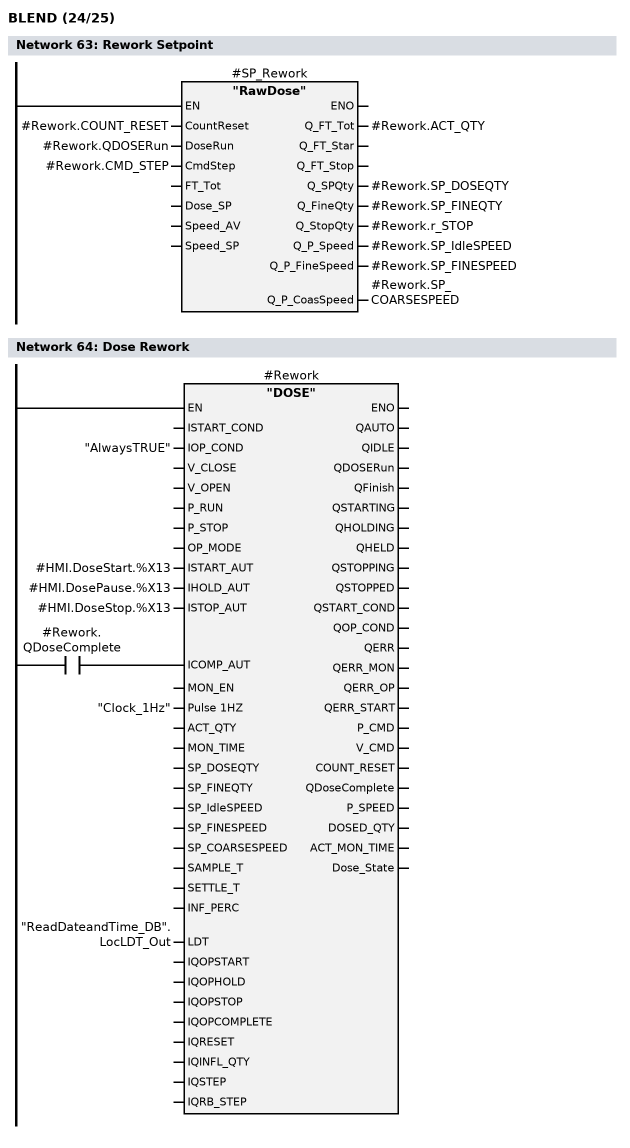
   RUNG wire#powerrail
      #SP_Rework(CountReset := #Rework.COUNT_RESET, DoseRun := #Rework.QDOSERun, CmdStep := #Rework.CMD_STEP, FT_Tot :=, Dose_SP :=, Speed_AV :=, Speed_SP :=, Q_FT_Tot => #Rework.ACT_QTY, Q_FT_Star =>, Q_FT_Stop =>, Q_SPQty => #Rework.SP_DOSEQTY, Q_FineQty => #Rework.SP_FINEQTY, Q_StopQty => #Rework.r_STOP, Q_P_Speed => #Rework.SP_IdleSPEED, Q_P_FineSpeed => #Rework.SP_FINESPEED, Q_P_CoasSpeed => #Rework.SP_COARSESPEED)
   END_RUNG
   // the same network as SCL:
   #SP_Rework(CountReset := #Rework.COUNT_RESET,   // "RawDose"
              DoseRun := #Rework.QDOSERun,
              CmdStep := #Rework.CMD_STEP,
              Q_FT_Tot => #Rework.ACT_QTY,
              Q_SPQty => #Rework.SP_DOSEQTY,
              Q_FineQty => #Rework.SP_FINEQTY,
              Q_StopQty => #Rework.r_STOP,
              Q_P_Speed => #Rework.SP_IdleSPEED,
              Q_P_FineSpeed => #Rework.SP_FINESPEED,
              Q_P_CoasSpeed => #Rework.SP_COARSESPEED);
END_REGION

REGION Network 64: Dose Rework
   RUNG wire#powerrail
      #Rework(ICOMP_AUT := wire#w1, ISTART_COND :=, IOP_COND := "AlwaysTRUE", V_CLOSE :=, V_OPEN :=, P_RUN :=, P_STOP :=, OP_MODE :=, ISTART_AUT := #HMI.DoseStart.%X13, IHOLD_AUT := #HMI.DosePause.%X13, ISTOP_AUT := #HMI.DoseStop.%X13, MON_EN :=, "Pulse 1HZ" := "Clock_1Hz", ACT_QTY :=, MON_TIME :=, SP_DOSEQTY :=, SP_FINEQTY :=, SP_IdleSPEED :=, SP_FINESPEED :=, SP_COARSESPEED :=, SAMPLE_T :=, SETTLE_T :=, INF_PERC :=, LDT := "ReadDateandTime_DB".LocLDT_Out, IQOPSTART :=, IQOPHOLD :=, IQOPSTOP :=, IQOPCOMPLETE :=, IQRESET :=, IQINFL_QTY :=, IQSTEP :=, IQRB_STEP :=, QAUTO =>, QIDLE =>, QDOSERun =>, QFinish =>, QSTARTING =>, QHOLDING =>, QHELD =>, QSTOPPING =>, QSTOPPED =>, QSTART_COND =>, QOP_COND =>, QERR =>, QERR_MON =>, QERR_OP =>, QERR_START =>, P_CMD =>, V_CMD =>, COUNT_RESET =>, QDoseComplete =>, P_SPEED =>, DOSED_QTY =>, ACT_MON_TIME =>, Dose_State =>)
   END_RUNG
   RUNG wire#powerrail
      Contact( #Rework.QDoseComplete )
   END_RUNG wire#w1
   // the same network as SCL:
   #Rework(IOP_COND := "AlwaysTRUE",   // "DOSE"
           ISTART_AUT := #HMI.DoseStart.%X13,
           IHOLD_AUT := #HMI.DosePause.%X13,
           ISTOP_AUT := #HMI.DoseStop.%X13,
           ICOMP_AUT := #Rework.QDoseComplete,
           "Pulse 1HZ" := "Clock_1Hz",
           LDT := "ReadDateandTime_DB".LocLDT_Out);
END_REGION

REGION Network 65: Dose Rework Enable Command
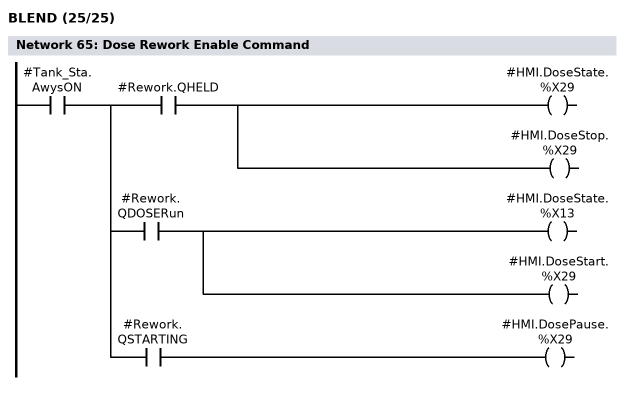
   RUNG wire#powerrail
      Contact( #Tank_Sta.AwysON )
      wire#w1
      Contact( #Rework.QHELD )
      wire#w2
      Coil( #HMI.DoseState.%X29 )
   END_RUNG
   RUNG wire#w2
      Coil( #HMI.DoseStop.%X29 )
   END_RUNG
   RUNG wire#w1
      Contact( #Rework.QDOSERun )
      wire#w3
      Coil( #HMI.DoseState.%X13 )
   END_RUNG
   RUNG wire#w3
      Coil( #HMI.DoseStart.%X29 )
   END_RUNG
   RUNG wire#w1
      Contact( #Rework.QSTARTING )
      Coil( #HMI.DosePause.%X29 )
   END_RUNG
   // the same network as SCL:
   #HMI.DoseState.%X29 := #Tank_Sta.AwysON AND #Rework.QHELD;
   #HMI.DoseStop.%X29 := #HMI.DoseState.%X29;
   #HMI.DoseState.%X13 := #Tank_Sta.AwysON AND #Rework.QDOSERun;
   #HMI.DoseStart.%X29 := #HMI.DoseState.%X13;
   #HMI.DosePause.%X29 := #Tank_Sta.AwysON AND #Rework.QSTARTING;
END_REGION
END_FUNCTION_BLOCK

FUNCTION "Blending" : Void   // FC8, LAD
{ S7_Optimized_Access := 'TRUE' }
VERSION : 0.1
// stored: AutoNumber true, IsIECCheckEnabled false, SetENOAutomatically false, UDAEnableTagReadback false
   VAR_TEMP   // added for the SCL form of the ladder/FBD networks
      _w1 : Bool;
   END_VAR
BEGIN

REGION Network 1
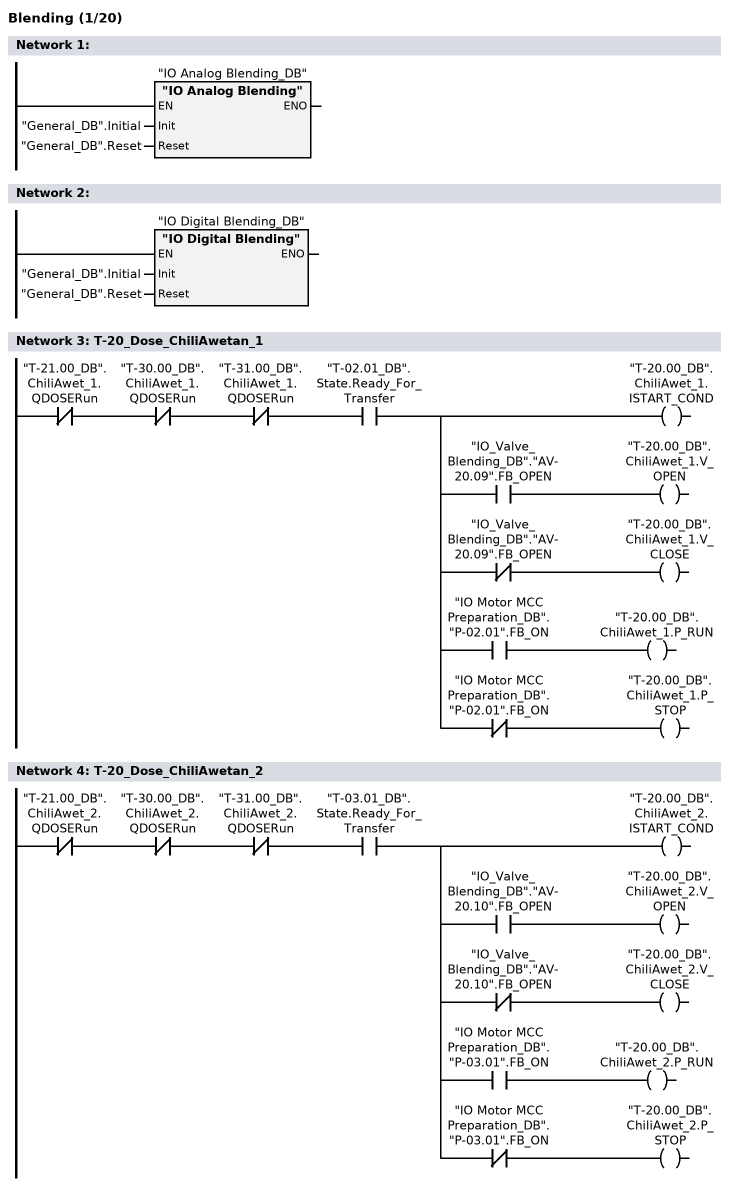
   RUNG wire#powerrail
      "IO Analog Blending_DB"(Init := "General_DB".Initial, Reset := "General_DB".Reset)
   END_RUNG
   // the same network as SCL:
   "IO Analog Blending_DB"(Init := "General_DB".Initial, Reset := "General_DB".Reset);   // "IO Analog Blending"
END_REGION

REGION Network 2
   RUNG wire#powerrail
      "IO Digital Blending_DB"(Init := "General_DB".Initial, Reset := "General_DB".Reset)
   END_RUNG
   // the same network as SCL:
   "IO Digital Blending_DB"(Init := "General_DB".Initial, Reset := "General_DB".Reset);   // "IO Digital Blending"
END_REGION

REGION Network 3: T-20_Dose_ChiliAwetan_1
   RUNG wire#powerrail
      I_Contact( "T-21.00_DB".ChiliAwet_1.QDOSERun )
      I_Contact( "T-30.00_DB".ChiliAwet_1.QDOSERun )
      I_Contact( "T-31.00_DB".ChiliAwet_1.QDOSERun )
      Contact( "T-02.01_DB".State.Ready_For_Transfer )
      wire#w1
      Coil( "T-20.00_DB".ChiliAwet_1.ISTART_COND )
   END_RUNG
   RUNG wire#w1
      Contact( "IO_Valve_Blending_DB"."AV-20.09".FB_OPEN )
      Coil( "T-20.00_DB".ChiliAwet_1.V_OPEN )
   END_RUNG
   RUNG wire#w1
      I_Contact( "IO_Valve_Blending_DB"."AV-20.09".FB_OPEN )
      Coil( "T-20.00_DB".ChiliAwet_1.V_CLOSE )
   END_RUNG
   RUNG wire#w1
      Contact( "IO Motor MCC Preparation_DB"."P-02.01".FB_ON )
      Coil( "T-20.00_DB".ChiliAwet_1.P_RUN )
   END_RUNG
   RUNG wire#w1
      I_Contact( "IO Motor MCC Preparation_DB"."P-02.01".FB_ON )
      Coil( "T-20.00_DB".ChiliAwet_1.P_STOP )
   END_RUNG
   // the same network as SCL:
   "T-20.00_DB".ChiliAwet_1.ISTART_COND := NOT "T-21.00_DB".ChiliAwet_1.QDOSERun AND NOT "T-30.00_DB".ChiliAwet_1.QDOSERun AND NOT "T-31.00_DB".ChiliAwet_1.QDOSERun AND "T-02.01_DB".State.Ready_For_Transfer;
   "T-20.00_DB".ChiliAwet_1.V_OPEN := "T-20.00_DB".ChiliAwet_1.ISTART_COND AND "IO_Valve_Blending_DB"."AV-20.09".FB_OPEN;
   "T-20.00_DB".ChiliAwet_1.V_CLOSE := "T-20.00_DB".ChiliAwet_1.ISTART_COND AND NOT "IO_Valve_Blending_DB"."AV-20.09".FB_OPEN;
   "T-20.00_DB".ChiliAwet_1.P_RUN := "T-20.00_DB".ChiliAwet_1.ISTART_COND AND "IO Motor MCC Preparation_DB"."P-02.01".FB_ON;
   "T-20.00_DB".ChiliAwet_1.P_STOP := "T-20.00_DB".ChiliAwet_1.ISTART_COND AND NOT "IO Motor MCC Preparation_DB"."P-02.01".FB_ON;
END_REGION

REGION Network 4: T-20_Dose_ChiliAwetan_2
   RUNG wire#powerrail
      I_Contact( "T-21.00_DB".ChiliAwet_2.QDOSERun )
      I_Contact( "T-30.00_DB".ChiliAwet_2.QDOSERun )
      I_Contact( "T-31.00_DB".ChiliAwet_2.QDOSERun )
      Contact( "T-03.01_DB".State.Ready_For_Transfer )
      wire#w1
      Coil( "T-20.00_DB".ChiliAwet_2.ISTART_COND )
   END_RUNG
   RUNG wire#w1
      Contact( "IO_Valve_Blending_DB"."AV-20.10".FB_OPEN )
      Coil( "T-20.00_DB".ChiliAwet_2.V_OPEN )
   END_RUNG
   RUNG wire#w1
      I_Contact( "IO_Valve_Blending_DB"."AV-20.10".FB_OPEN )
      Coil( "T-20.00_DB".ChiliAwet_2.V_CLOSE )
   END_RUNG
   RUNG wire#w1
      Contact( "IO Motor MCC Preparation_DB"."P-03.01".FB_ON )
      Coil( "T-20.00_DB".ChiliAwet_2.P_RUN )
   END_RUNG
   RUNG wire#w1
      I_Contact( "IO Motor MCC Preparation_DB"."P-03.01".FB_ON )
      Coil( "T-20.00_DB".ChiliAwet_2.P_STOP )
   END_RUNG
   // the same network as SCL:
   "T-20.00_DB".ChiliAwet_2.ISTART_COND := NOT "T-21.00_DB".ChiliAwet_2.QDOSERun AND NOT "T-30.00_DB".ChiliAwet_2.QDOSERun AND NOT "T-31.00_DB".ChiliAwet_2.QDOSERun AND "T-03.01_DB".State.Ready_For_Transfer;
   "T-20.00_DB".ChiliAwet_2.V_OPEN := "T-20.00_DB".ChiliAwet_2.ISTART_COND AND "IO_Valve_Blending_DB"."AV-20.10".FB_OPEN;
   "T-20.00_DB".ChiliAwet_2.V_CLOSE := "T-20.00_DB".ChiliAwet_2.ISTART_COND AND NOT "IO_Valve_Blending_DB"."AV-20.10".FB_OPEN;
   "T-20.00_DB".ChiliAwet_2.P_RUN := "T-20.00_DB".ChiliAwet_2.ISTART_COND AND "IO Motor MCC Preparation_DB"."P-03.01".FB_ON;
   "T-20.00_DB".ChiliAwet_2.P_STOP := "T-20.00_DB".ChiliAwet_2.ISTART_COND AND NOT "IO Motor MCC Preparation_DB"."P-03.01".FB_ON;
END_REGION

REGION Network 5: T-20_Dose_ChiliAwetan_3
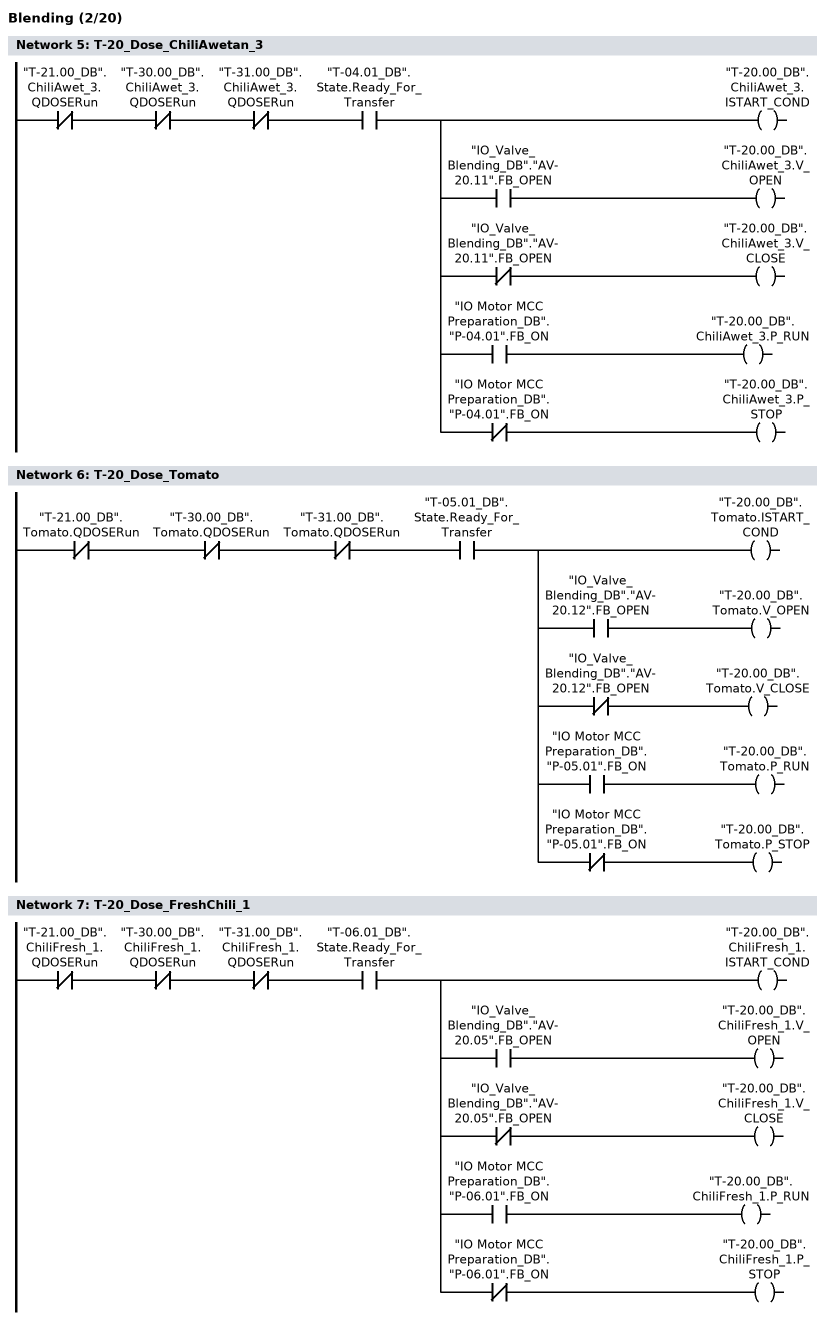
   RUNG wire#powerrail
      I_Contact( "T-21.00_DB".ChiliAwet_3.QDOSERun )
      I_Contact( "T-30.00_DB".ChiliAwet_3.QDOSERun )
      I_Contact( "T-31.00_DB".ChiliAwet_3.QDOSERun )
      Contact( "T-04.01_DB".State.Ready_For_Transfer )
      wire#w1
      Coil( "T-20.00_DB".ChiliAwet_3.ISTART_COND )
   END_RUNG
   RUNG wire#w1
      Contact( "IO_Valve_Blending_DB"."AV-20.11".FB_OPEN )
      Coil( "T-20.00_DB".ChiliAwet_3.V_OPEN )
   END_RUNG
   RUNG wire#w1
      I_Contact( "IO_Valve_Blending_DB"."AV-20.11".FB_OPEN )
      Coil( "T-20.00_DB".ChiliAwet_3.V_CLOSE )
   END_RUNG
   RUNG wire#w1
      Contact( "IO Motor MCC Preparation_DB"."P-04.01".FB_ON )
      Coil( "T-20.00_DB".ChiliAwet_3.P_RUN )
   END_RUNG
   RUNG wire#w1
      I_Contact( "IO Motor MCC Preparation_DB"."P-04.01".FB_ON )
      Coil( "T-20.00_DB".ChiliAwet_3.P_STOP )
   END_RUNG
   // the same network as SCL:
   "T-20.00_DB".ChiliAwet_3.ISTART_COND := NOT "T-21.00_DB".ChiliAwet_3.QDOSERun AND NOT "T-30.00_DB".ChiliAwet_3.QDOSERun AND NOT "T-31.00_DB".ChiliAwet_3.QDOSERun AND "T-04.01_DB".State.Ready_For_Transfer;
   "T-20.00_DB".ChiliAwet_3.V_OPEN := "T-20.00_DB".ChiliAwet_3.ISTART_COND AND "IO_Valve_Blending_DB"."AV-20.11".FB_OPEN;
   "T-20.00_DB".ChiliAwet_3.V_CLOSE := "T-20.00_DB".ChiliAwet_3.ISTART_COND AND NOT "IO_Valve_Blending_DB"."AV-20.11".FB_OPEN;
   "T-20.00_DB".ChiliAwet_3.P_RUN := "T-20.00_DB".ChiliAwet_3.ISTART_COND AND "IO Motor MCC Preparation_DB"."P-04.01".FB_ON;
   "T-20.00_DB".ChiliAwet_3.P_STOP := "T-20.00_DB".ChiliAwet_3.ISTART_COND AND NOT "IO Motor MCC Preparation_DB"."P-04.01".FB_ON;
END_REGION

REGION Network 6: T-20_Dose_Tomato
   RUNG wire#powerrail
      I_Contact( "T-21.00_DB".Tomato.QDOSERun )
      I_Contact( "T-30.00_DB".Tomato.QDOSERun )
      I_Contact( "T-31.00_DB".Tomato.QDOSERun )
      Contact( "T-05.01_DB".State.Ready_For_Transfer )
      wire#w1
      Coil( "T-20.00_DB".Tomato.ISTART_COND )
   END_RUNG
   RUNG wire#w1
      Contact( "IO_Valve_Blending_DB"."AV-20.12".FB_OPEN )
      Coil( "T-20.00_DB".Tomato.V_OPEN )
   END_RUNG
   RUNG wire#w1
      I_Contact( "IO_Valve_Blending_DB"."AV-20.12".FB_OPEN )
      Coil( "T-20.00_DB".Tomato.V_CLOSE )
   END_RUNG
   RUNG wire#w1
      Contact( "IO Motor MCC Preparation_DB"."P-05.01".FB_ON )
      Coil( "T-20.00_DB".Tomato.P_RUN )
   END_RUNG
   RUNG wire#w1
      I_Contact( "IO Motor MCC Preparation_DB"."P-05.01".FB_ON )
      Coil( "T-20.00_DB".Tomato.P_STOP )
   END_RUNG
   // the same network as SCL:
   "T-20.00_DB".Tomato.ISTART_COND := NOT "T-21.00_DB".Tomato.QDOSERun AND NOT "T-30.00_DB".Tomato.QDOSERun AND NOT "T-31.00_DB".Tomato.QDOSERun AND "T-05.01_DB".State.Ready_For_Transfer;
   "T-20.00_DB".Tomato.V_OPEN := "T-20.00_DB".Tomato.ISTART_COND AND "IO_Valve_Blending_DB"."AV-20.12".FB_OPEN;
   "T-20.00_DB".Tomato.V_CLOSE := "T-20.00_DB".Tomato.ISTART_COND AND NOT "IO_Valve_Blending_DB"."AV-20.12".FB_OPEN;
   "T-20.00_DB".Tomato.P_RUN := "T-20.00_DB".Tomato.ISTART_COND AND "IO Motor MCC Preparation_DB"."P-05.01".FB_ON;
   "T-20.00_DB".Tomato.P_STOP := "T-20.00_DB".Tomato.ISTART_COND AND NOT "IO Motor MCC Preparation_DB"."P-05.01".FB_ON;
END_REGION

REGION Network 7: T-20_Dose_FreshChili_1
   RUNG wire#powerrail
      I_Contact( "T-21.00_DB".ChiliFresh_1.QDOSERun )
      I_Contact( "T-30.00_DB".ChiliFresh_1.QDOSERun )
      I_Contact( "T-31.00_DB".ChiliFresh_1.QDOSERun )
      Contact( "T-06.01_DB".State.Ready_For_Transfer )
      wire#w1
      Coil( "T-20.00_DB".ChiliFresh_1.ISTART_COND )
   END_RUNG
   RUNG wire#w1
      Contact( "IO_Valve_Blending_DB"."AV-20.05".FB_OPEN )
      Coil( "T-20.00_DB".ChiliFresh_1.V_OPEN )
   END_RUNG
   RUNG wire#w1
      I_Contact( "IO_Valve_Blending_DB"."AV-20.05".FB_OPEN )
      Coil( "T-20.00_DB".ChiliFresh_1.V_CLOSE )
   END_RUNG
   RUNG wire#w1
      Contact( "IO Motor MCC Preparation_DB"."P-06.01".FB_ON )
      Coil( "T-20.00_DB".ChiliFresh_1.P_RUN )
   END_RUNG
   RUNG wire#w1
      I_Contact( "IO Motor MCC Preparation_DB"."P-06.01".FB_ON )
      Coil( "T-20.00_DB".ChiliFresh_1.P_STOP )
   END_RUNG
   // the same network as SCL:
   "T-20.00_DB".ChiliFresh_1.ISTART_COND := NOT "T-21.00_DB".ChiliFresh_1.QDOSERun AND NOT "T-30.00_DB".ChiliFresh_1.QDOSERun AND NOT "T-31.00_DB".ChiliFresh_1.QDOSERun AND "T-06.01_DB".State.Ready_For_Transfer;
   "T-20.00_DB".ChiliFresh_1.V_OPEN := "T-20.00_DB".ChiliFresh_1.ISTART_COND AND "IO_Valve_Blending_DB"."AV-20.05".FB_OPEN;
   "T-20.00_DB".ChiliFresh_1.V_CLOSE := "T-20.00_DB".ChiliFresh_1.ISTART_COND AND NOT "IO_Valve_Blending_DB"."AV-20.05".FB_OPEN;
   "T-20.00_DB".ChiliFresh_1.P_RUN := "T-20.00_DB".ChiliFresh_1.ISTART_COND AND "IO Motor MCC Preparation_DB"."P-06.01".FB_ON;
   "T-20.00_DB".ChiliFresh_1.P_STOP := "T-20.00_DB".ChiliFresh_1.ISTART_COND AND NOT "IO Motor MCC Preparation_DB"."P-06.01".FB_ON;
END_REGION

REGION Network 8: T-20_Dose_FreshChili_2
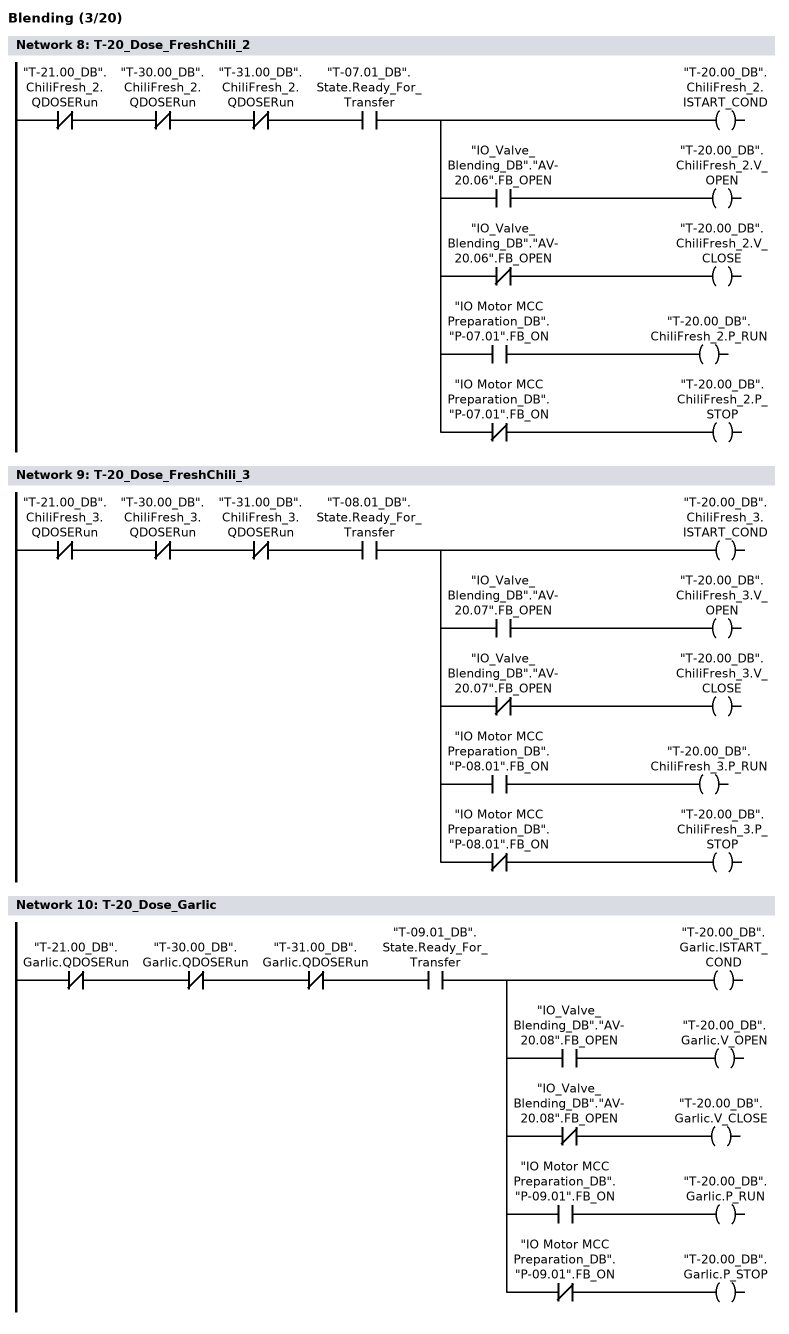
   RUNG wire#powerrail
      I_Contact( "T-21.00_DB".ChiliFresh_2.QDOSERun )
      I_Contact( "T-30.00_DB".ChiliFresh_2.QDOSERun )
      I_Contact( "T-31.00_DB".ChiliFresh_2.QDOSERun )
      Contact( "T-07.01_DB".State.Ready_For_Transfer )
      wire#w1
      Coil( "T-20.00_DB".ChiliFresh_2.ISTART_COND )
   END_RUNG
   RUNG wire#w1
      Contact( "IO_Valve_Blending_DB"."AV-20.06".FB_OPEN )
      Coil( "T-20.00_DB".ChiliFresh_2.V_OPEN )
   END_RUNG
   RUNG wire#w1
      I_Contact( "IO_Valve_Blending_DB"."AV-20.06".FB_OPEN )
      Coil( "T-20.00_DB".ChiliFresh_2.V_CLOSE )
   END_RUNG
   RUNG wire#w1
      Contact( "IO Motor MCC Preparation_DB"."P-07.01".FB_ON )
      Coil( "T-20.00_DB".ChiliFresh_2.P_RUN )
   END_RUNG
   RUNG wire#w1
      I_Contact( "IO Motor MCC Preparation_DB"."P-07.01".FB_ON )
      Coil( "T-20.00_DB".ChiliFresh_2.P_STOP )
   END_RUNG
   // the same network as SCL:
   "T-20.00_DB".ChiliFresh_2.ISTART_COND := NOT "T-21.00_DB".ChiliFresh_2.QDOSERun AND NOT "T-30.00_DB".ChiliFresh_2.QDOSERun AND NOT "T-31.00_DB".ChiliFresh_2.QDOSERun AND "T-07.01_DB".State.Ready_For_Transfer;
   "T-20.00_DB".ChiliFresh_2.V_OPEN := "T-20.00_DB".ChiliFresh_2.ISTART_COND AND "IO_Valve_Blending_DB"."AV-20.06".FB_OPEN;
   "T-20.00_DB".ChiliFresh_2.V_CLOSE := "T-20.00_DB".ChiliFresh_2.ISTART_COND AND NOT "IO_Valve_Blending_DB"."AV-20.06".FB_OPEN;
   "T-20.00_DB".ChiliFresh_2.P_RUN := "T-20.00_DB".ChiliFresh_2.ISTART_COND AND "IO Motor MCC Preparation_DB"."P-07.01".FB_ON;
   "T-20.00_DB".ChiliFresh_2.P_STOP := "T-20.00_DB".ChiliFresh_2.ISTART_COND AND NOT "IO Motor MCC Preparation_DB"."P-07.01".FB_ON;
END_REGION

REGION Network 9: T-20_Dose_FreshChili_3
   RUNG wire#powerrail
      I_Contact( "T-21.00_DB".ChiliFresh_3.QDOSERun )
      I_Contact( "T-30.00_DB".ChiliFresh_3.QDOSERun )
      I_Contact( "T-31.00_DB".ChiliFresh_3.QDOSERun )
      Contact( "T-08.01_DB".State.Ready_For_Transfer )
      wire#w1
      Coil( "T-20.00_DB".ChiliFresh_3.ISTART_COND )
   END_RUNG
   RUNG wire#w1
      Contact( "IO_Valve_Blending_DB"."AV-20.07".FB_OPEN )
      Coil( "T-20.00_DB".ChiliFresh_3.V_OPEN )
   END_RUNG
   RUNG wire#w1
      I_Contact( "IO_Valve_Blending_DB"."AV-20.07".FB_OPEN )
      Coil( "T-20.00_DB".ChiliFresh_3.V_CLOSE )
   END_RUNG
   RUNG wire#w1
      Contact( "IO Motor MCC Preparation_DB"."P-08.01".FB_ON )
      Coil( "T-20.00_DB".ChiliFresh_3.P_RUN )
   END_RUNG
   RUNG wire#w1
      I_Contact( "IO Motor MCC Preparation_DB"."P-08.01".FB_ON )
      Coil( "T-20.00_DB".ChiliFresh_3.P_STOP )
   END_RUNG
   // the same network as SCL:
   "T-20.00_DB".ChiliFresh_3.ISTART_COND := NOT "T-21.00_DB".ChiliFresh_3.QDOSERun AND NOT "T-30.00_DB".ChiliFresh_3.QDOSERun AND NOT "T-31.00_DB".ChiliFresh_3.QDOSERun AND "T-08.01_DB".State.Ready_For_Transfer;
   "T-20.00_DB".ChiliFresh_3.V_OPEN := "T-20.00_DB".ChiliFresh_3.ISTART_COND AND "IO_Valve_Blending_DB"."AV-20.07".FB_OPEN;
   "T-20.00_DB".ChiliFresh_3.V_CLOSE := "T-20.00_DB".ChiliFresh_3.ISTART_COND AND NOT "IO_Valve_Blending_DB"."AV-20.07".FB_OPEN;
   "T-20.00_DB".ChiliFresh_3.P_RUN := "T-20.00_DB".ChiliFresh_3.ISTART_COND AND "IO Motor MCC Preparation_DB"."P-08.01".FB_ON;
   "T-20.00_DB".ChiliFresh_3.P_STOP := "T-20.00_DB".ChiliFresh_3.ISTART_COND AND NOT "IO Motor MCC Preparation_DB"."P-08.01".FB_ON;
END_REGION

REGION Network 10: T-20_Dose_Garlic
   RUNG wire#powerrail
      I_Contact( "T-21.00_DB".Garlic.QDOSERun )
      I_Contact( "T-30.00_DB".Garlic.QDOSERun )
      I_Contact( "T-31.00_DB".Garlic.QDOSERun )
      Contact( "T-09.01_DB".State.Ready_For_Transfer )
      wire#w1
      Coil( "T-20.00_DB".Garlic.ISTART_COND )
   END_RUNG
   RUNG wire#w1
      Contact( "IO_Valve_Blending_DB"."AV-20.08".FB_OPEN )
      Coil( "T-20.00_DB".Garlic.V_OPEN )
   END_RUNG
   RUNG wire#w1
      I_Contact( "IO_Valve_Blending_DB"."AV-20.08".FB_OPEN )
      Coil( "T-20.00_DB".Garlic.V_CLOSE )
   END_RUNG
   RUNG wire#w1
      Contact( "IO Motor MCC Preparation_DB"."P-09.01".FB_ON )
      Coil( "T-20.00_DB".Garlic.P_RUN )
   END_RUNG
   RUNG wire#w1
      I_Contact( "IO Motor MCC Preparation_DB"."P-09.01".FB_ON )
      Coil( "T-20.00_DB".Garlic.P_STOP )
   END_RUNG
   // the same network as SCL:
   "T-20.00_DB".Garlic.ISTART_COND := NOT "T-21.00_DB".Garlic.QDOSERun AND NOT "T-30.00_DB".Garlic.QDOSERun AND NOT "T-31.00_DB".Garlic.QDOSERun AND "T-09.01_DB".State.Ready_For_Transfer;
   "T-20.00_DB".Garlic.V_OPEN := "T-20.00_DB".Garlic.ISTART_COND AND "IO_Valve_Blending_DB"."AV-20.08".FB_OPEN;
   "T-20.00_DB".Garlic.V_CLOSE := "T-20.00_DB".Garlic.ISTART_COND AND NOT "IO_Valve_Blending_DB"."AV-20.08".FB_OPEN;
   "T-20.00_DB".Garlic.P_RUN := "T-20.00_DB".Garlic.ISTART_COND AND "IO Motor MCC Preparation_DB"."P-09.01".FB_ON;
   "T-20.00_DB".Garlic.P_STOP := "T-20.00_DB".Garlic.ISTART_COND AND NOT "IO Motor MCC Preparation_DB"."P-09.01".FB_ON;
END_REGION

REGION Network 11: T-20_Dose_Vinegar
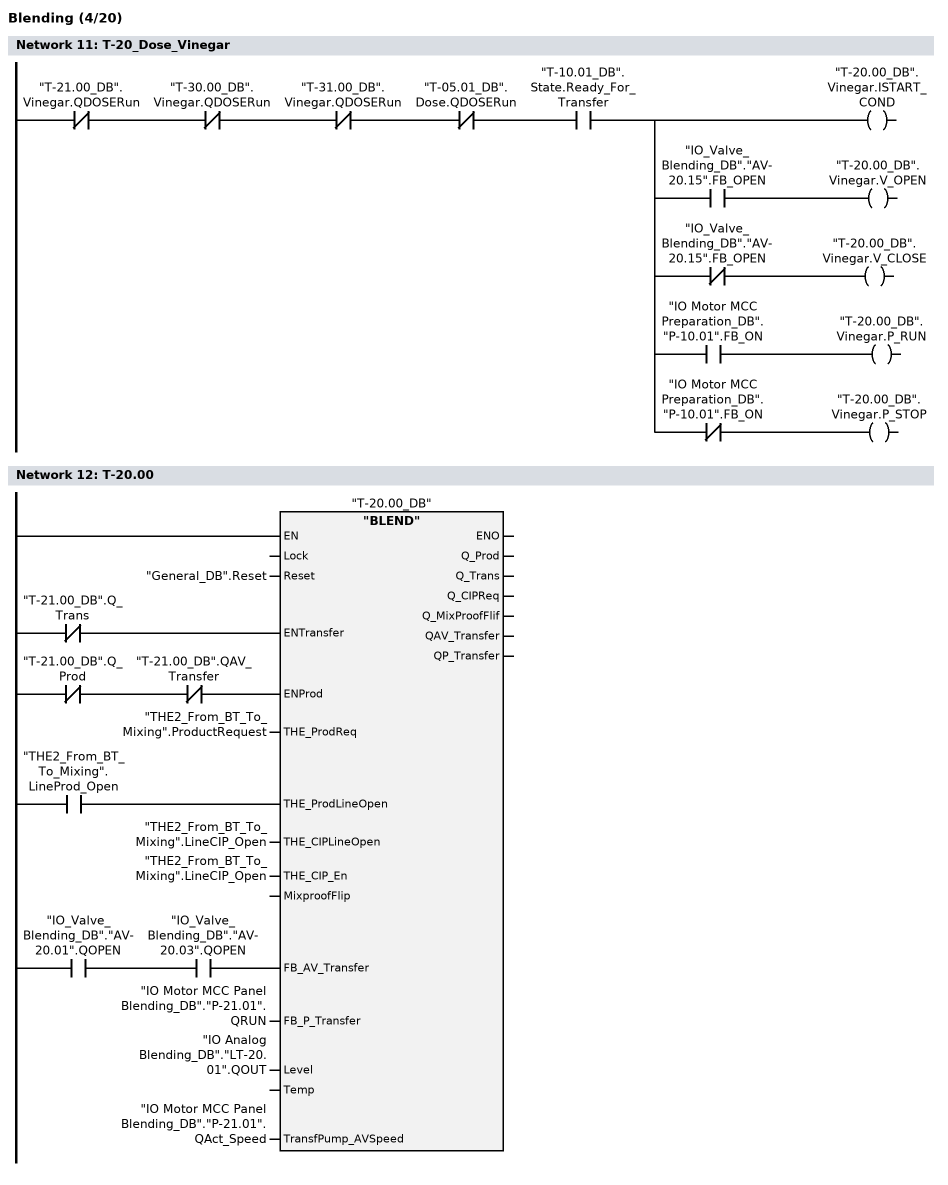
   RUNG wire#powerrail
      I_Contact( "T-21.00_DB".Vinegar.QDOSERun )
      I_Contact( "T-30.00_DB".Vinegar.QDOSERun )
      I_Contact( "T-31.00_DB".Vinegar.QDOSERun )
      I_Contact( "T-05.01_DB".Dose.QDOSERun )
      Contact( "T-10.01_DB".State.Ready_For_Transfer )
      wire#w1
      Coil( "T-20.00_DB".Vinegar.ISTART_COND )
   END_RUNG
   RUNG wire#w1
      Contact( "IO_Valve_Blending_DB"."AV-20.15".FB_OPEN )
      Coil( "T-20.00_DB".Vinegar.V_OPEN )
   END_RUNG
   RUNG wire#w1
      I_Contact( "IO_Valve_Blending_DB"."AV-20.15".FB_OPEN )
      Coil( "T-20.00_DB".Vinegar.V_CLOSE )
   END_RUNG
   RUNG wire#w1
      Contact( "IO Motor MCC Preparation_DB"."P-10.01".FB_ON )
      Coil( "T-20.00_DB".Vinegar.P_RUN )
   END_RUNG
   RUNG wire#w1
      I_Contact( "IO Motor MCC Preparation_DB"."P-10.01".FB_ON )
      Coil( "T-20.00_DB".Vinegar.P_STOP )
   END_RUNG
   // the same network as SCL:
   "T-20.00_DB".Vinegar.ISTART_COND := NOT "T-21.00_DB".Vinegar.QDOSERun AND NOT "T-30.00_DB".Vinegar.QDOSERun AND NOT "T-31.00_DB".Vinegar.QDOSERun AND NOT "T-05.01_DB".Dose.QDOSERun AND "T-10.01_DB".State.Ready_For_Transfer;
   "T-20.00_DB".Vinegar.V_OPEN := "T-20.00_DB".Vinegar.ISTART_COND AND "IO_Valve_Blending_DB"."AV-20.15".FB_OPEN;
   "T-20.00_DB".Vinegar.V_CLOSE := "T-20.00_DB".Vinegar.ISTART_COND AND NOT "IO_Valve_Blending_DB"."AV-20.15".FB_OPEN;
   "T-20.00_DB".Vinegar.P_RUN := "T-20.00_DB".Vinegar.ISTART_COND AND "IO Motor MCC Preparation_DB"."P-10.01".FB_ON;
   "T-20.00_DB".Vinegar.P_STOP := "T-20.00_DB".Vinegar.ISTART_COND AND NOT "IO Motor MCC Preparation_DB"."P-10.01".FB_ON;
END_REGION

REGION Network 12: T-20.00
   RUNG wire#powerrail
      "T-20.00_DB"(ENTransfer := wire#w1, ENProd := wire#w2, THE_ProdLineOpen := wire#w3, FB_AV_Transfer := wire#w4, Lock :=, Reset := "General_DB".Reset, THE_ProdReq := "THE2_From_BT_To_Mixing".ProductRequest, THE_CIPLineOpen := "THE2_From_BT_To_Mixing".LineCIP_Open, THE_CIP_En := "THE2_From_BT_To_Mixing".LineCIP_Open, MixproofFlip :=, FB_P_Transfer := "IO Motor MCC Panel Blending_DB"."P-21.01".QRUN, Level := "IO Analog Blending_DB"."LT-20.01".QOUT, Temp :=, TransfPump_AVSpeed := "IO Motor MCC Panel Blending_DB"."P-21.01".QAct_Speed, Q_Prod =>, Q_Trans =>, Q_CIPReq =>, Q_MixProofFlif =>, QAV_Transfer =>, QP_Transfer =>)
   END_RUNG
   RUNG wire#powerrail
      I_Contact( "T-21.00_DB".Q_Trans )
   END_RUNG wire#w1
   RUNG wire#powerrail
      I_Contact( "T-21.00_DB".Q_Prod )
      I_Contact( "T-21.00_DB".QAV_Transfer )
   END_RUNG wire#w2
   RUNG wire#powerrail
      Contact( "THE2_From_BT_To_Mixing".LineProd_Open )
   END_RUNG wire#w3
   RUNG wire#powerrail
      Contact( "IO_Valve_Blending_DB"."AV-20.01".QOPEN )
      Contact( "IO_Valve_Blending_DB"."AV-20.03".QOPEN )
   END_RUNG wire#w4
   // the same network as SCL:
   "T-20.00_DB"(Reset := "General_DB".Reset,   // "BLEND"
                ENTransfer := NOT "T-21.00_DB".Q_Trans,
                ENProd := NOT "T-21.00_DB".Q_Prod AND NOT "T-21.00_DB".QAV_Transfer,
                THE_ProdReq := "THE2_From_BT_To_Mixing".ProductRequest,
                THE_ProdLineOpen := "THE2_From_BT_To_Mixing".LineProd_Open,
                THE_CIPLineOpen := "THE2_From_BT_To_Mixing".LineCIP_Open,
                THE_CIP_En := "THE2_From_BT_To_Mixing".LineCIP_Open,
                FB_AV_Transfer := "IO_Valve_Blending_DB"."AV-20.01".QOPEN AND "IO_Valve_Blending_DB"."AV-20.03".QOPEN,
                FB_P_Transfer := "IO Motor MCC Panel Blending_DB"."P-21.01".QRUN,
                Level := "IO Analog Blending_DB"."LT-20.01".QOUT,
                TransfPump_AVSpeed := "IO Motor MCC Panel Blending_DB"."P-21.01".QAct_Speed);
END_REGION

REGION Network 14: T-21_Dose_ChiliAwetan_1
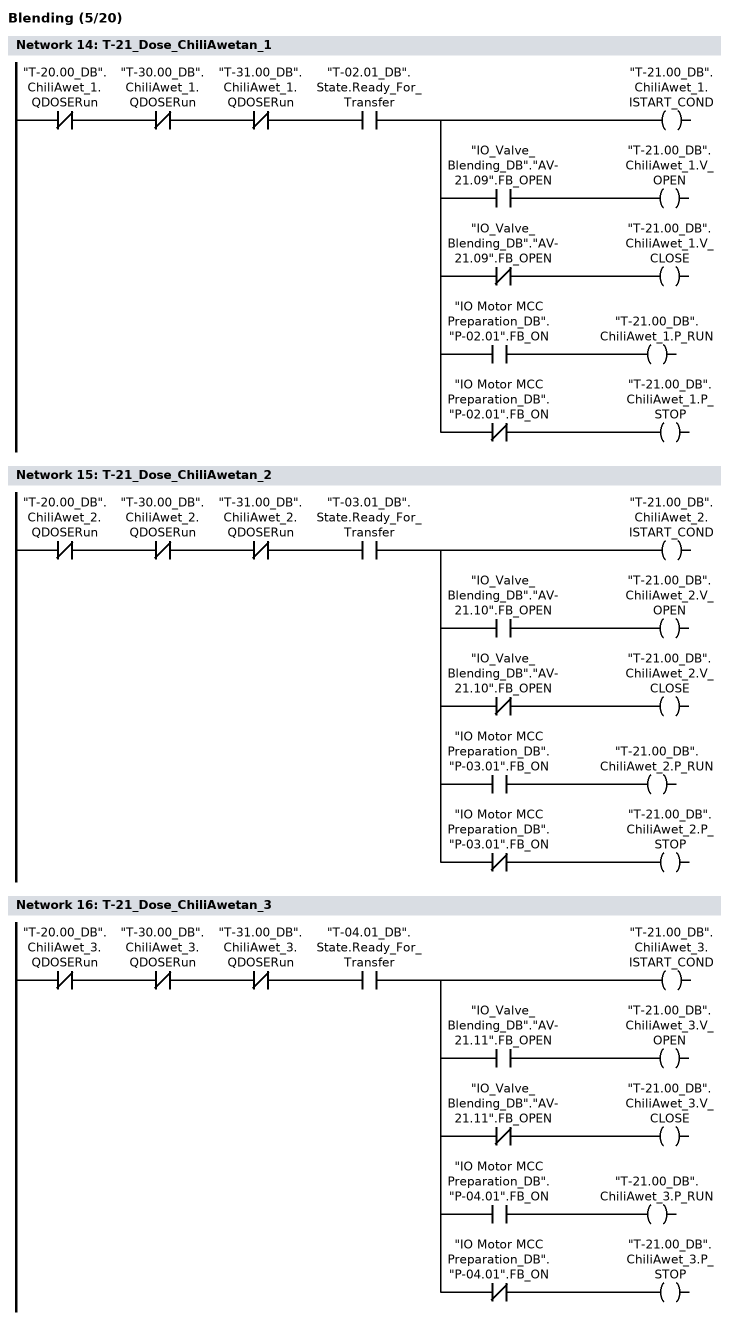
   RUNG wire#powerrail
      I_Contact( "T-20.00_DB".ChiliAwet_1.QDOSERun )
      I_Contact( "T-30.00_DB".ChiliAwet_1.QDOSERun )
      I_Contact( "T-31.00_DB".ChiliAwet_1.QDOSERun )
      Contact( "T-02.01_DB".State.Ready_For_Transfer )
      wire#w1
      Coil( "T-21.00_DB".ChiliAwet_1.ISTART_COND )
   END_RUNG
   RUNG wire#w1
      Contact( "IO_Valve_Blending_DB"."AV-21.09".FB_OPEN )
      Coil( "T-21.00_DB".ChiliAwet_1.V_OPEN )
   END_RUNG
   RUNG wire#w1
      I_Contact( "IO_Valve_Blending_DB"."AV-21.09".FB_OPEN )
      Coil( "T-21.00_DB".ChiliAwet_1.V_CLOSE )
   END_RUNG
   RUNG wire#w1
      Contact( "IO Motor MCC Preparation_DB"."P-02.01".FB_ON )
      Coil( "T-21.00_DB".ChiliAwet_1.P_RUN )
   END_RUNG
   RUNG wire#w1
      I_Contact( "IO Motor MCC Preparation_DB"."P-02.01".FB_ON )
      Coil( "T-21.00_DB".ChiliAwet_1.P_STOP )
   END_RUNG
   // the same network as SCL:
   "T-21.00_DB".ChiliAwet_1.ISTART_COND := NOT "T-20.00_DB".ChiliAwet_1.QDOSERun AND NOT "T-30.00_DB".ChiliAwet_1.QDOSERun AND NOT "T-31.00_DB".ChiliAwet_1.QDOSERun AND "T-02.01_DB".State.Ready_For_Transfer;
   "T-21.00_DB".ChiliAwet_1.V_OPEN := "T-21.00_DB".ChiliAwet_1.ISTART_COND AND "IO_Valve_Blending_DB"."AV-21.09".FB_OPEN;
   "T-21.00_DB".ChiliAwet_1.V_CLOSE := "T-21.00_DB".ChiliAwet_1.ISTART_COND AND NOT "IO_Valve_Blending_DB"."AV-21.09".FB_OPEN;
   "T-21.00_DB".ChiliAwet_1.P_RUN := "T-21.00_DB".ChiliAwet_1.ISTART_COND AND "IO Motor MCC Preparation_DB"."P-02.01".FB_ON;
   "T-21.00_DB".ChiliAwet_1.P_STOP := "T-21.00_DB".ChiliAwet_1.ISTART_COND AND NOT "IO Motor MCC Preparation_DB"."P-02.01".FB_ON;
END_REGION

REGION Network 15: T-21_Dose_ChiliAwetan_2
   RUNG wire#powerrail
      I_Contact( "T-20.00_DB".ChiliAwet_2.QDOSERun )
      I_Contact( "T-30.00_DB".ChiliAwet_2.QDOSERun )
      I_Contact( "T-31.00_DB".ChiliAwet_2.QDOSERun )
      Contact( "T-03.01_DB".State.Ready_For_Transfer )
      wire#w1
      Coil( "T-21.00_DB".ChiliAwet_2.ISTART_COND )
   END_RUNG
   RUNG wire#w1
      Contact( "IO_Valve_Blending_DB"."AV-21.10".FB_OPEN )
      Coil( "T-21.00_DB".ChiliAwet_2.V_OPEN )
   END_RUNG
   RUNG wire#w1
      I_Contact( "IO_Valve_Blending_DB"."AV-21.10".FB_OPEN )
      Coil( "T-21.00_DB".ChiliAwet_2.V_CLOSE )
   END_RUNG
   RUNG wire#w1
      Contact( "IO Motor MCC Preparation_DB"."P-03.01".FB_ON )
      Coil( "T-21.00_DB".ChiliAwet_2.P_RUN )
   END_RUNG
   RUNG wire#w1
      I_Contact( "IO Motor MCC Preparation_DB"."P-03.01".FB_ON )
      Coil( "T-21.00_DB".ChiliAwet_2.P_STOP )
   END_RUNG
   // the same network as SCL:
   "T-21.00_DB".ChiliAwet_2.ISTART_COND := NOT "T-20.00_DB".ChiliAwet_2.QDOSERun AND NOT "T-30.00_DB".ChiliAwet_2.QDOSERun AND NOT "T-31.00_DB".ChiliAwet_2.QDOSERun AND "T-03.01_DB".State.Ready_For_Transfer;
   "T-21.00_DB".ChiliAwet_2.V_OPEN := "T-21.00_DB".ChiliAwet_2.ISTART_COND AND "IO_Valve_Blending_DB"."AV-21.10".FB_OPEN;
   "T-21.00_DB".ChiliAwet_2.V_CLOSE := "T-21.00_DB".ChiliAwet_2.ISTART_COND AND NOT "IO_Valve_Blending_DB"."AV-21.10".FB_OPEN;
   "T-21.00_DB".ChiliAwet_2.P_RUN := "T-21.00_DB".ChiliAwet_2.ISTART_COND AND "IO Motor MCC Preparation_DB"."P-03.01".FB_ON;
   "T-21.00_DB".ChiliAwet_2.P_STOP := "T-21.00_DB".ChiliAwet_2.ISTART_COND AND NOT "IO Motor MCC Preparation_DB"."P-03.01".FB_ON;
END_REGION

REGION Network 16: T-21_Dose_ChiliAwetan_3
   RUNG wire#powerrail
      I_Contact( "T-20.00_DB".ChiliAwet_3.QDOSERun )
      I_Contact( "T-30.00_DB".ChiliAwet_3.QDOSERun )
      I_Contact( "T-31.00_DB".ChiliAwet_3.QDOSERun )
      Contact( "T-04.01_DB".State.Ready_For_Transfer )
      wire#w1
      Coil( "T-21.00_DB".ChiliAwet_3.ISTART_COND )
   END_RUNG
   RUNG wire#w1
      Contact( "IO_Valve_Blending_DB"."AV-21.11".FB_OPEN )
      Coil( "T-21.00_DB".ChiliAwet_3.V_OPEN )
   END_RUNG
   RUNG wire#w1
      I_Contact( "IO_Valve_Blending_DB"."AV-21.11".FB_OPEN )
      Coil( "T-21.00_DB".ChiliAwet_3.V_CLOSE )
   END_RUNG
   RUNG wire#w1
      Contact( "IO Motor MCC Preparation_DB"."P-04.01".FB_ON )
      Coil( "T-21.00_DB".ChiliAwet_3.P_RUN )
   END_RUNG
   RUNG wire#w1
      I_Contact( "IO Motor MCC Preparation_DB"."P-04.01".FB_ON )
      Coil( "T-21.00_DB".ChiliAwet_3.P_STOP )
   END_RUNG
   // the same network as SCL:
   "T-21.00_DB".ChiliAwet_3.ISTART_COND := NOT "T-20.00_DB".ChiliAwet_3.QDOSERun AND NOT "T-30.00_DB".ChiliAwet_3.QDOSERun AND NOT "T-31.00_DB".ChiliAwet_3.QDOSERun AND "T-04.01_DB".State.Ready_For_Transfer;
   "T-21.00_DB".ChiliAwet_3.V_OPEN := "T-21.00_DB".ChiliAwet_3.ISTART_COND AND "IO_Valve_Blending_DB"."AV-21.11".FB_OPEN;
   "T-21.00_DB".ChiliAwet_3.V_CLOSE := "T-21.00_DB".ChiliAwet_3.ISTART_COND AND NOT "IO_Valve_Blending_DB"."AV-21.11".FB_OPEN;
   "T-21.00_DB".ChiliAwet_3.P_RUN := "T-21.00_DB".ChiliAwet_3.ISTART_COND AND "IO Motor MCC Preparation_DB"."P-04.01".FB_ON;
   "T-21.00_DB".ChiliAwet_3.P_STOP := "T-21.00_DB".ChiliAwet_3.ISTART_COND AND NOT "IO Motor MCC Preparation_DB"."P-04.01".FB_ON;
END_REGION

REGION Network 17: T-21_Dose_Tomato
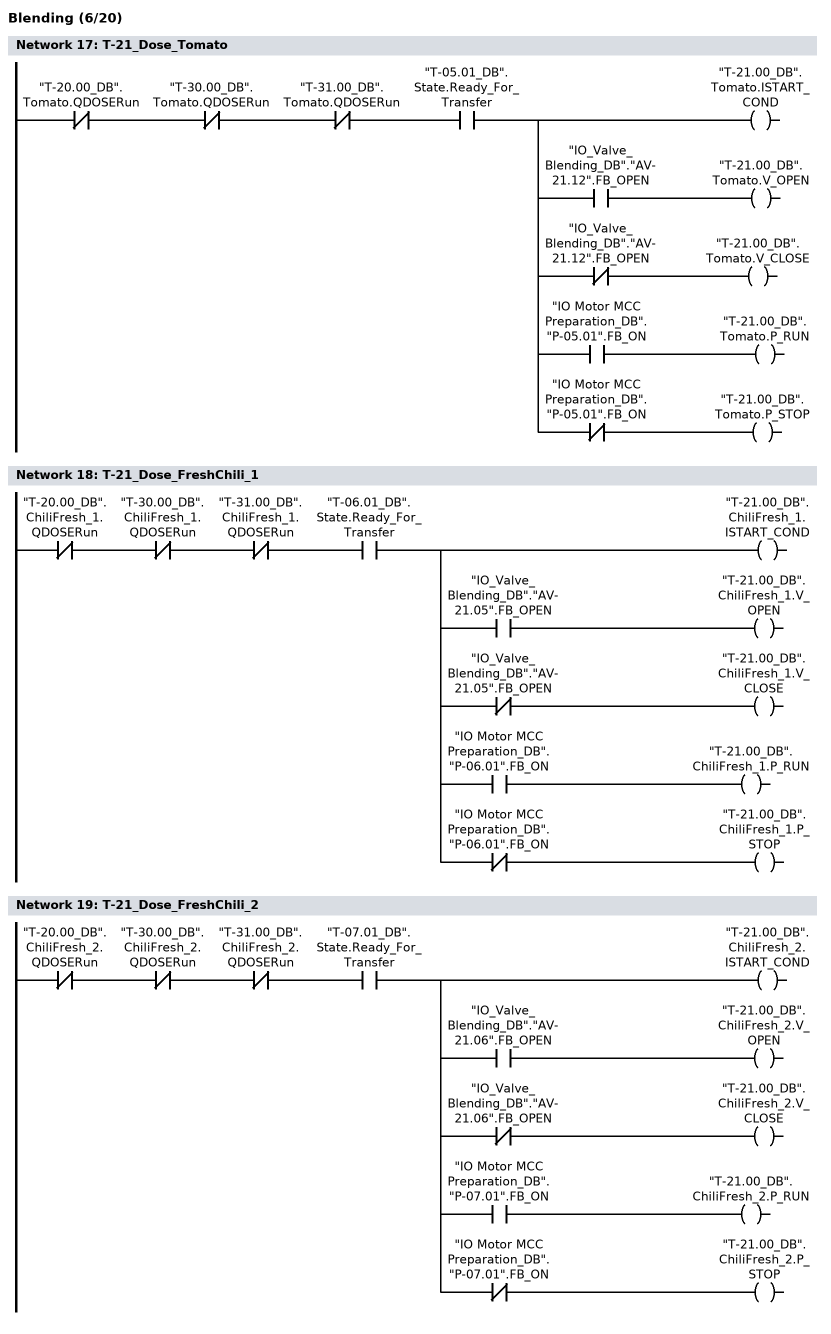
   RUNG wire#powerrail
      I_Contact( "T-20.00_DB".Tomato.QDOSERun )
      I_Contact( "T-30.00_DB".Tomato.QDOSERun )
      I_Contact( "T-31.00_DB".Tomato.QDOSERun )
      Contact( "T-05.01_DB".State.Ready_For_Transfer )
      wire#w1
      Coil( "T-21.00_DB".Tomato.ISTART_COND )
   END_RUNG
   RUNG wire#w1
      Contact( "IO_Valve_Blending_DB"."AV-21.12".FB_OPEN )
      Coil( "T-21.00_DB".Tomato.V_OPEN )
   END_RUNG
   RUNG wire#w1
      I_Contact( "IO_Valve_Blending_DB"."AV-21.12".FB_OPEN )
      Coil( "T-21.00_DB".Tomato.V_CLOSE )
   END_RUNG
   RUNG wire#w1
      Contact( "IO Motor MCC Preparation_DB"."P-05.01".FB_ON )
      Coil( "T-21.00_DB".Tomato.P_RUN )
   END_RUNG
   RUNG wire#w1
      I_Contact( "IO Motor MCC Preparation_DB"."P-05.01".FB_ON )
      Coil( "T-21.00_DB".Tomato.P_STOP )
   END_RUNG
   // the same network as SCL:
   "T-21.00_DB".Tomato.ISTART_COND := NOT "T-20.00_DB".Tomato.QDOSERun AND NOT "T-30.00_DB".Tomato.QDOSERun AND NOT "T-31.00_DB".Tomato.QDOSERun AND "T-05.01_DB".State.Ready_For_Transfer;
   "T-21.00_DB".Tomato.V_OPEN := "T-21.00_DB".Tomato.ISTART_COND AND "IO_Valve_Blending_DB"."AV-21.12".FB_OPEN;
   "T-21.00_DB".Tomato.V_CLOSE := "T-21.00_DB".Tomato.ISTART_COND AND NOT "IO_Valve_Blending_DB"."AV-21.12".FB_OPEN;
   "T-21.00_DB".Tomato.P_RUN := "T-21.00_DB".Tomato.ISTART_COND AND "IO Motor MCC Preparation_DB"."P-05.01".FB_ON;
   "T-21.00_DB".Tomato.P_STOP := "T-21.00_DB".Tomato.ISTART_COND AND NOT "IO Motor MCC Preparation_DB"."P-05.01".FB_ON;
END_REGION

REGION Network 18: T-21_Dose_FreshChili_1
   RUNG wire#powerrail
      I_Contact( "T-20.00_DB".ChiliFresh_1.QDOSERun )
      I_Contact( "T-30.00_DB".ChiliFresh_1.QDOSERun )
      I_Contact( "T-31.00_DB".ChiliFresh_1.QDOSERun )
      Contact( "T-06.01_DB".State.Ready_For_Transfer )
      wire#w1
      Coil( "T-21.00_DB".ChiliFresh_1.ISTART_COND )
   END_RUNG
   RUNG wire#w1
      Contact( "IO_Valve_Blending_DB"."AV-21.05".FB_OPEN )
      Coil( "T-21.00_DB".ChiliFresh_1.V_OPEN )
   END_RUNG
   RUNG wire#w1
      I_Contact( "IO_Valve_Blending_DB"."AV-21.05".FB_OPEN )
      Coil( "T-21.00_DB".ChiliFresh_1.V_CLOSE )
   END_RUNG
   RUNG wire#w1
      Contact( "IO Motor MCC Preparation_DB"."P-06.01".FB_ON )
      Coil( "T-21.00_DB".ChiliFresh_1.P_RUN )
   END_RUNG
   RUNG wire#w1
      I_Contact( "IO Motor MCC Preparation_DB"."P-06.01".FB_ON )
      Coil( "T-21.00_DB".ChiliFresh_1.P_STOP )
   END_RUNG
   // the same network as SCL:
   "T-21.00_DB".ChiliFresh_1.ISTART_COND := NOT "T-20.00_DB".ChiliFresh_1.QDOSERun AND NOT "T-30.00_DB".ChiliFresh_1.QDOSERun AND NOT "T-31.00_DB".ChiliFresh_1.QDOSERun AND "T-06.01_DB".State.Ready_For_Transfer;
   "T-21.00_DB".ChiliFresh_1.V_OPEN := "T-21.00_DB".ChiliFresh_1.ISTART_COND AND "IO_Valve_Blending_DB"."AV-21.05".FB_OPEN;
   "T-21.00_DB".ChiliFresh_1.V_CLOSE := "T-21.00_DB".ChiliFresh_1.ISTART_COND AND NOT "IO_Valve_Blending_DB"."AV-21.05".FB_OPEN;
   "T-21.00_DB".ChiliFresh_1.P_RUN := "T-21.00_DB".ChiliFresh_1.ISTART_COND AND "IO Motor MCC Preparation_DB"."P-06.01".FB_ON;
   "T-21.00_DB".ChiliFresh_1.P_STOP := "T-21.00_DB".ChiliFresh_1.ISTART_COND AND NOT "IO Motor MCC Preparation_DB"."P-06.01".FB_ON;
END_REGION

REGION Network 19: T-21_Dose_FreshChili_2
   RUNG wire#powerrail
      I_Contact( "T-20.00_DB".ChiliFresh_2.QDOSERun )
      I_Contact( "T-30.00_DB".ChiliFresh_2.QDOSERun )
      I_Contact( "T-31.00_DB".ChiliFresh_2.QDOSERun )
      Contact( "T-07.01_DB".State.Ready_For_Transfer )
      wire#w1
      Coil( "T-21.00_DB".ChiliFresh_2.ISTART_COND )
   END_RUNG
   RUNG wire#w1
      Contact( "IO_Valve_Blending_DB"."AV-21.06".FB_OPEN )
      Coil( "T-21.00_DB".ChiliFresh_2.V_OPEN )
   END_RUNG
   RUNG wire#w1
      I_Contact( "IO_Valve_Blending_DB"."AV-21.06".FB_OPEN )
      Coil( "T-21.00_DB".ChiliFresh_2.V_CLOSE )
   END_RUNG
   RUNG wire#w1
      Contact( "IO Motor MCC Preparation_DB"."P-07.01".FB_ON )
      Coil( "T-21.00_DB".ChiliFresh_2.P_RUN )
   END_RUNG
   RUNG wire#w1
      I_Contact( "IO Motor MCC Preparation_DB"."P-07.01".FB_ON )
      Coil( "T-21.00_DB".ChiliFresh_2.P_STOP )
   END_RUNG
   // the same network as SCL:
   "T-21.00_DB".ChiliFresh_2.ISTART_COND := NOT "T-20.00_DB".ChiliFresh_2.QDOSERun AND NOT "T-30.00_DB".ChiliFresh_2.QDOSERun AND NOT "T-31.00_DB".ChiliFresh_2.QDOSERun AND "T-07.01_DB".State.Ready_For_Transfer;
   "T-21.00_DB".ChiliFresh_2.V_OPEN := "T-21.00_DB".ChiliFresh_2.ISTART_COND AND "IO_Valve_Blending_DB"."AV-21.06".FB_OPEN;
   "T-21.00_DB".ChiliFresh_2.V_CLOSE := "T-21.00_DB".ChiliFresh_2.ISTART_COND AND NOT "IO_Valve_Blending_DB"."AV-21.06".FB_OPEN;
   "T-21.00_DB".ChiliFresh_2.P_RUN := "T-21.00_DB".ChiliFresh_2.ISTART_COND AND "IO Motor MCC Preparation_DB"."P-07.01".FB_ON;
   "T-21.00_DB".ChiliFresh_2.P_STOP := "T-21.00_DB".ChiliFresh_2.ISTART_COND AND NOT "IO Motor MCC Preparation_DB"."P-07.01".FB_ON;
END_REGION

REGION Network 20: T-21_Dose_FreshChili_3
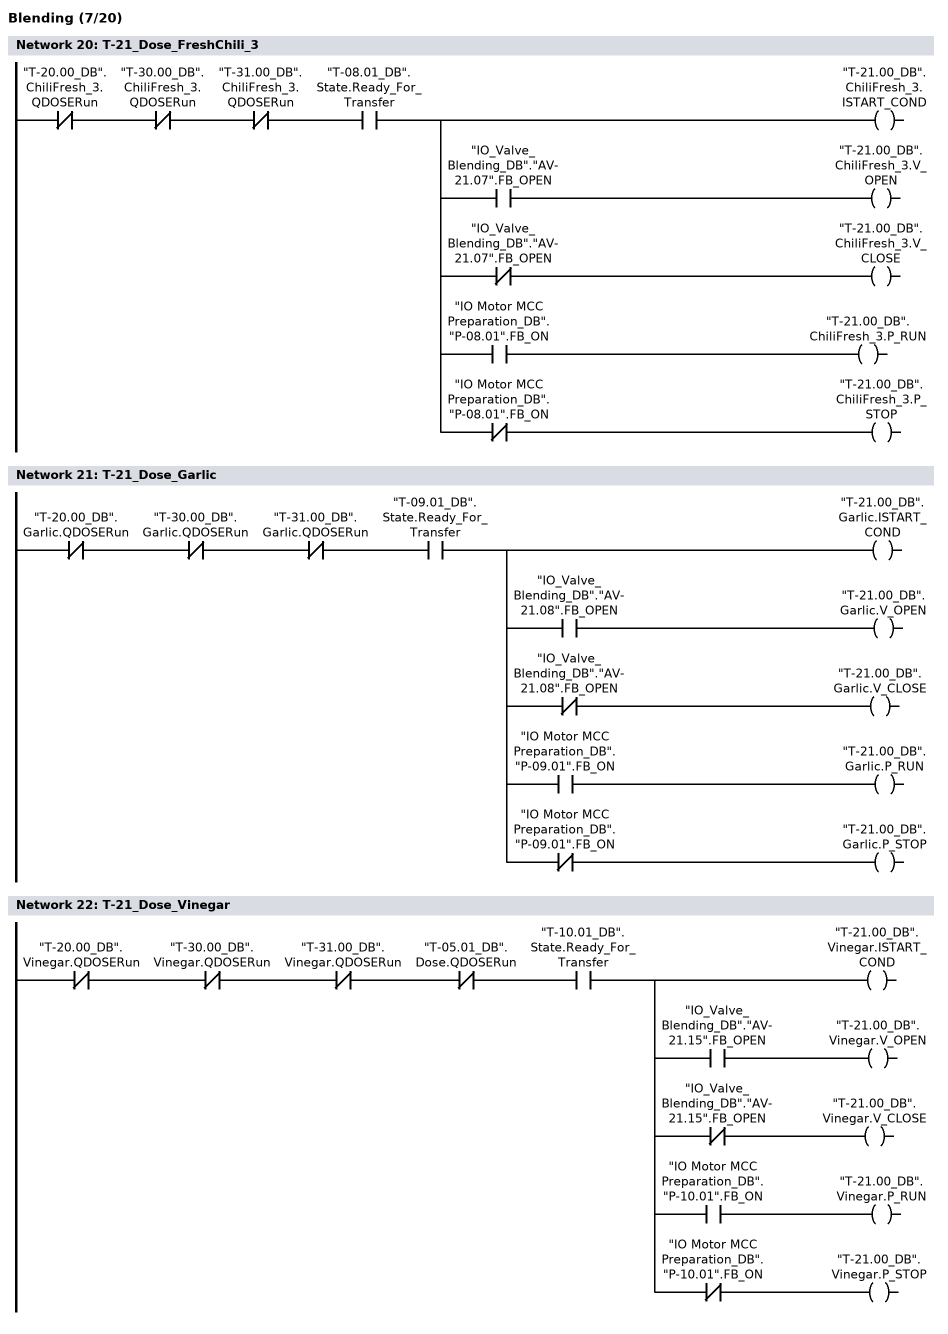
   RUNG wire#powerrail
      I_Contact( "T-20.00_DB".ChiliFresh_3.QDOSERun )
      I_Contact( "T-30.00_DB".ChiliFresh_3.QDOSERun )
      I_Contact( "T-31.00_DB".ChiliFresh_3.QDOSERun )
      Contact( "T-08.01_DB".State.Ready_For_Transfer )
      wire#w1
      Coil( "T-21.00_DB".ChiliFresh_3.ISTART_COND )
   END_RUNG
   RUNG wire#w1
      Contact( "IO_Valve_Blending_DB"."AV-21.07".FB_OPEN )
      Coil( "T-21.00_DB".ChiliFresh_3.V_OPEN )
   END_RUNG
   RUNG wire#w1
      I_Contact( "IO_Valve_Blending_DB"."AV-21.07".FB_OPEN )
      Coil( "T-21.00_DB".ChiliFresh_3.V_CLOSE )
   END_RUNG
   RUNG wire#w1
      Contact( "IO Motor MCC Preparation_DB"."P-08.01".FB_ON )
      Coil( "T-21.00_DB".ChiliFresh_3.P_RUN )
   END_RUNG
   RUNG wire#w1
      I_Contact( "IO Motor MCC Preparation_DB"."P-08.01".FB_ON )
      Coil( "T-21.00_DB".ChiliFresh_3.P_STOP )
   END_RUNG
   // the same network as SCL:
   "T-21.00_DB".ChiliFresh_3.ISTART_COND := NOT "T-20.00_DB".ChiliFresh_3.QDOSERun AND NOT "T-30.00_DB".ChiliFresh_3.QDOSERun AND NOT "T-31.00_DB".ChiliFresh_3.QDOSERun AND "T-08.01_DB".State.Ready_For_Transfer;
   "T-21.00_DB".ChiliFresh_3.V_OPEN := "T-21.00_DB".ChiliFresh_3.ISTART_COND AND "IO_Valve_Blending_DB"."AV-21.07".FB_OPEN;
   "T-21.00_DB".ChiliFresh_3.V_CLOSE := "T-21.00_DB".ChiliFresh_3.ISTART_COND AND NOT "IO_Valve_Blending_DB"."AV-21.07".FB_OPEN;
   "T-21.00_DB".ChiliFresh_3.P_RUN := "T-21.00_DB".ChiliFresh_3.ISTART_COND AND "IO Motor MCC Preparation_DB"."P-08.01".FB_ON;
   "T-21.00_DB".ChiliFresh_3.P_STOP := "T-21.00_DB".ChiliFresh_3.ISTART_COND AND NOT "IO Motor MCC Preparation_DB"."P-08.01".FB_ON;
END_REGION

REGION Network 21: T-21_Dose_Garlic
   RUNG wire#powerrail
      I_Contact( "T-20.00_DB".Garlic.QDOSERun )
      I_Contact( "T-30.00_DB".Garlic.QDOSERun )
      I_Contact( "T-31.00_DB".Garlic.QDOSERun )
      Contact( "T-09.01_DB".State.Ready_For_Transfer )
      wire#w1
      Coil( "T-21.00_DB".Garlic.ISTART_COND )
   END_RUNG
   RUNG wire#w1
      Contact( "IO_Valve_Blending_DB"."AV-21.08".FB_OPEN )
      Coil( "T-21.00_DB".Garlic.V_OPEN )
   END_RUNG
   RUNG wire#w1
      I_Contact( "IO_Valve_Blending_DB"."AV-21.08".FB_OPEN )
      Coil( "T-21.00_DB".Garlic.V_CLOSE )
   END_RUNG
   RUNG wire#w1
      Contact( "IO Motor MCC Preparation_DB"."P-09.01".FB_ON )
      Coil( "T-21.00_DB".Garlic.P_RUN )
   END_RUNG
   RUNG wire#w1
      I_Contact( "IO Motor MCC Preparation_DB"."P-09.01".FB_ON )
      Coil( "T-21.00_DB".Garlic.P_STOP )
   END_RUNG
   // the same network as SCL:
   "T-21.00_DB".Garlic.ISTART_COND := NOT "T-20.00_DB".Garlic.QDOSERun AND NOT "T-30.00_DB".Garlic.QDOSERun AND NOT "T-31.00_DB".Garlic.QDOSERun AND "T-09.01_DB".State.Ready_For_Transfer;
   "T-21.00_DB".Garlic.V_OPEN := "T-21.00_DB".Garlic.ISTART_COND AND "IO_Valve_Blending_DB"."AV-21.08".FB_OPEN;
   "T-21.00_DB".Garlic.V_CLOSE := "T-21.00_DB".Garlic.ISTART_COND AND NOT "IO_Valve_Blending_DB"."AV-21.08".FB_OPEN;
   "T-21.00_DB".Garlic.P_RUN := "T-21.00_DB".Garlic.ISTART_COND AND "IO Motor MCC Preparation_DB"."P-09.01".FB_ON;
   "T-21.00_DB".Garlic.P_STOP := "T-21.00_DB".Garlic.ISTART_COND AND NOT "IO Motor MCC Preparation_DB"."P-09.01".FB_ON;
END_REGION

REGION Network 22: T-21_Dose_Vinegar
   RUNG wire#powerrail
      I_Contact( "T-20.00_DB".Vinegar.QDOSERun )
      I_Contact( "T-30.00_DB".Vinegar.QDOSERun )
      I_Contact( "T-31.00_DB".Vinegar.QDOSERun )
      I_Contact( "T-05.01_DB".Dose.QDOSERun )
      Contact( "T-10.01_DB".State.Ready_For_Transfer )
      wire#w1
      Coil( "T-21.00_DB".Vinegar.ISTART_COND )
   END_RUNG
   RUNG wire#w1
      Contact( "IO_Valve_Blending_DB"."AV-21.15".FB_OPEN )
      Coil( "T-21.00_DB".Vinegar.V_OPEN )
   END_RUNG
   RUNG wire#w1
      I_Contact( "IO_Valve_Blending_DB"."AV-21.15".FB_OPEN )
      Coil( "T-21.00_DB".Vinegar.V_CLOSE )
   END_RUNG
   RUNG wire#w1
      Contact( "IO Motor MCC Preparation_DB"."P-10.01".FB_ON )
      Coil( "T-21.00_DB".Vinegar.P_RUN )
   END_RUNG
   RUNG wire#w1
      I_Contact( "IO Motor MCC Preparation_DB"."P-10.01".FB_ON )
      Coil( "T-21.00_DB".Vinegar.P_STOP )
   END_RUNG
   // the same network as SCL:
   "T-21.00_DB".Vinegar.ISTART_COND := NOT "T-20.00_DB".Vinegar.QDOSERun AND NOT "T-30.00_DB".Vinegar.QDOSERun AND NOT "T-31.00_DB".Vinegar.QDOSERun AND NOT "T-05.01_DB".Dose.QDOSERun AND "T-10.01_DB".State.Ready_For_Transfer;
   "T-21.00_DB".Vinegar.V_OPEN := "T-21.00_DB".Vinegar.ISTART_COND AND "IO_Valve_Blending_DB"."AV-21.15".FB_OPEN;
   "T-21.00_DB".Vinegar.V_CLOSE := "T-21.00_DB".Vinegar.ISTART_COND AND NOT "IO_Valve_Blending_DB"."AV-21.15".FB_OPEN;
   "T-21.00_DB".Vinegar.P_RUN := "T-21.00_DB".Vinegar.ISTART_COND AND "IO Motor MCC Preparation_DB"."P-10.01".FB_ON;
   "T-21.00_DB".Vinegar.P_STOP := "T-21.00_DB".Vinegar.ISTART_COND AND NOT "IO Motor MCC Preparation_DB"."P-10.01".FB_ON;
END_REGION

REGION Network 23: T-21.00
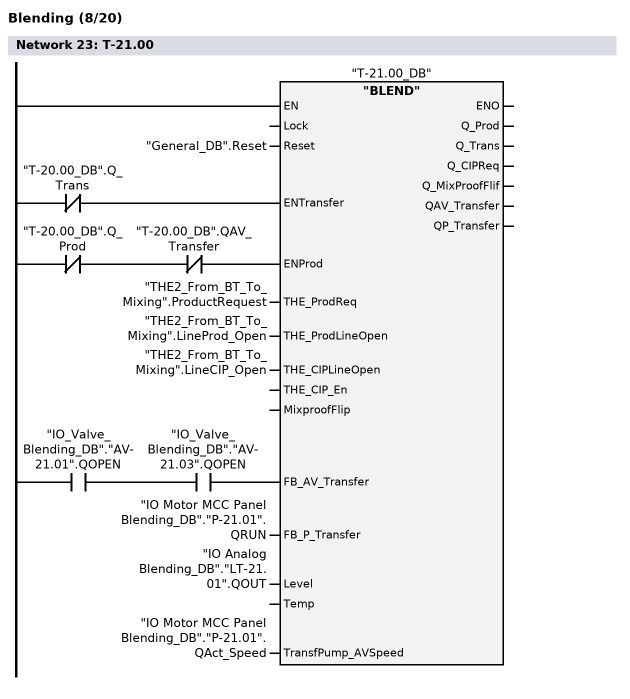
   RUNG wire#powerrail
      "T-21.00_DB"(ENTransfer := wire#w1, ENProd := wire#w2, FB_AV_Transfer := wire#w3, Lock :=, Reset := "General_DB".Reset, THE_ProdReq := "THE2_From_BT_To_Mixing".ProductRequest, THE_ProdLineOpen := "THE2_From_BT_To_Mixing".LineProd_Open, THE_CIPLineOpen := "THE2_From_BT_To_Mixing".LineCIP_Open, THE_CIP_En :=, MixproofFlip :=, FB_P_Transfer := "IO Motor MCC Panel Blending_DB"."P-21.01".QRUN, Level := "IO Analog Blending_DB"."LT-21.01".QOUT, Temp :=, TransfPump_AVSpeed := "IO Motor MCC Panel Blending_DB"."P-21.01".QAct_Speed, Q_Prod =>, Q_Trans =>, Q_CIPReq =>, Q_MixProofFlif =>, QAV_Transfer =>, QP_Transfer =>)
   END_RUNG
   RUNG wire#powerrail
      I_Contact( "T-20.00_DB".Q_Trans )
   END_RUNG wire#w1
   RUNG wire#powerrail
      I_Contact( "T-20.00_DB".Q_Prod )
      I_Contact( "T-20.00_DB".QAV_Transfer )
   END_RUNG wire#w2
   RUNG wire#powerrail
      Contact( "IO_Valve_Blending_DB"."AV-21.01".QOPEN )
      Contact( "IO_Valve_Blending_DB"."AV-21.03".QOPEN )
   END_RUNG wire#w3
   // the same network as SCL:
   "T-21.00_DB"(Reset := "General_DB".Reset,   // "BLEND"
                ENTransfer := NOT "T-20.00_DB".Q_Trans,
                ENProd := NOT "T-20.00_DB".Q_Prod AND NOT "T-20.00_DB".QAV_Transfer,
                THE_ProdReq := "THE2_From_BT_To_Mixing".ProductRequest,
                THE_ProdLineOpen := "THE2_From_BT_To_Mixing".LineProd_Open,
                THE_CIPLineOpen := "THE2_From_BT_To_Mixing".LineCIP_Open,
                FB_AV_Transfer := "IO_Valve_Blending_DB"."AV-21.01".QOPEN AND "IO_Valve_Blending_DB"."AV-21.03".QOPEN,
                FB_P_Transfer := "IO Motor MCC Panel Blending_DB"."P-21.01".QRUN,
                Level := "IO Analog Blending_DB"."LT-21.01".QOUT,
                TransfPump_AVSpeed := "IO Motor MCC Panel Blending_DB"."P-21.01".QAct_Speed);
END_REGION

REGION Network 24: Comm to Buffer Tank THE 2
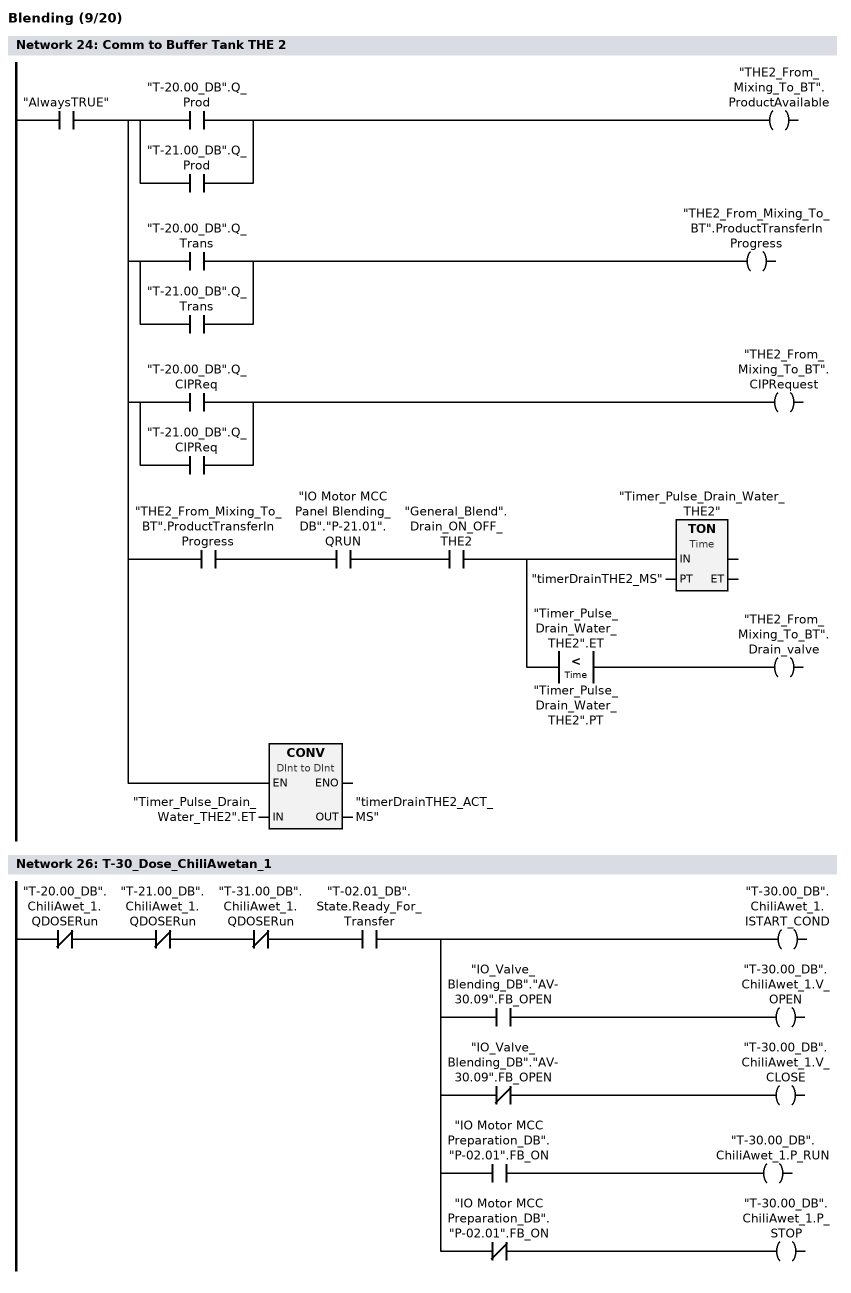
   RUNG wire#powerrail
      Contact( "AlwaysTRUE" )
      wire#w1
      Contact( "T-20.00_DB".Q_Prod )
      wire#w2
      Coil( "THE2_From_Mixing_To_BT".ProductAvailable )
   END_RUNG
   RUNG wire#w1
      Contact( "T-21.00_DB".Q_Prod )
   END_RUNG wire#w2
   RUNG wire#w1
      Contact( "T-20.00_DB".Q_Trans )
      wire#w3
      Coil( "THE2_From_Mixing_To_BT".ProductTransferInProgress )
   END_RUNG
   RUNG wire#w1
      Contact( "T-21.00_DB".Q_Trans )
   END_RUNG wire#w3
   RUNG wire#w1
      Contact( "T-20.00_DB".Q_CIPReq )
      wire#w4
      Coil( "THE2_From_Mixing_To_BT".CIPRequest )
   END_RUNG
   RUNG wire#w1
      Contact( "T-21.00_DB".Q_CIPReq )
   END_RUNG wire#w4
   RUNG wire#w1
      Contact( "THE2_From_Mixing_To_BT".ProductTransferInProgress )
      Contact( "IO Motor MCC Panel Blending_DB"."P-21.01".QRUN )
      Contact( "General_Blend".Drain_ON_OFF_THE2 )
      wire#w5
      { S7_Templates := "time_type := Time" } "Timer_Pulse_Drain_Water_THE2".TON(pt := "timerDrainTHE2_MS", et =>)
   END_RUNG
   RUNG wire#w5
      { S7_Templates := "SrcType := Time" } LT_Contact(in1 := "Timer_Pulse_Drain_Water_THE2".ET, in2 := "Timer_Pulse_Drain_Water_THE2".PT)
      Coil( "THE2_From_Mixing_To_BT".Drain_valve )
   END_RUNG
   RUNG wire#w1
      { S7_Templates := "[SrcType := DInt, DestType := DInt]" } Convert(in := "Timer_Pulse_Drain_Water_THE2".ET, out => "timerDrainTHE2_ACT_MS")
   END_RUNG
   // the same network as SCL:
   "THE2_From_Mixing_To_BT".ProductAvailable := "AlwaysTRUE" AND ("T-20.00_DB".Q_Prod OR "T-21.00_DB".Q_Prod);
   "THE2_From_Mixing_To_BT".ProductTransferInProgress := "AlwaysTRUE" AND ("T-20.00_DB".Q_Trans OR "T-21.00_DB".Q_Trans);
   "THE2_From_Mixing_To_BT".CIPRequest := "AlwaysTRUE" AND ("T-20.00_DB".Q_CIPReq OR "T-21.00_DB".Q_CIPReq);
   #_w1 := "AlwaysTRUE" AND "THE2_From_Mixing_To_BT".ProductTransferInProgress AND "IO Motor MCC Panel Blending_DB"."P-21.01".QRUN AND "General_Blend".Drain_ON_OFF_THE2;
   "Timer_Pulse_Drain_Water_THE2".TON(IN := #_w1, PT := "timerDrainTHE2_MS");
   "THE2_From_Mixing_To_BT".Drain_valve := #_w1 AND ("Timer_Pulse_Drain_Water_THE2".ET < "Timer_Pulse_Drain_Water_THE2".PT);
   IF "AlwaysTRUE" THEN "timerDrainTHE2_ACT_MS" := DINT_TO_DINT("Timer_Pulse_Drain_Water_THE2".ET); END_IF;
END_REGION

REGION Network 26: T-30_Dose_ChiliAwetan_1
   RUNG wire#powerrail
      I_Contact( "T-20.00_DB".ChiliAwet_1.QDOSERun )
      I_Contact( "T-21.00_DB".ChiliAwet_1.QDOSERun )
      I_Contact( "T-31.00_DB".ChiliAwet_1.QDOSERun )
      Contact( "T-02.01_DB".State.Ready_For_Transfer )
      wire#w1
      Coil( "T-30.00_DB".ChiliAwet_1.ISTART_COND )
   END_RUNG
   RUNG wire#w1
      Contact( "IO_Valve_Blending_DB"."AV-30.09".FB_OPEN )
      Coil( "T-30.00_DB".ChiliAwet_1.V_OPEN )
   END_RUNG
   RUNG wire#w1
      I_Contact( "IO_Valve_Blending_DB"."AV-30.09".FB_OPEN )
      Coil( "T-30.00_DB".ChiliAwet_1.V_CLOSE )
   END_RUNG
   RUNG wire#w1
      Contact( "IO Motor MCC Preparation_DB"."P-02.01".FB_ON )
      Coil( "T-30.00_DB".ChiliAwet_1.P_RUN )
   END_RUNG
   RUNG wire#w1
      I_Contact( "IO Motor MCC Preparation_DB"."P-02.01".FB_ON )
      Coil( "T-30.00_DB".ChiliAwet_1.P_STOP )
   END_RUNG
   // the same network as SCL:
   "T-30.00_DB".ChiliAwet_1.ISTART_COND := NOT "T-20.00_DB".ChiliAwet_1.QDOSERun AND NOT "T-21.00_DB".ChiliAwet_1.QDOSERun AND NOT "T-31.00_DB".ChiliAwet_1.QDOSERun AND "T-02.01_DB".State.Ready_For_Transfer;
   "T-30.00_DB".ChiliAwet_1.V_OPEN := "T-30.00_DB".ChiliAwet_1.ISTART_COND AND "IO_Valve_Blending_DB"."AV-30.09".FB_OPEN;
   "T-30.00_DB".ChiliAwet_1.V_CLOSE := "T-30.00_DB".ChiliAwet_1.ISTART_COND AND NOT "IO_Valve_Blending_DB"."AV-30.09".FB_OPEN;
   "T-30.00_DB".ChiliAwet_1.P_RUN := "T-30.00_DB".ChiliAwet_1.ISTART_COND AND "IO Motor MCC Preparation_DB"."P-02.01".FB_ON;
   "T-30.00_DB".ChiliAwet_1.P_STOP := "T-30.00_DB".ChiliAwet_1.ISTART_COND AND NOT "IO Motor MCC Preparation_DB"."P-02.01".FB_ON;
END_REGION

REGION Network 27: T-30_Dose_ChiliAwetan_2
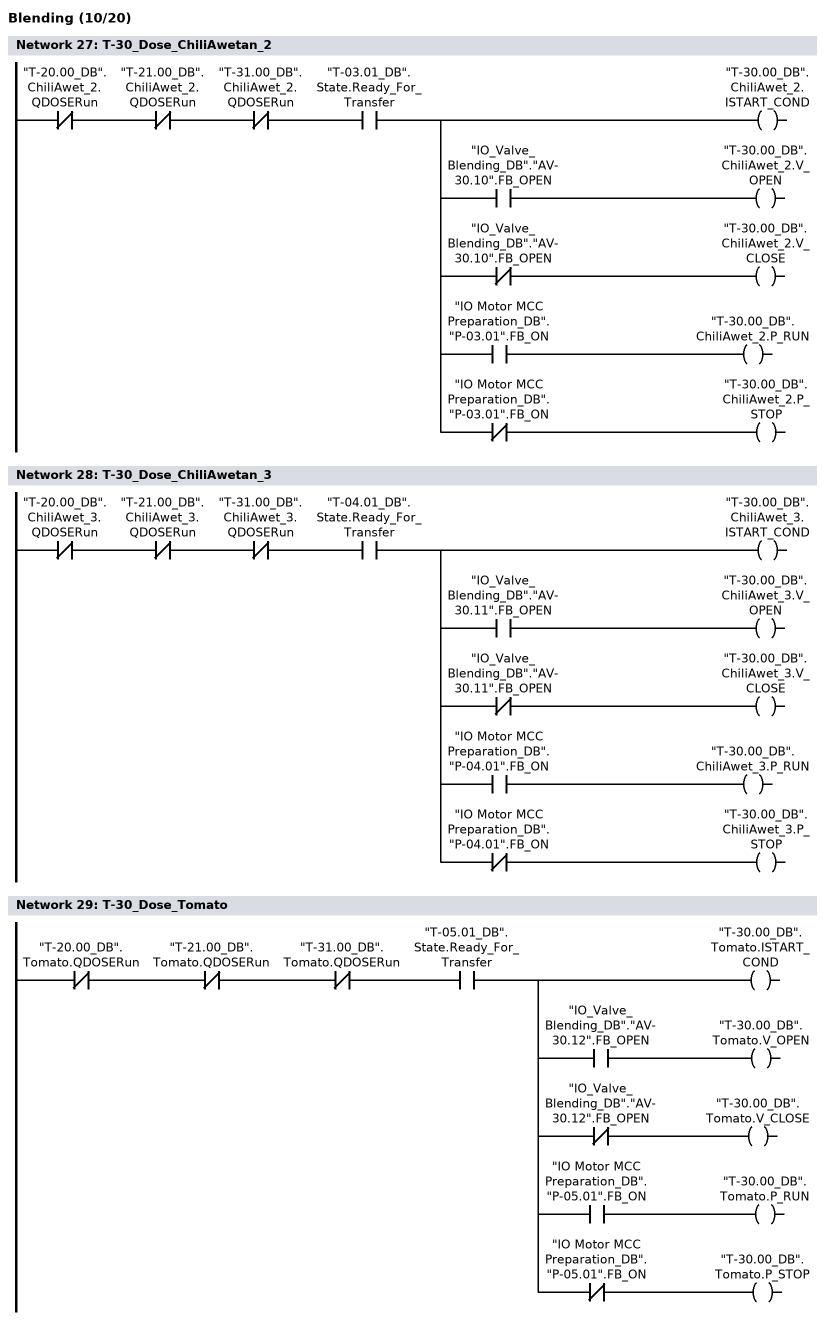
   RUNG wire#powerrail
      I_Contact( "T-20.00_DB".ChiliAwet_2.QDOSERun )
      I_Contact( "T-21.00_DB".ChiliAwet_2.QDOSERun )
      I_Contact( "T-31.00_DB".ChiliAwet_2.QDOSERun )
      Contact( "T-03.01_DB".State.Ready_For_Transfer )
      wire#w1
      Coil( "T-30.00_DB".ChiliAwet_2.ISTART_COND )
   END_RUNG
   RUNG wire#w1
      Contact( "IO_Valve_Blending_DB"."AV-30.10".FB_OPEN )
      Coil( "T-30.00_DB".ChiliAwet_2.V_OPEN )
   END_RUNG
   RUNG wire#w1
      I_Contact( "IO_Valve_Blending_DB"."AV-30.10".FB_OPEN )
      Coil( "T-30.00_DB".ChiliAwet_2.V_CLOSE )
   END_RUNG
   RUNG wire#w1
      Contact( "IO Motor MCC Preparation_DB"."P-03.01".FB_ON )
      Coil( "T-30.00_DB".ChiliAwet_2.P_RUN )
   END_RUNG
   RUNG wire#w1
      I_Contact( "IO Motor MCC Preparation_DB"."P-03.01".FB_ON )
      Coil( "T-30.00_DB".ChiliAwet_2.P_STOP )
   END_RUNG
   // the same network as SCL:
   "T-30.00_DB".ChiliAwet_2.ISTART_COND := NOT "T-20.00_DB".ChiliAwet_2.QDOSERun AND NOT "T-21.00_DB".ChiliAwet_2.QDOSERun AND NOT "T-31.00_DB".ChiliAwet_2.QDOSERun AND "T-03.01_DB".State.Ready_For_Transfer;
   "T-30.00_DB".ChiliAwet_2.V_OPEN := "T-30.00_DB".ChiliAwet_2.ISTART_COND AND "IO_Valve_Blending_DB"."AV-30.10".FB_OPEN;
   "T-30.00_DB".ChiliAwet_2.V_CLOSE := "T-30.00_DB".ChiliAwet_2.ISTART_COND AND NOT "IO_Valve_Blending_DB"."AV-30.10".FB_OPEN;
   "T-30.00_DB".ChiliAwet_2.P_RUN := "T-30.00_DB".ChiliAwet_2.ISTART_COND AND "IO Motor MCC Preparation_DB"."P-03.01".FB_ON;
   "T-30.00_DB".ChiliAwet_2.P_STOP := "T-30.00_DB".ChiliAwet_2.ISTART_COND AND NOT "IO Motor MCC Preparation_DB"."P-03.01".FB_ON;
END_REGION

REGION Network 28: T-30_Dose_ChiliAwetan_3
   RUNG wire#powerrail
      I_Contact( "T-20.00_DB".ChiliAwet_3.QDOSERun )
      I_Contact( "T-21.00_DB".ChiliAwet_3.QDOSERun )
      I_Contact( "T-31.00_DB".ChiliAwet_3.QDOSERun )
      Contact( "T-04.01_DB".State.Ready_For_Transfer )
      wire#w1
      Coil( "T-30.00_DB".ChiliAwet_3.ISTART_COND )
   END_RUNG
   RUNG wire#w1
      Contact( "IO_Valve_Blending_DB"."AV-30.11".FB_OPEN )
      Coil( "T-30.00_DB".ChiliAwet_3.V_OPEN )
   END_RUNG
   RUNG wire#w1
      I_Contact( "IO_Valve_Blending_DB"."AV-30.11".FB_OPEN )
      Coil( "T-30.00_DB".ChiliAwet_3.V_CLOSE )
   END_RUNG
   RUNG wire#w1
      Contact( "IO Motor MCC Preparation_DB"."P-04.01".FB_ON )
      Coil( "T-30.00_DB".ChiliAwet_3.P_RUN )
   END_RUNG
   RUNG wire#w1
      I_Contact( "IO Motor MCC Preparation_DB"."P-04.01".FB_ON )
      Coil( "T-30.00_DB".ChiliAwet_3.P_STOP )
   END_RUNG
   // the same network as SCL:
   "T-30.00_DB".ChiliAwet_3.ISTART_COND := NOT "T-20.00_DB".ChiliAwet_3.QDOSERun AND NOT "T-21.00_DB".ChiliAwet_3.QDOSERun AND NOT "T-31.00_DB".ChiliAwet_3.QDOSERun AND "T-04.01_DB".State.Ready_For_Transfer;
   "T-30.00_DB".ChiliAwet_3.V_OPEN := "T-30.00_DB".ChiliAwet_3.ISTART_COND AND "IO_Valve_Blending_DB"."AV-30.11".FB_OPEN;
   "T-30.00_DB".ChiliAwet_3.V_CLOSE := "T-30.00_DB".ChiliAwet_3.ISTART_COND AND NOT "IO_Valve_Blending_DB"."AV-30.11".FB_OPEN;
   "T-30.00_DB".ChiliAwet_3.P_RUN := "T-30.00_DB".ChiliAwet_3.ISTART_COND AND "IO Motor MCC Preparation_DB"."P-04.01".FB_ON;
   "T-30.00_DB".ChiliAwet_3.P_STOP := "T-30.00_DB".ChiliAwet_3.ISTART_COND AND NOT "IO Motor MCC Preparation_DB"."P-04.01".FB_ON;
END_REGION

REGION Network 29: T-30_Dose_Tomato
   RUNG wire#powerrail
      I_Contact( "T-20.00_DB".Tomato.QDOSERun )
      I_Contact( "T-21.00_DB".Tomato.QDOSERun )
      I_Contact( "T-31.00_DB".Tomato.QDOSERun )
      Contact( "T-05.01_DB".State.Ready_For_Transfer )
      wire#w1
      Coil( "T-30.00_DB".Tomato.ISTART_COND )
   END_RUNG
   RUNG wire#w1
      Contact( "IO_Valve_Blending_DB"."AV-30.12".FB_OPEN )
      Coil( "T-30.00_DB".Tomato.V_OPEN )
   END_RUNG
   RUNG wire#w1
      I_Contact( "IO_Valve_Blending_DB"."AV-30.12".FB_OPEN )
      Coil( "T-30.00_DB".Tomato.V_CLOSE )
   END_RUNG
   RUNG wire#w1
      Contact( "IO Motor MCC Preparation_DB"."P-05.01".FB_ON )
      Coil( "T-30.00_DB".Tomato.P_RUN )
   END_RUNG
   RUNG wire#w1
      I_Contact( "IO Motor MCC Preparation_DB"."P-05.01".FB_ON )
      Coil( "T-30.00_DB".Tomato.P_STOP )
   END_RUNG
   // the same network as SCL:
   "T-30.00_DB".Tomato.ISTART_COND := NOT "T-20.00_DB".Tomato.QDOSERun AND NOT "T-21.00_DB".Tomato.QDOSERun AND NOT "T-31.00_DB".Tomato.QDOSERun AND "T-05.01_DB".State.Ready_For_Transfer;
   "T-30.00_DB".Tomato.V_OPEN := "T-30.00_DB".Tomato.ISTART_COND AND "IO_Valve_Blending_DB"."AV-30.12".FB_OPEN;
   "T-30.00_DB".Tomato.V_CLOSE := "T-30.00_DB".Tomato.ISTART_COND AND NOT "IO_Valve_Blending_DB"."AV-30.12".FB_OPEN;
   "T-30.00_DB".Tomato.P_RUN := "T-30.00_DB".Tomato.ISTART_COND AND "IO Motor MCC Preparation_DB"."P-05.01".FB_ON;
   "T-30.00_DB".Tomato.P_STOP := "T-30.00_DB".Tomato.ISTART_COND AND NOT "IO Motor MCC Preparation_DB"."P-05.01".FB_ON;
END_REGION

REGION Network 30: T-30_Dose_FreshChili_1
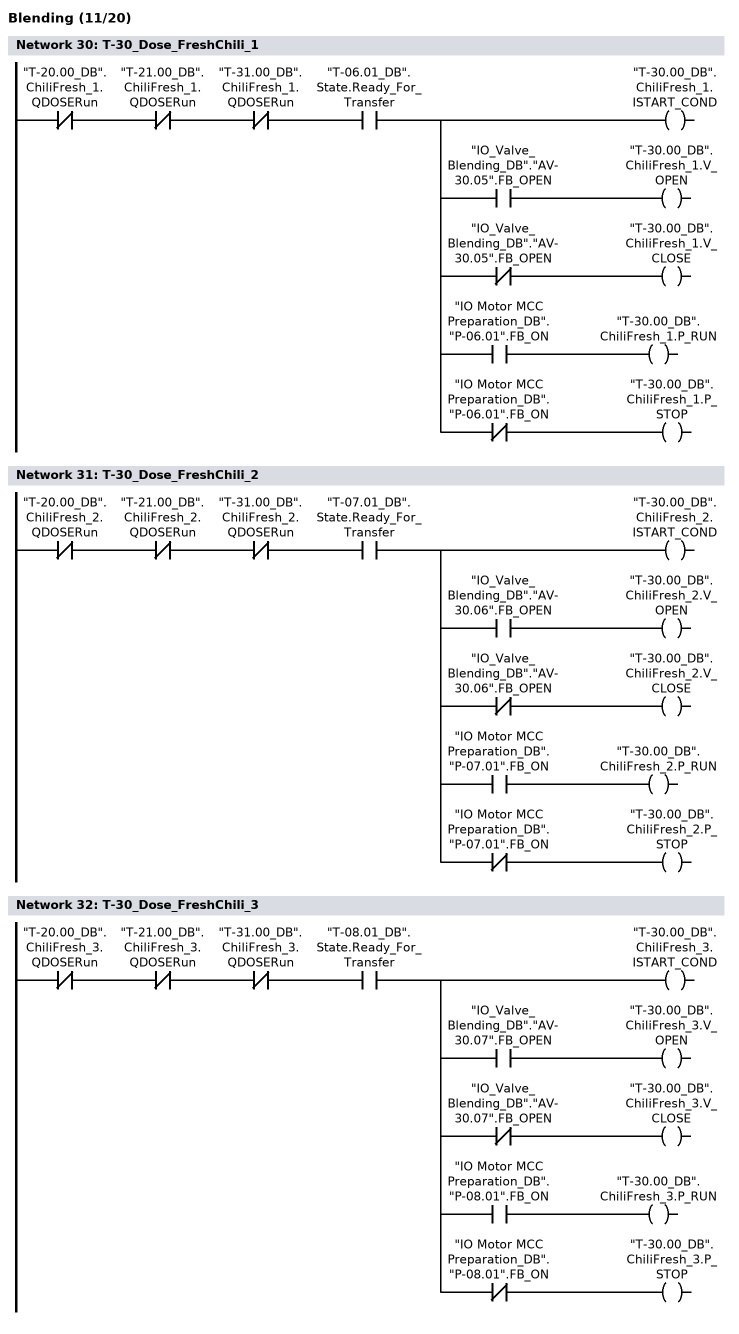
   RUNG wire#powerrail
      I_Contact( "T-20.00_DB".ChiliFresh_1.QDOSERun )
      I_Contact( "T-21.00_DB".ChiliFresh_1.QDOSERun )
      I_Contact( "T-31.00_DB".ChiliFresh_1.QDOSERun )
      Contact( "T-06.01_DB".State.Ready_For_Transfer )
      wire#w1
      Coil( "T-30.00_DB".ChiliFresh_1.ISTART_COND )
   END_RUNG
   RUNG wire#w1
      Contact( "IO_Valve_Blending_DB"."AV-30.05".FB_OPEN )
      Coil( "T-30.00_DB".ChiliFresh_1.V_OPEN )
   END_RUNG
   RUNG wire#w1
      I_Contact( "IO_Valve_Blending_DB"."AV-30.05".FB_OPEN )
      Coil( "T-30.00_DB".ChiliFresh_1.V_CLOSE )
   END_RUNG
   RUNG wire#w1
      Contact( "IO Motor MCC Preparation_DB"."P-06.01".FB_ON )
      Coil( "T-30.00_DB".ChiliFresh_1.P_RUN )
   END_RUNG
   RUNG wire#w1
      I_Contact( "IO Motor MCC Preparation_DB"."P-06.01".FB_ON )
      Coil( "T-30.00_DB".ChiliFresh_1.P_STOP )
   END_RUNG
   // the same network as SCL:
   "T-30.00_DB".ChiliFresh_1.ISTART_COND := NOT "T-20.00_DB".ChiliFresh_1.QDOSERun AND NOT "T-21.00_DB".ChiliFresh_1.QDOSERun AND NOT "T-31.00_DB".ChiliFresh_1.QDOSERun AND "T-06.01_DB".State.Ready_For_Transfer;
   "T-30.00_DB".ChiliFresh_1.V_OPEN := "T-30.00_DB".ChiliFresh_1.ISTART_COND AND "IO_Valve_Blending_DB"."AV-30.05".FB_OPEN;
   "T-30.00_DB".ChiliFresh_1.V_CLOSE := "T-30.00_DB".ChiliFresh_1.ISTART_COND AND NOT "IO_Valve_Blending_DB"."AV-30.05".FB_OPEN;
   "T-30.00_DB".ChiliFresh_1.P_RUN := "T-30.00_DB".ChiliFresh_1.ISTART_COND AND "IO Motor MCC Preparation_DB"."P-06.01".FB_ON;
   "T-30.00_DB".ChiliFresh_1.P_STOP := "T-30.00_DB".ChiliFresh_1.ISTART_COND AND NOT "IO Motor MCC Preparation_DB"."P-06.01".FB_ON;
END_REGION

REGION Network 31: T-30_Dose_FreshChili_2
   RUNG wire#powerrail
      I_Contact( "T-20.00_DB".ChiliFresh_2.QDOSERun )
      I_Contact( "T-21.00_DB".ChiliFresh_2.QDOSERun )
      I_Contact( "T-31.00_DB".ChiliFresh_2.QDOSERun )
      Contact( "T-07.01_DB".State.Ready_For_Transfer )
      wire#w1
      Coil( "T-30.00_DB".ChiliFresh_2.ISTART_COND )
   END_RUNG
   RUNG wire#w1
      Contact( "IO_Valve_Blending_DB"."AV-30.06".FB_OPEN )
      Coil( "T-30.00_DB".ChiliFresh_2.V_OPEN )
   END_RUNG
   RUNG wire#w1
      I_Contact( "IO_Valve_Blending_DB"."AV-30.06".FB_OPEN )
      Coil( "T-30.00_DB".ChiliFresh_2.V_CLOSE )
   END_RUNG
   RUNG wire#w1
      Contact( "IO Motor MCC Preparation_DB"."P-07.01".FB_ON )
      Coil( "T-30.00_DB".ChiliFresh_2.P_RUN )
   END_RUNG
   RUNG wire#w1
      I_Contact( "IO Motor MCC Preparation_DB"."P-07.01".FB_ON )
      Coil( "T-30.00_DB".ChiliFresh_2.P_STOP )
   END_RUNG
   // the same network as SCL:
   "T-30.00_DB".ChiliFresh_2.ISTART_COND := NOT "T-20.00_DB".ChiliFresh_2.QDOSERun AND NOT "T-21.00_DB".ChiliFresh_2.QDOSERun AND NOT "T-31.00_DB".ChiliFresh_2.QDOSERun AND "T-07.01_DB".State.Ready_For_Transfer;
   "T-30.00_DB".ChiliFresh_2.V_OPEN := "T-30.00_DB".ChiliFresh_2.ISTART_COND AND "IO_Valve_Blending_DB"."AV-30.06".FB_OPEN;
   "T-30.00_DB".ChiliFresh_2.V_CLOSE := "T-30.00_DB".ChiliFresh_2.ISTART_COND AND NOT "IO_Valve_Blending_DB"."AV-30.06".FB_OPEN;
   "T-30.00_DB".ChiliFresh_2.P_RUN := "T-30.00_DB".ChiliFresh_2.ISTART_COND AND "IO Motor MCC Preparation_DB"."P-07.01".FB_ON;
   "T-30.00_DB".ChiliFresh_2.P_STOP := "T-30.00_DB".ChiliFresh_2.ISTART_COND AND NOT "IO Motor MCC Preparation_DB"."P-07.01".FB_ON;
END_REGION

REGION Network 32: T-30_Dose_FreshChili_3
   RUNG wire#powerrail
      I_Contact( "T-20.00_DB".ChiliFresh_3.QDOSERun )
      I_Contact( "T-21.00_DB".ChiliFresh_3.QDOSERun )
      I_Contact( "T-31.00_DB".ChiliFresh_3.QDOSERun )
      Contact( "T-08.01_DB".State.Ready_For_Transfer )
      wire#w1
      Coil( "T-30.00_DB".ChiliFresh_3.ISTART_COND )
   END_RUNG
   RUNG wire#w1
      Contact( "IO_Valve_Blending_DB"."AV-30.07".FB_OPEN )
      Coil( "T-30.00_DB".ChiliFresh_3.V_OPEN )
   END_RUNG
   RUNG wire#w1
      I_Contact( "IO_Valve_Blending_DB"."AV-30.07".FB_OPEN )
      Coil( "T-30.00_DB".ChiliFresh_3.V_CLOSE )
   END_RUNG
   RUNG wire#w1
      Contact( "IO Motor MCC Preparation_DB"."P-08.01".FB_ON )
      Coil( "T-30.00_DB".ChiliFresh_3.P_RUN )
   END_RUNG
   RUNG wire#w1
      I_Contact( "IO Motor MCC Preparation_DB"."P-08.01".FB_ON )
      Coil( "T-30.00_DB".ChiliFresh_3.P_STOP )
   END_RUNG
   // the same network as SCL:
   "T-30.00_DB".ChiliFresh_3.ISTART_COND := NOT "T-20.00_DB".ChiliFresh_3.QDOSERun AND NOT "T-21.00_DB".ChiliFresh_3.QDOSERun AND NOT "T-31.00_DB".ChiliFresh_3.QDOSERun AND "T-08.01_DB".State.Ready_For_Transfer;
   "T-30.00_DB".ChiliFresh_3.V_OPEN := "T-30.00_DB".ChiliFresh_3.ISTART_COND AND "IO_Valve_Blending_DB"."AV-30.07".FB_OPEN;
   "T-30.00_DB".ChiliFresh_3.V_CLOSE := "T-30.00_DB".ChiliFresh_3.ISTART_COND AND NOT "IO_Valve_Blending_DB"."AV-30.07".FB_OPEN;
   "T-30.00_DB".ChiliFresh_3.P_RUN := "T-30.00_DB".ChiliFresh_3.ISTART_COND AND "IO Motor MCC Preparation_DB"."P-08.01".FB_ON;
   "T-30.00_DB".ChiliFresh_3.P_STOP := "T-30.00_DB".ChiliFresh_3.ISTART_COND AND NOT "IO Motor MCC Preparation_DB"."P-08.01".FB_ON;
END_REGION

REGION Network 33: T-30_Dose_Garlic
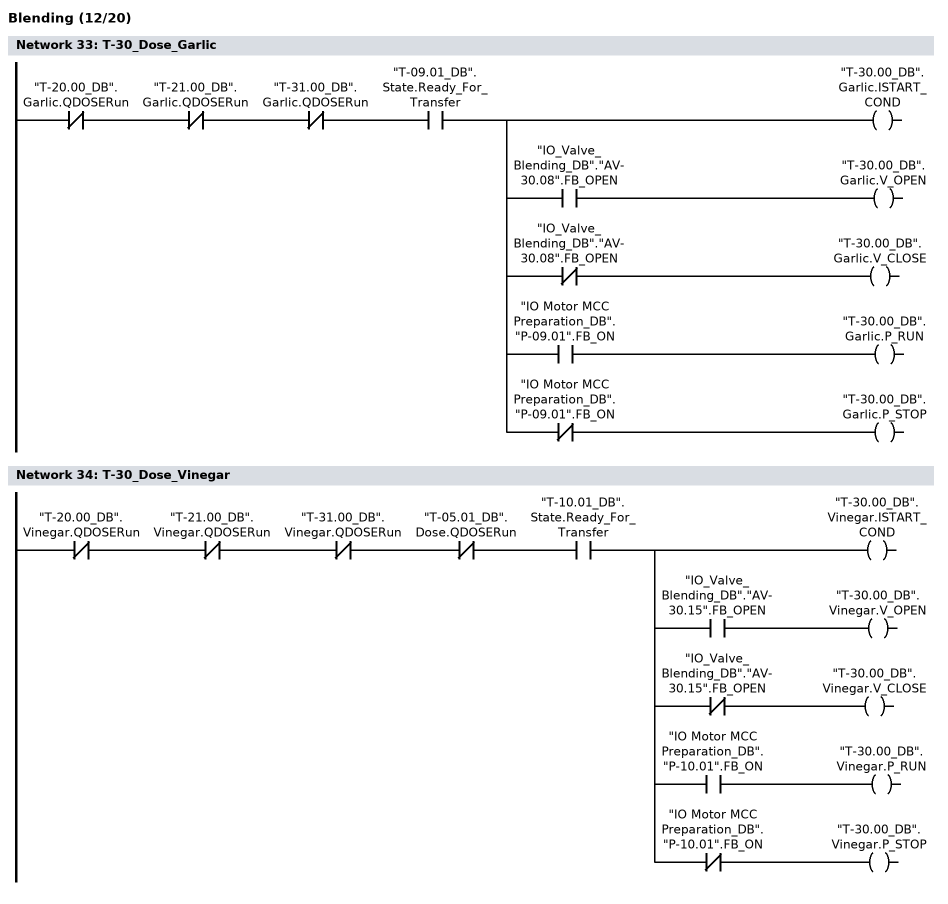
   RUNG wire#powerrail
      I_Contact( "T-20.00_DB".Garlic.QDOSERun )
      I_Contact( "T-21.00_DB".Garlic.QDOSERun )
      I_Contact( "T-31.00_DB".Garlic.QDOSERun )
      Contact( "T-09.01_DB".State.Ready_For_Transfer )
      wire#w1
      Coil( "T-30.00_DB".Garlic.ISTART_COND )
   END_RUNG
   RUNG wire#w1
      Contact( "IO_Valve_Blending_DB"."AV-30.08".FB_OPEN )
      Coil( "T-30.00_DB".Garlic.V_OPEN )
   END_RUNG
   RUNG wire#w1
      I_Contact( "IO_Valve_Blending_DB"."AV-30.08".FB_OPEN )
      Coil( "T-30.00_DB".Garlic.V_CLOSE )
   END_RUNG
   RUNG wire#w1
      Contact( "IO Motor MCC Preparation_DB"."P-09.01".FB_ON )
      Coil( "T-30.00_DB".Garlic.P_RUN )
   END_RUNG
   RUNG wire#w1
      I_Contact( "IO Motor MCC Preparation_DB"."P-09.01".FB_ON )
      Coil( "T-30.00_DB".Garlic.P_STOP )
   END_RUNG
   // the same network as SCL:
   "T-30.00_DB".Garlic.ISTART_COND := NOT "T-20.00_DB".Garlic.QDOSERun AND NOT "T-21.00_DB".Garlic.QDOSERun AND NOT "T-31.00_DB".Garlic.QDOSERun AND "T-09.01_DB".State.Ready_For_Transfer;
   "T-30.00_DB".Garlic.V_OPEN := "T-30.00_DB".Garlic.ISTART_COND AND "IO_Valve_Blending_DB"."AV-30.08".FB_OPEN;
   "T-30.00_DB".Garlic.V_CLOSE := "T-30.00_DB".Garlic.ISTART_COND AND NOT "IO_Valve_Blending_DB"."AV-30.08".FB_OPEN;
   "T-30.00_DB".Garlic.P_RUN := "T-30.00_DB".Garlic.ISTART_COND AND "IO Motor MCC Preparation_DB"."P-09.01".FB_ON;
   "T-30.00_DB".Garlic.P_STOP := "T-30.00_DB".Garlic.ISTART_COND AND NOT "IO Motor MCC Preparation_DB"."P-09.01".FB_ON;
END_REGION

REGION Network 34: T-30_Dose_Vinegar
   RUNG wire#powerrail
      I_Contact( "T-20.00_DB".Vinegar.QDOSERun )
      I_Contact( "T-21.00_DB".Vinegar.QDOSERun )
      I_Contact( "T-31.00_DB".Vinegar.QDOSERun )
      I_Contact( "T-05.01_DB".Dose.QDOSERun )
      Contact( "T-10.01_DB".State.Ready_For_Transfer )
      wire#w1
      Coil( "T-30.00_DB".Vinegar.ISTART_COND )
   END_RUNG
   RUNG wire#w1
      Contact( "IO_Valve_Blending_DB"."AV-30.15".FB_OPEN )
      Coil( "T-30.00_DB".Vinegar.V_OPEN )
   END_RUNG
   RUNG wire#w1
      I_Contact( "IO_Valve_Blending_DB"."AV-30.15".FB_OPEN )
      Coil( "T-30.00_DB".Vinegar.V_CLOSE )
   END_RUNG
   RUNG wire#w1
      Contact( "IO Motor MCC Preparation_DB"."P-10.01".FB_ON )
      Coil( "T-30.00_DB".Vinegar.P_RUN )
   END_RUNG
   RUNG wire#w1
      I_Contact( "IO Motor MCC Preparation_DB"."P-10.01".FB_ON )
      Coil( "T-30.00_DB".Vinegar.P_STOP )
   END_RUNG
   // the same network as SCL:
   "T-30.00_DB".Vinegar.ISTART_COND := NOT "T-20.00_DB".Vinegar.QDOSERun AND NOT "T-21.00_DB".Vinegar.QDOSERun AND NOT "T-31.00_DB".Vinegar.QDOSERun AND NOT "T-05.01_DB".Dose.QDOSERun AND "T-10.01_DB".State.Ready_For_Transfer;
   "T-30.00_DB".Vinegar.V_OPEN := "T-30.00_DB".Vinegar.ISTART_COND AND "IO_Valve_Blending_DB"."AV-30.15".FB_OPEN;
   "T-30.00_DB".Vinegar.V_CLOSE := "T-30.00_DB".Vinegar.ISTART_COND AND NOT "IO_Valve_Blending_DB"."AV-30.15".FB_OPEN;
   "T-30.00_DB".Vinegar.P_RUN := "T-30.00_DB".Vinegar.ISTART_COND AND "IO Motor MCC Preparation_DB"."P-10.01".FB_ON;
   "T-30.00_DB".Vinegar.P_STOP := "T-30.00_DB".Vinegar.ISTART_COND AND NOT "IO Motor MCC Preparation_DB"."P-10.01".FB_ON;
END_REGION

REGION Network 35: T-30.00
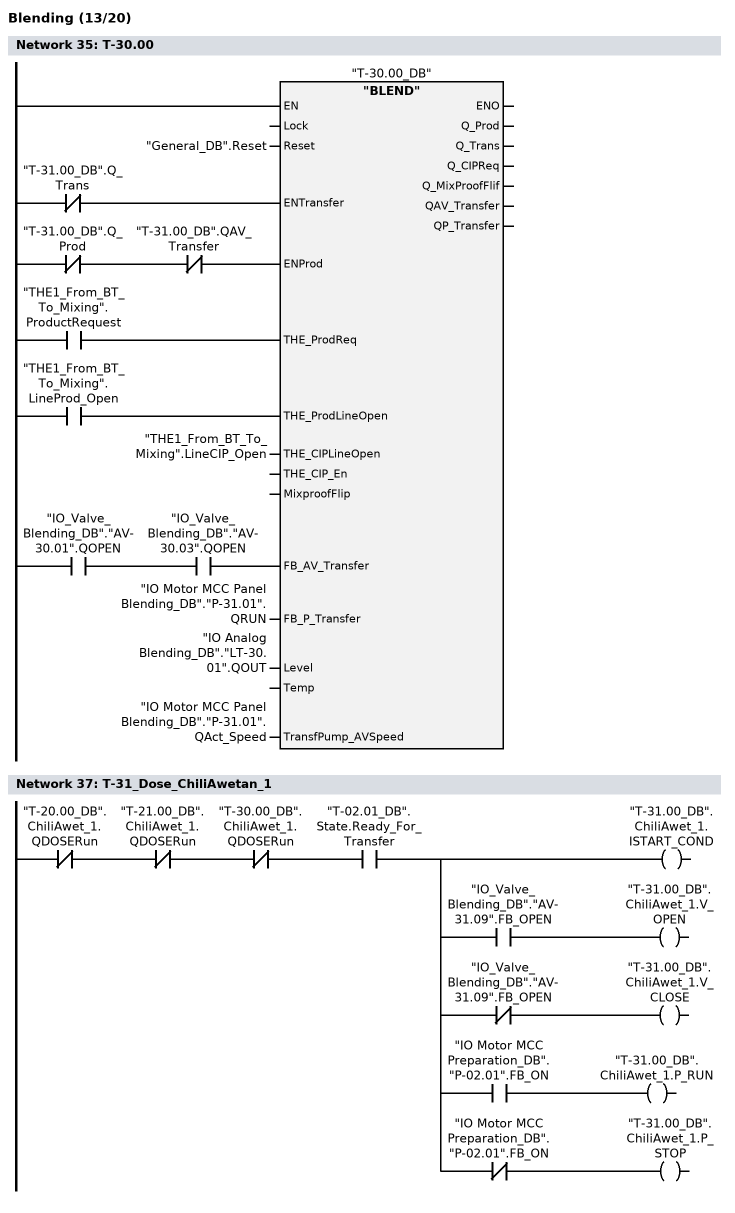
   RUNG wire#powerrail
      "T-30.00_DB"(ENTransfer := wire#w1, ENProd := wire#w2, THE_ProdReq := wire#w3, THE_ProdLineOpen := wire#w4, FB_AV_Transfer := wire#w5, Lock :=, Reset := "General_DB".Reset, THE_CIPLineOpen := "THE1_From_BT_To_Mixing".LineCIP_Open, THE_CIP_En :=, MixproofFlip :=, FB_P_Transfer := "IO Motor MCC Panel Blending_DB"."P-31.01".QRUN, Level := "IO Analog Blending_DB"."LT-30.01".QOUT, Temp :=, TransfPump_AVSpeed := "IO Motor MCC Panel Blending_DB"."P-31.01".QAct_Speed, Q_Prod =>, Q_Trans =>, Q_CIPReq =>, Q_MixProofFlif =>, QAV_Transfer =>, QP_Transfer =>)
   END_RUNG
   RUNG wire#powerrail
      I_Contact( "T-31.00_DB".Q_Trans )
   END_RUNG wire#w1
   RUNG wire#powerrail
      I_Contact( "T-31.00_DB".Q_Prod )
      I_Contact( "T-31.00_DB".QAV_Transfer )
   END_RUNG wire#w2
   RUNG wire#powerrail
      Contact( "THE1_From_BT_To_Mixing".ProductRequest )
   END_RUNG wire#w3
   RUNG wire#powerrail
      Contact( "THE1_From_BT_To_Mixing".LineProd_Open )
   END_RUNG wire#w4
   RUNG wire#powerrail
      Contact( "IO_Valve_Blending_DB"."AV-30.01".QOPEN )
      Contact( "IO_Valve_Blending_DB"."AV-30.03".QOPEN )
   END_RUNG wire#w5
   // the same network as SCL:
   "T-30.00_DB"(Reset := "General_DB".Reset,   // "BLEND"
                ENTransfer := NOT "T-31.00_DB".Q_Trans,
                ENProd := NOT "T-31.00_DB".Q_Prod AND NOT "T-31.00_DB".QAV_Transfer,
                THE_ProdReq := "THE1_From_BT_To_Mixing".ProductRequest,
                THE_ProdLineOpen := "THE1_From_BT_To_Mixing".LineProd_Open,
                THE_CIPLineOpen := "THE1_From_BT_To_Mixing".LineCIP_Open,
                FB_AV_Transfer := "IO_Valve_Blending_DB"."AV-30.01".QOPEN AND "IO_Valve_Blending_DB"."AV-30.03".QOPEN,
                FB_P_Transfer := "IO Motor MCC Panel Blending_DB"."P-31.01".QRUN,
                Level := "IO Analog Blending_DB"."LT-30.01".QOUT,
                TransfPump_AVSpeed := "IO Motor MCC Panel Blending_DB"."P-31.01".QAct_Speed);
END_REGION

REGION Network 37: T-31_Dose_ChiliAwetan_1
   RUNG wire#powerrail
      I_Contact( "T-20.00_DB".ChiliAwet_1.QDOSERun )
      I_Contact( "T-21.00_DB".ChiliAwet_1.QDOSERun )
      I_Contact( "T-30.00_DB".ChiliAwet_1.QDOSERun )
      Contact( "T-02.01_DB".State.Ready_For_Transfer )
      wire#w1
      Coil( "T-31.00_DB".ChiliAwet_1.ISTART_COND )
   END_RUNG
   RUNG wire#w1
      Contact( "IO_Valve_Blending_DB"."AV-31.09".FB_OPEN )
      Coil( "T-31.00_DB".ChiliAwet_1.V_OPEN )
   END_RUNG
   RUNG wire#w1
      I_Contact( "IO_Valve_Blending_DB"."AV-31.09".FB_OPEN )
      Coil( "T-31.00_DB".ChiliAwet_1.V_CLOSE )
   END_RUNG
   RUNG wire#w1
      Contact( "IO Motor MCC Preparation_DB"."P-02.01".FB_ON )
      Coil( "T-31.00_DB".ChiliAwet_1.P_RUN )
   END_RUNG
   RUNG wire#w1
      I_Contact( "IO Motor MCC Preparation_DB"."P-02.01".FB_ON )
      Coil( "T-31.00_DB".ChiliAwet_1.P_STOP )
   END_RUNG
   // the same network as SCL:
   "T-31.00_DB".ChiliAwet_1.ISTART_COND := NOT "T-20.00_DB".ChiliAwet_1.QDOSERun AND NOT "T-21.00_DB".ChiliAwet_1.QDOSERun AND NOT "T-30.00_DB".ChiliAwet_1.QDOSERun AND "T-02.01_DB".State.Ready_For_Transfer;
   "T-31.00_DB".ChiliAwet_1.V_OPEN := "T-31.00_DB".ChiliAwet_1.ISTART_COND AND "IO_Valve_Blending_DB"."AV-31.09".FB_OPEN;
   "T-31.00_DB".ChiliAwet_1.V_CLOSE := "T-31.00_DB".ChiliAwet_1.ISTART_COND AND NOT "IO_Valve_Blending_DB"."AV-31.09".FB_OPEN;
   "T-31.00_DB".ChiliAwet_1.P_RUN := "T-31.00_DB".ChiliAwet_1.ISTART_COND AND "IO Motor MCC Preparation_DB"."P-02.01".FB_ON;
   "T-31.00_DB".ChiliAwet_1.P_STOP := "T-31.00_DB".ChiliAwet_1.ISTART_COND AND NOT "IO Motor MCC Preparation_DB"."P-02.01".FB_ON;
END_REGION

REGION Network 38: T-31_Dose_ChiliAwetan_2
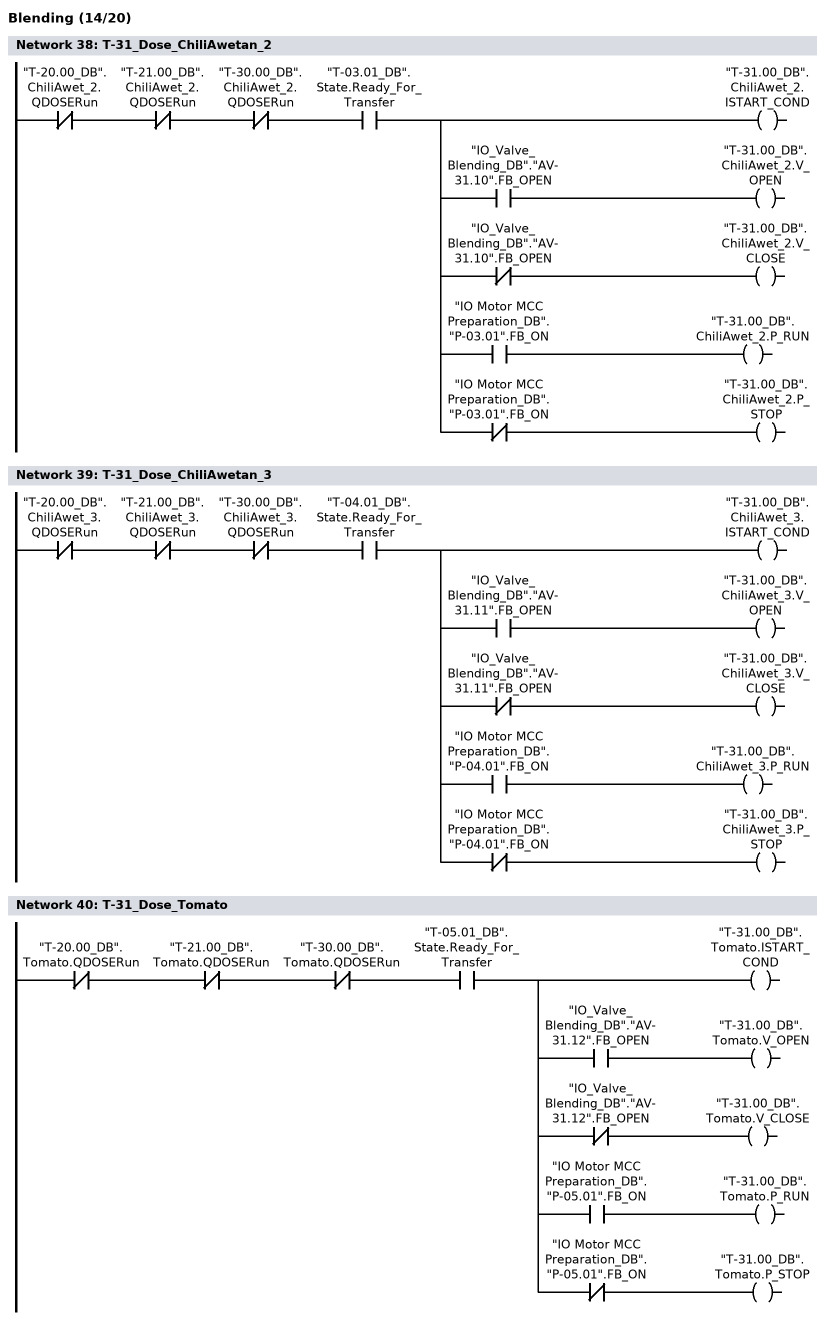
   RUNG wire#powerrail
      I_Contact( "T-20.00_DB".ChiliAwet_2.QDOSERun )
      I_Contact( "T-21.00_DB".ChiliAwet_2.QDOSERun )
      I_Contact( "T-30.00_DB".ChiliAwet_2.QDOSERun )
      Contact( "T-03.01_DB".State.Ready_For_Transfer )
      wire#w1
      Coil( "T-31.00_DB".ChiliAwet_2.ISTART_COND )
   END_RUNG
   RUNG wire#w1
      Contact( "IO_Valve_Blending_DB"."AV-31.10".FB_OPEN )
      Coil( "T-31.00_DB".ChiliAwet_2.V_OPEN )
   END_RUNG
   RUNG wire#w1
      I_Contact( "IO_Valve_Blending_DB"."AV-31.10".FB_OPEN )
      Coil( "T-31.00_DB".ChiliAwet_2.V_CLOSE )
   END_RUNG
   RUNG wire#w1
      Contact( "IO Motor MCC Preparation_DB"."P-03.01".FB_ON )
      Coil( "T-31.00_DB".ChiliAwet_2.P_RUN )
   END_RUNG
   RUNG wire#w1
      I_Contact( "IO Motor MCC Preparation_DB"."P-03.01".FB_ON )
      Coil( "T-31.00_DB".ChiliAwet_2.P_STOP )
   END_RUNG
   // the same network as SCL:
   "T-31.00_DB".ChiliAwet_2.ISTART_COND := NOT "T-20.00_DB".ChiliAwet_2.QDOSERun AND NOT "T-21.00_DB".ChiliAwet_2.QDOSERun AND NOT "T-30.00_DB".ChiliAwet_2.QDOSERun AND "T-03.01_DB".State.Ready_For_Transfer;
   "T-31.00_DB".ChiliAwet_2.V_OPEN := "T-31.00_DB".ChiliAwet_2.ISTART_COND AND "IO_Valve_Blending_DB"."AV-31.10".FB_OPEN;
   "T-31.00_DB".ChiliAwet_2.V_CLOSE := "T-31.00_DB".ChiliAwet_2.ISTART_COND AND NOT "IO_Valve_Blending_DB"."AV-31.10".FB_OPEN;
   "T-31.00_DB".ChiliAwet_2.P_RUN := "T-31.00_DB".ChiliAwet_2.ISTART_COND AND "IO Motor MCC Preparation_DB"."P-03.01".FB_ON;
   "T-31.00_DB".ChiliAwet_2.P_STOP := "T-31.00_DB".ChiliAwet_2.ISTART_COND AND NOT "IO Motor MCC Preparation_DB"."P-03.01".FB_ON;
END_REGION

REGION Network 39: T-31_Dose_ChiliAwetan_3
   RUNG wire#powerrail
      I_Contact( "T-20.00_DB".ChiliAwet_3.QDOSERun )
      I_Contact( "T-21.00_DB".ChiliAwet_3.QDOSERun )
      I_Contact( "T-30.00_DB".ChiliAwet_3.QDOSERun )
      Contact( "T-04.01_DB".State.Ready_For_Transfer )
      wire#w1
      Coil( "T-31.00_DB".ChiliAwet_3.ISTART_COND )
   END_RUNG
   RUNG wire#w1
      Contact( "IO_Valve_Blending_DB"."AV-31.11".FB_OPEN )
      Coil( "T-31.00_DB".ChiliAwet_3.V_OPEN )
   END_RUNG
   RUNG wire#w1
      I_Contact( "IO_Valve_Blending_DB"."AV-31.11".FB_OPEN )
      Coil( "T-31.00_DB".ChiliAwet_3.V_CLOSE )
   END_RUNG
   RUNG wire#w1
      Contact( "IO Motor MCC Preparation_DB"."P-04.01".FB_ON )
      Coil( "T-31.00_DB".ChiliAwet_3.P_RUN )
   END_RUNG
   RUNG wire#w1
      I_Contact( "IO Motor MCC Preparation_DB"."P-04.01".FB_ON )
      Coil( "T-31.00_DB".ChiliAwet_3.P_STOP )
   END_RUNG
   // the same network as SCL:
   "T-31.00_DB".ChiliAwet_3.ISTART_COND := NOT "T-20.00_DB".ChiliAwet_3.QDOSERun AND NOT "T-21.00_DB".ChiliAwet_3.QDOSERun AND NOT "T-30.00_DB".ChiliAwet_3.QDOSERun AND "T-04.01_DB".State.Ready_For_Transfer;
   "T-31.00_DB".ChiliAwet_3.V_OPEN := "T-31.00_DB".ChiliAwet_3.ISTART_COND AND "IO_Valve_Blending_DB"."AV-31.11".FB_OPEN;
   "T-31.00_DB".ChiliAwet_3.V_CLOSE := "T-31.00_DB".ChiliAwet_3.ISTART_COND AND NOT "IO_Valve_Blending_DB"."AV-31.11".FB_OPEN;
   "T-31.00_DB".ChiliAwet_3.P_RUN := "T-31.00_DB".ChiliAwet_3.ISTART_COND AND "IO Motor MCC Preparation_DB"."P-04.01".FB_ON;
   "T-31.00_DB".ChiliAwet_3.P_STOP := "T-31.00_DB".ChiliAwet_3.ISTART_COND AND NOT "IO Motor MCC Preparation_DB"."P-04.01".FB_ON;
END_REGION

REGION Network 40: T-31_Dose_Tomato
   RUNG wire#powerrail
      I_Contact( "T-20.00_DB".Tomato.QDOSERun )
      I_Contact( "T-21.00_DB".Tomato.QDOSERun )
      I_Contact( "T-30.00_DB".Tomato.QDOSERun )
      Contact( "T-05.01_DB".State.Ready_For_Transfer )
      wire#w1
      Coil( "T-31.00_DB".Tomato.ISTART_COND )
   END_RUNG
   RUNG wire#w1
      Contact( "IO_Valve_Blending_DB"."AV-31.12".FB_OPEN )
      Coil( "T-31.00_DB".Tomato.V_OPEN )
   END_RUNG
   RUNG wire#w1
      I_Contact( "IO_Valve_Blending_DB"."AV-31.12".FB_OPEN )
      Coil( "T-31.00_DB".Tomato.V_CLOSE )
   END_RUNG
   RUNG wire#w1
      Contact( "IO Motor MCC Preparation_DB"."P-05.01".FB_ON )
      Coil( "T-31.00_DB".Tomato.P_RUN )
   END_RUNG
   RUNG wire#w1
      I_Contact( "IO Motor MCC Preparation_DB"."P-05.01".FB_ON )
      Coil( "T-31.00_DB".Tomato.P_STOP )
   END_RUNG
   // the same network as SCL:
   "T-31.00_DB".Tomato.ISTART_COND := NOT "T-20.00_DB".Tomato.QDOSERun AND NOT "T-21.00_DB".Tomato.QDOSERun AND NOT "T-30.00_DB".Tomato.QDOSERun AND "T-05.01_DB".State.Ready_For_Transfer;
   "T-31.00_DB".Tomato.V_OPEN := "T-31.00_DB".Tomato.ISTART_COND AND "IO_Valve_Blending_DB"."AV-31.12".FB_OPEN;
   "T-31.00_DB".Tomato.V_CLOSE := "T-31.00_DB".Tomato.ISTART_COND AND NOT "IO_Valve_Blending_DB"."AV-31.12".FB_OPEN;
   "T-31.00_DB".Tomato.P_RUN := "T-31.00_DB".Tomato.ISTART_COND AND "IO Motor MCC Preparation_DB"."P-05.01".FB_ON;
   "T-31.00_DB".Tomato.P_STOP := "T-31.00_DB".Tomato.ISTART_COND AND NOT "IO Motor MCC Preparation_DB"."P-05.01".FB_ON;
END_REGION

REGION Network 41: T-31_Dose_FreshChili_1
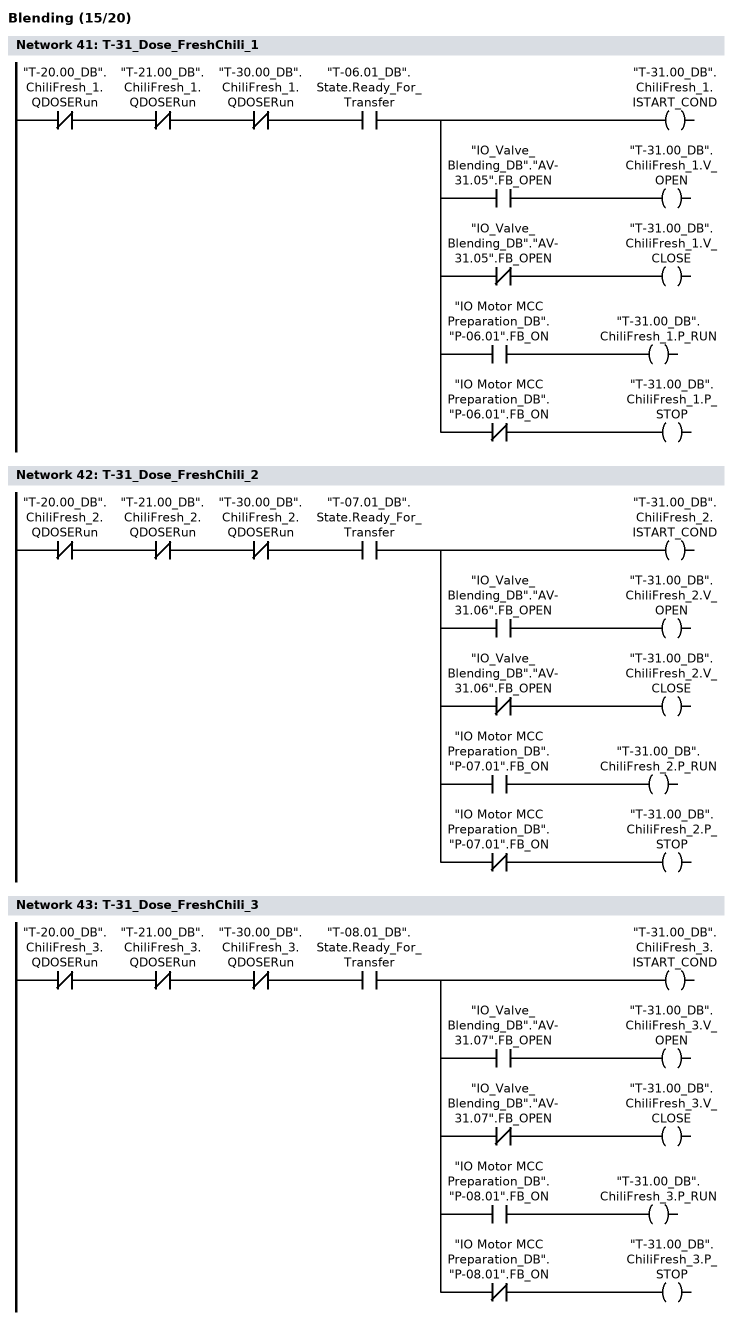
   RUNG wire#powerrail
      I_Contact( "T-20.00_DB".ChiliFresh_1.QDOSERun )
      I_Contact( "T-21.00_DB".ChiliFresh_1.QDOSERun )
      I_Contact( "T-30.00_DB".ChiliFresh_1.QDOSERun )
      Contact( "T-06.01_DB".State.Ready_For_Transfer )
      wire#w1
      Coil( "T-31.00_DB".ChiliFresh_1.ISTART_COND )
   END_RUNG
   RUNG wire#w1
      Contact( "IO_Valve_Blending_DB"."AV-31.05".FB_OPEN )
      Coil( "T-31.00_DB".ChiliFresh_1.V_OPEN )
   END_RUNG
   RUNG wire#w1
      I_Contact( "IO_Valve_Blending_DB"."AV-31.05".FB_OPEN )
      Coil( "T-31.00_DB".ChiliFresh_1.V_CLOSE )
   END_RUNG
   RUNG wire#w1
      Contact( "IO Motor MCC Preparation_DB"."P-06.01".FB_ON )
      Coil( "T-31.00_DB".ChiliFresh_1.P_RUN )
   END_RUNG
   RUNG wire#w1
      I_Contact( "IO Motor MCC Preparation_DB"."P-06.01".FB_ON )
      Coil( "T-31.00_DB".ChiliFresh_1.P_STOP )
   END_RUNG
   // the same network as SCL:
   "T-31.00_DB".ChiliFresh_1.ISTART_COND := NOT "T-20.00_DB".ChiliFresh_1.QDOSERun AND NOT "T-21.00_DB".ChiliFresh_1.QDOSERun AND NOT "T-30.00_DB".ChiliFresh_1.QDOSERun AND "T-06.01_DB".State.Ready_For_Transfer;
   "T-31.00_DB".ChiliFresh_1.V_OPEN := "T-31.00_DB".ChiliFresh_1.ISTART_COND AND "IO_Valve_Blending_DB"."AV-31.05".FB_OPEN;
   "T-31.00_DB".ChiliFresh_1.V_CLOSE := "T-31.00_DB".ChiliFresh_1.ISTART_COND AND NOT "IO_Valve_Blending_DB"."AV-31.05".FB_OPEN;
   "T-31.00_DB".ChiliFresh_1.P_RUN := "T-31.00_DB".ChiliFresh_1.ISTART_COND AND "IO Motor MCC Preparation_DB"."P-06.01".FB_ON;
   "T-31.00_DB".ChiliFresh_1.P_STOP := "T-31.00_DB".ChiliFresh_1.ISTART_COND AND NOT "IO Motor MCC Preparation_DB"."P-06.01".FB_ON;
END_REGION

REGION Network 42: T-31_Dose_FreshChili_2
   RUNG wire#powerrail
      I_Contact( "T-20.00_DB".ChiliFresh_2.QDOSERun )
      I_Contact( "T-21.00_DB".ChiliFresh_2.QDOSERun )
      I_Contact( "T-30.00_DB".ChiliFresh_2.QDOSERun )
      Contact( "T-07.01_DB".State.Ready_For_Transfer )
      wire#w1
      Coil( "T-31.00_DB".ChiliFresh_2.ISTART_COND )
   END_RUNG
   RUNG wire#w1
      Contact( "IO_Valve_Blending_DB"."AV-31.06".FB_OPEN )
      Coil( "T-31.00_DB".ChiliFresh_2.V_OPEN )
   END_RUNG
   RUNG wire#w1
      I_Contact( "IO_Valve_Blending_DB"."AV-31.06".FB_OPEN )
      Coil( "T-31.00_DB".ChiliFresh_2.V_CLOSE )
   END_RUNG
   RUNG wire#w1
      Contact( "IO Motor MCC Preparation_DB"."P-07.01".FB_ON )
      Coil( "T-31.00_DB".ChiliFresh_2.P_RUN )
   END_RUNG
   RUNG wire#w1
      I_Contact( "IO Motor MCC Preparation_DB"."P-07.01".FB_ON )
      Coil( "T-31.00_DB".ChiliFresh_2.P_STOP )
   END_RUNG
   // the same network as SCL:
   "T-31.00_DB".ChiliFresh_2.ISTART_COND := NOT "T-20.00_DB".ChiliFresh_2.QDOSERun AND NOT "T-21.00_DB".ChiliFresh_2.QDOSERun AND NOT "T-30.00_DB".ChiliFresh_2.QDOSERun AND "T-07.01_DB".State.Ready_For_Transfer;
   "T-31.00_DB".ChiliFresh_2.V_OPEN := "T-31.00_DB".ChiliFresh_2.ISTART_COND AND "IO_Valve_Blending_DB"."AV-31.06".FB_OPEN;
   "T-31.00_DB".ChiliFresh_2.V_CLOSE := "T-31.00_DB".ChiliFresh_2.ISTART_COND AND NOT "IO_Valve_Blending_DB"."AV-31.06".FB_OPEN;
   "T-31.00_DB".ChiliFresh_2.P_RUN := "T-31.00_DB".ChiliFresh_2.ISTART_COND AND "IO Motor MCC Preparation_DB"."P-07.01".FB_ON;
   "T-31.00_DB".ChiliFresh_2.P_STOP := "T-31.00_DB".ChiliFresh_2.ISTART_COND AND NOT "IO Motor MCC Preparation_DB"."P-07.01".FB_ON;
END_REGION

REGION Network 43: T-31_Dose_FreshChili_3
   RUNG wire#powerrail
      I_Contact( "T-20.00_DB".ChiliFresh_3.QDOSERun )
      I_Contact( "T-21.00_DB".ChiliFresh_3.QDOSERun )
      I_Contact( "T-30.00_DB".ChiliFresh_3.QDOSERun )
      Contact( "T-08.01_DB".State.Ready_For_Transfer )
      wire#w1
      Coil( "T-31.00_DB".ChiliFresh_3.ISTART_COND )
   END_RUNG
   RUNG wire#w1
      Contact( "IO_Valve_Blending_DB"."AV-31.07".FB_OPEN )
      Coil( "T-31.00_DB".ChiliFresh_3.V_OPEN )
   END_RUNG
   RUNG wire#w1
      I_Contact( "IO_Valve_Blending_DB"."AV-31.07".FB_OPEN )
      Coil( "T-31.00_DB".ChiliFresh_3.V_CLOSE )
   END_RUNG
   RUNG wire#w1
      Contact( "IO Motor MCC Preparation_DB"."P-08.01".FB_ON )
      Coil( "T-31.00_DB".ChiliFresh_3.P_RUN )
   END_RUNG
   RUNG wire#w1
      I_Contact( "IO Motor MCC Preparation_DB"."P-08.01".FB_ON )
      Coil( "T-31.00_DB".ChiliFresh_3.P_STOP )
   END_RUNG
   // the same network as SCL:
   "T-31.00_DB".ChiliFresh_3.ISTART_COND := NOT "T-20.00_DB".ChiliFresh_3.QDOSERun AND NOT "T-21.00_DB".ChiliFresh_3.QDOSERun AND NOT "T-30.00_DB".ChiliFresh_3.QDOSERun AND "T-08.01_DB".State.Ready_For_Transfer;
   "T-31.00_DB".ChiliFresh_3.V_OPEN := "T-31.00_DB".ChiliFresh_3.ISTART_COND AND "IO_Valve_Blending_DB"."AV-31.07".FB_OPEN;
   "T-31.00_DB".ChiliFresh_3.V_CLOSE := "T-31.00_DB".ChiliFresh_3.ISTART_COND AND NOT "IO_Valve_Blending_DB"."AV-31.07".FB_OPEN;
   "T-31.00_DB".ChiliFresh_3.P_RUN := "T-31.00_DB".ChiliFresh_3.ISTART_COND AND "IO Motor MCC Preparation_DB"."P-08.01".FB_ON;
   "T-31.00_DB".ChiliFresh_3.P_STOP := "T-31.00_DB".ChiliFresh_3.ISTART_COND AND NOT "IO Motor MCC Preparation_DB"."P-08.01".FB_ON;
END_REGION

REGION Network 44: T-31_Dose_Garlic
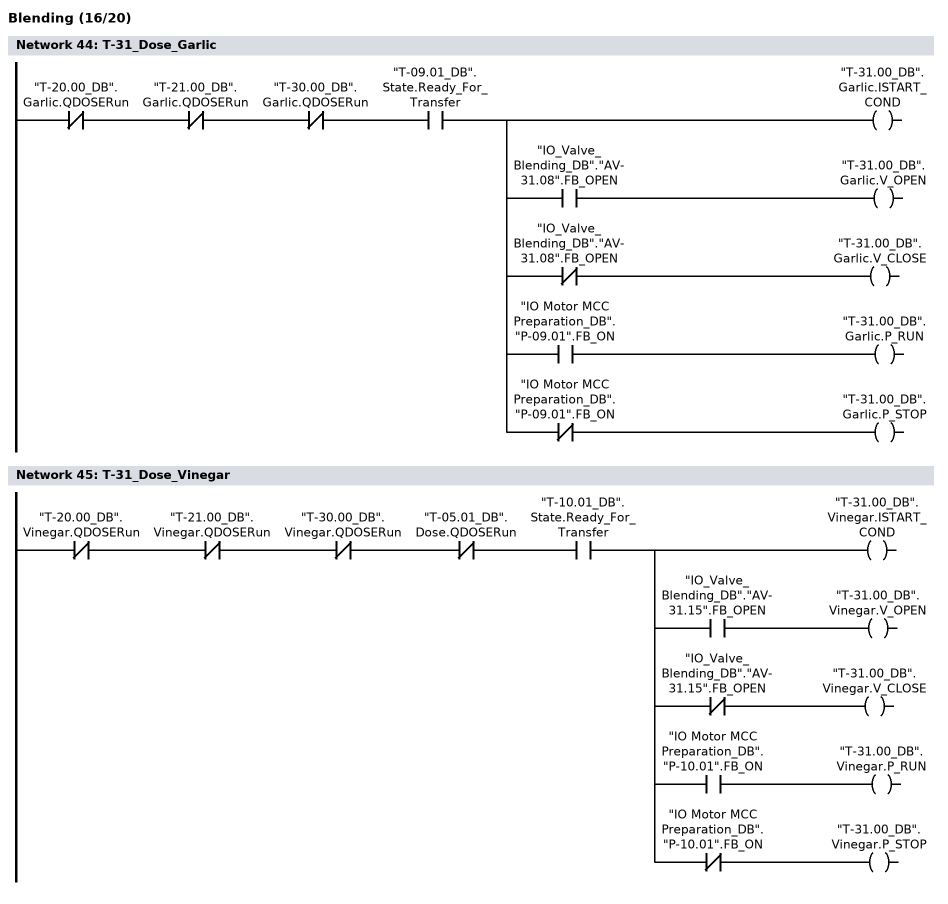
   RUNG wire#powerrail
      I_Contact( "T-20.00_DB".Garlic.QDOSERun )
      I_Contact( "T-21.00_DB".Garlic.QDOSERun )
      I_Contact( "T-30.00_DB".Garlic.QDOSERun )
      Contact( "T-09.01_DB".State.Ready_For_Transfer )
      wire#w1
      Coil( "T-31.00_DB".Garlic.ISTART_COND )
   END_RUNG
   RUNG wire#w1
      Contact( "IO_Valve_Blending_DB"."AV-31.08".FB_OPEN )
      Coil( "T-31.00_DB".Garlic.V_OPEN )
   END_RUNG
   RUNG wire#w1
      I_Contact( "IO_Valve_Blending_DB"."AV-31.08".FB_OPEN )
      Coil( "T-31.00_DB".Garlic.V_CLOSE )
   END_RUNG
   RUNG wire#w1
      Contact( "IO Motor MCC Preparation_DB"."P-09.01".FB_ON )
      Coil( "T-31.00_DB".Garlic.P_RUN )
   END_RUNG
   RUNG wire#w1
      I_Contact( "IO Motor MCC Preparation_DB"."P-09.01".FB_ON )
      Coil( "T-31.00_DB".Garlic.P_STOP )
   END_RUNG
   // the same network as SCL:
   "T-31.00_DB".Garlic.ISTART_COND := NOT "T-20.00_DB".Garlic.QDOSERun AND NOT "T-21.00_DB".Garlic.QDOSERun AND NOT "T-30.00_DB".Garlic.QDOSERun AND "T-09.01_DB".State.Ready_For_Transfer;
   "T-31.00_DB".Garlic.V_OPEN := "T-31.00_DB".Garlic.ISTART_COND AND "IO_Valve_Blending_DB"."AV-31.08".FB_OPEN;
   "T-31.00_DB".Garlic.V_CLOSE := "T-31.00_DB".Garlic.ISTART_COND AND NOT "IO_Valve_Blending_DB"."AV-31.08".FB_OPEN;
   "T-31.00_DB".Garlic.P_RUN := "T-31.00_DB".Garlic.ISTART_COND AND "IO Motor MCC Preparation_DB"."P-09.01".FB_ON;
   "T-31.00_DB".Garlic.P_STOP := "T-31.00_DB".Garlic.ISTART_COND AND NOT "IO Motor MCC Preparation_DB"."P-09.01".FB_ON;
END_REGION

REGION Network 45: T-31_Dose_Vinegar
   RUNG wire#powerrail
      I_Contact( "T-20.00_DB".Vinegar.QDOSERun )
      I_Contact( "T-21.00_DB".Vinegar.QDOSERun )
      I_Contact( "T-30.00_DB".Vinegar.QDOSERun )
      I_Contact( "T-05.01_DB".Dose.QDOSERun )
      Contact( "T-10.01_DB".State.Ready_For_Transfer )
      wire#w1
      Coil( "T-31.00_DB".Vinegar.ISTART_COND )
   END_RUNG
   RUNG wire#w1
      Contact( "IO_Valve_Blending_DB"."AV-31.15".FB_OPEN )
      Coil( "T-31.00_DB".Vinegar.V_OPEN )
   END_RUNG
   RUNG wire#w1
      I_Contact( "IO_Valve_Blending_DB"."AV-31.15".FB_OPEN )
      Coil( "T-31.00_DB".Vinegar.V_CLOSE )
   END_RUNG
   RUNG wire#w1
      Contact( "IO Motor MCC Preparation_DB"."P-10.01".FB_ON )
      Coil( "T-31.00_DB".Vinegar.P_RUN )
   END_RUNG
   RUNG wire#w1
      I_Contact( "IO Motor MCC Preparation_DB"."P-10.01".FB_ON )
      Coil( "T-31.00_DB".Vinegar.P_STOP )
   END_RUNG
   // the same network as SCL:
   "T-31.00_DB".Vinegar.ISTART_COND := NOT "T-20.00_DB".Vinegar.QDOSERun AND NOT "T-21.00_DB".Vinegar.QDOSERun AND NOT "T-30.00_DB".Vinegar.QDOSERun AND NOT "T-05.01_DB".Dose.QDOSERun AND "T-10.01_DB".State.Ready_For_Transfer;
   "T-31.00_DB".Vinegar.V_OPEN := "T-31.00_DB".Vinegar.ISTART_COND AND "IO_Valve_Blending_DB"."AV-31.15".FB_OPEN;
   "T-31.00_DB".Vinegar.V_CLOSE := "T-31.00_DB".Vinegar.ISTART_COND AND NOT "IO_Valve_Blending_DB"."AV-31.15".FB_OPEN;
   "T-31.00_DB".Vinegar.P_RUN := "T-31.00_DB".Vinegar.ISTART_COND AND "IO Motor MCC Preparation_DB"."P-10.01".FB_ON;
   "T-31.00_DB".Vinegar.P_STOP := "T-31.00_DB".Vinegar.ISTART_COND AND NOT "IO Motor MCC Preparation_DB"."P-10.01".FB_ON;
END_REGION

REGION Network 46: T-31.00
   // "IO Analog Blending_DB"."LT-31.01".QOUT
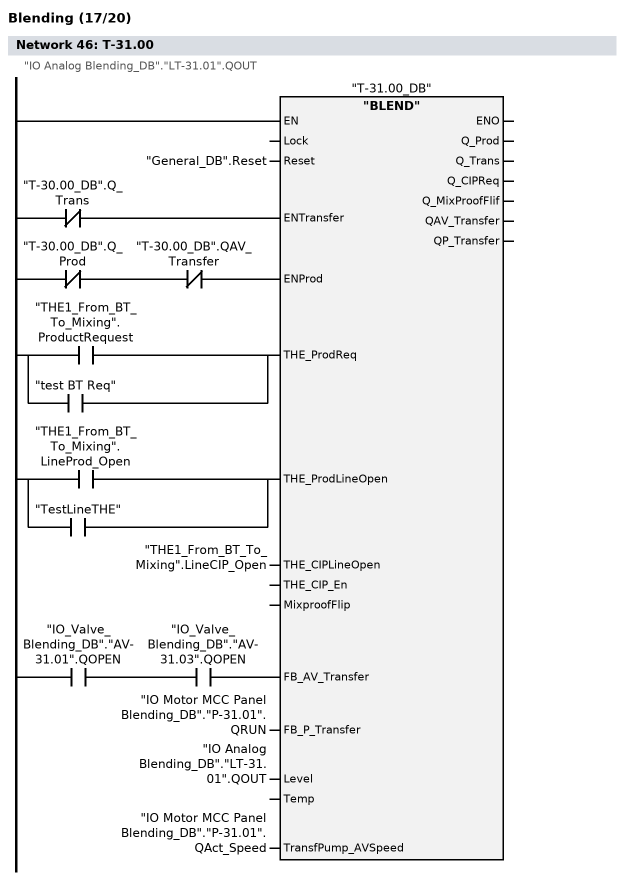
   RUNG wire#powerrail
      "T-31.00_DB"(ENTransfer := wire#w1, ENProd := wire#w2, THE_ProdReq := wire#w3, THE_ProdLineOpen := wire#w4, FB_AV_Transfer := wire#w5, Lock :=, Reset := "General_DB".Reset, THE_CIPLineOpen := "THE1_From_BT_To_Mixing".LineCIP_Open, THE_CIP_En :=, MixproofFlip :=, FB_P_Transfer := "IO Motor MCC Panel Blending_DB"."P-31.01".QRUN, Level := "IO Analog Blending_DB"."LT-31.01".QOUT, Temp :=, TransfPump_AVSpeed := "IO Motor MCC Panel Blending_DB"."P-31.01".QAct_Speed, Q_Prod =>, Q_Trans =>, Q_CIPReq =>, Q_MixProofFlif =>, QAV_Transfer =>, QP_Transfer =>)
   END_RUNG
   RUNG wire#powerrail
      I_Contact( "T-30.00_DB".Q_Trans )
   END_RUNG wire#w1
   RUNG wire#powerrail
      I_Contact( "T-30.00_DB".Q_Prod )
      I_Contact( "T-30.00_DB".QAV_Transfer )
   END_RUNG wire#w2
   RUNG wire#powerrail
      Contact( "THE1_From_BT_To_Mixing".ProductRequest )
   END_RUNG wire#w3
   RUNG wire#powerrail
      Contact( "test BT Req" )
   END_RUNG wire#w3
   RUNG wire#powerrail
      Contact( "THE1_From_BT_To_Mixing".LineProd_Open )
   END_RUNG wire#w4
   RUNG wire#powerrail
      Contact( "TestLineTHE" )
   END_RUNG wire#w4
   RUNG wire#powerrail
      Contact( "IO_Valve_Blending_DB"."AV-31.01".QOPEN )
      Contact( "IO_Valve_Blending_DB"."AV-31.03".QOPEN )
   END_RUNG wire#w5
   // the same network as SCL:
   "T-31.00_DB"(Reset := "General_DB".Reset,   // "BLEND"
                ENTransfer := NOT "T-30.00_DB".Q_Trans,
                ENProd := NOT "T-30.00_DB".Q_Prod AND NOT "T-30.00_DB".QAV_Transfer,
                THE_ProdReq := "THE1_From_BT_To_Mixing".ProductRequest OR "test BT Req",
                THE_ProdLineOpen := "THE1_From_BT_To_Mixing".LineProd_Open OR "TestLineTHE",
                THE_CIPLineOpen := "THE1_From_BT_To_Mixing".LineCIP_Open,
                FB_AV_Transfer := "IO_Valve_Blending_DB"."AV-31.01".QOPEN AND "IO_Valve_Blending_DB"."AV-31.03".QOPEN,
                FB_P_Transfer := "IO Motor MCC Panel Blending_DB"."P-31.01".QRUN,
                Level := "IO Analog Blending_DB"."LT-31.01".QOUT,
                TransfPump_AVSpeed := "IO Motor MCC Panel Blending_DB"."P-31.01".QAct_Speed);
END_REGION

REGION Network 47: Comm to Buffer Tank THE 1
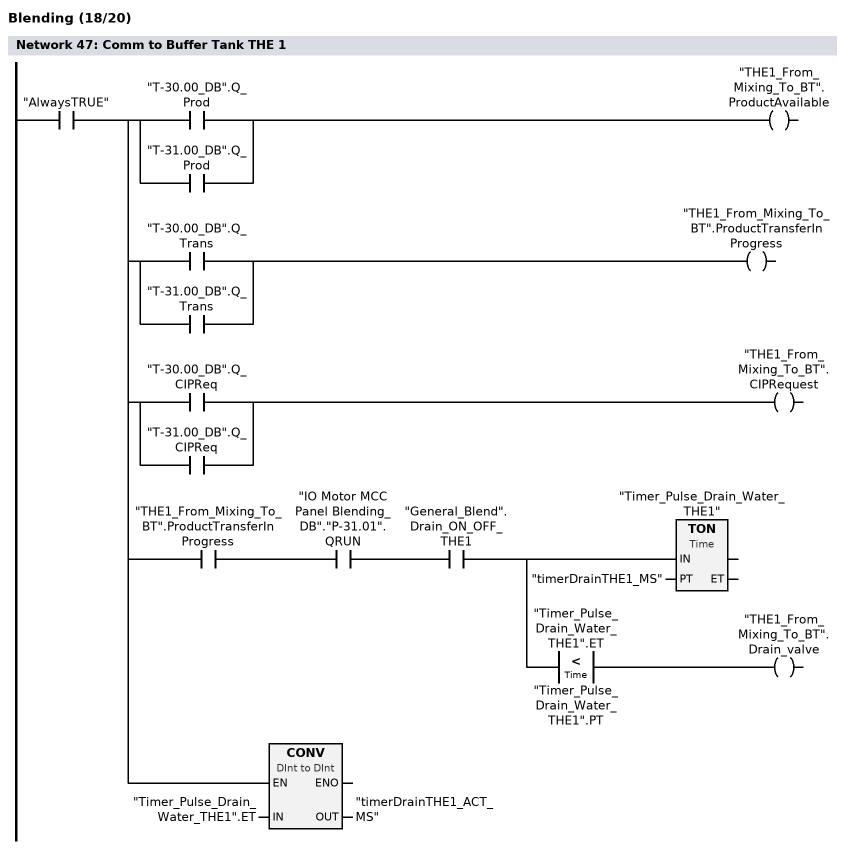
   RUNG wire#powerrail
      Contact( "AlwaysTRUE" )
      wire#w1
      Contact( "T-30.00_DB".Q_Prod )
      wire#w2
      Coil( "THE1_From_Mixing_To_BT".ProductAvailable )
   END_RUNG
   RUNG wire#w1
      Contact( "T-31.00_DB".Q_Prod )
   END_RUNG wire#w2
   RUNG wire#w1
      Contact( "T-30.00_DB".Q_Trans )
      wire#w3
      Coil( "THE1_From_Mixing_To_BT".ProductTransferInProgress )
   END_RUNG
   RUNG wire#w1
      Contact( "T-31.00_DB".Q_Trans )
   END_RUNG wire#w3
   RUNG wire#w1
      Contact( "T-30.00_DB".Q_CIPReq )
      wire#w4
      Coil( "THE1_From_Mixing_To_BT".CIPRequest )
   END_RUNG
   RUNG wire#w1
      Contact( "T-31.00_DB".Q_CIPReq )
   END_RUNG wire#w4
   RUNG wire#w1
      Contact( "THE1_From_Mixing_To_BT".ProductTransferInProgress )
      Contact( "IO Motor MCC Panel Blending_DB"."P-31.01".QRUN )
      Contact( "General_Blend".Drain_ON_OFF_THE1 )
      wire#w5
      { S7_Templates := "time_type := Time" } "Timer_Pulse_Drain_Water_THE1".TON(pt := "timerDrainTHE1_MS", et =>)
   END_RUNG
   RUNG wire#w5
      { S7_Templates := "SrcType := Time" } LT_Contact(in1 := "Timer_Pulse_Drain_Water_THE1".ET, in2 := "Timer_Pulse_Drain_Water_THE1".PT)
      Coil( "THE1_From_Mixing_To_BT".Drain_valve )
   END_RUNG
   RUNG wire#w1
      { S7_Templates := "[SrcType := DInt, DestType := DInt]" } Convert(in := "Timer_Pulse_Drain_Water_THE1".ET, out => "timerDrainTHE1_ACT_MS")
   END_RUNG
   // the same network as SCL:
   "THE1_From_Mixing_To_BT".ProductAvailable := "AlwaysTRUE" AND ("T-30.00_DB".Q_Prod OR "T-31.00_DB".Q_Prod);
   "THE1_From_Mixing_To_BT".ProductTransferInProgress := "AlwaysTRUE" AND ("T-30.00_DB".Q_Trans OR "T-31.00_DB".Q_Trans);
   "THE1_From_Mixing_To_BT".CIPRequest := "AlwaysTRUE" AND ("T-30.00_DB".Q_CIPReq OR "T-31.00_DB".Q_CIPReq);
   #_w1 := "AlwaysTRUE" AND "THE1_From_Mixing_To_BT".ProductTransferInProgress AND "IO Motor MCC Panel Blending_DB"."P-31.01".QRUN AND "General_Blend".Drain_ON_OFF_THE1;
   "Timer_Pulse_Drain_Water_THE1".TON(IN := #_w1, PT := "timerDrainTHE1_MS");
   "THE1_From_Mixing_To_BT".Drain_valve := #_w1 AND ("Timer_Pulse_Drain_Water_THE1".ET < "Timer_Pulse_Drain_Water_THE1".PT);
   IF "AlwaysTRUE" THEN "timerDrainTHE1_ACT_MS" := DINT_TO_DINT("Timer_Pulse_Drain_Water_THE1".ET); END_IF;
END_REGION

REGION Network 48: Rework T-22
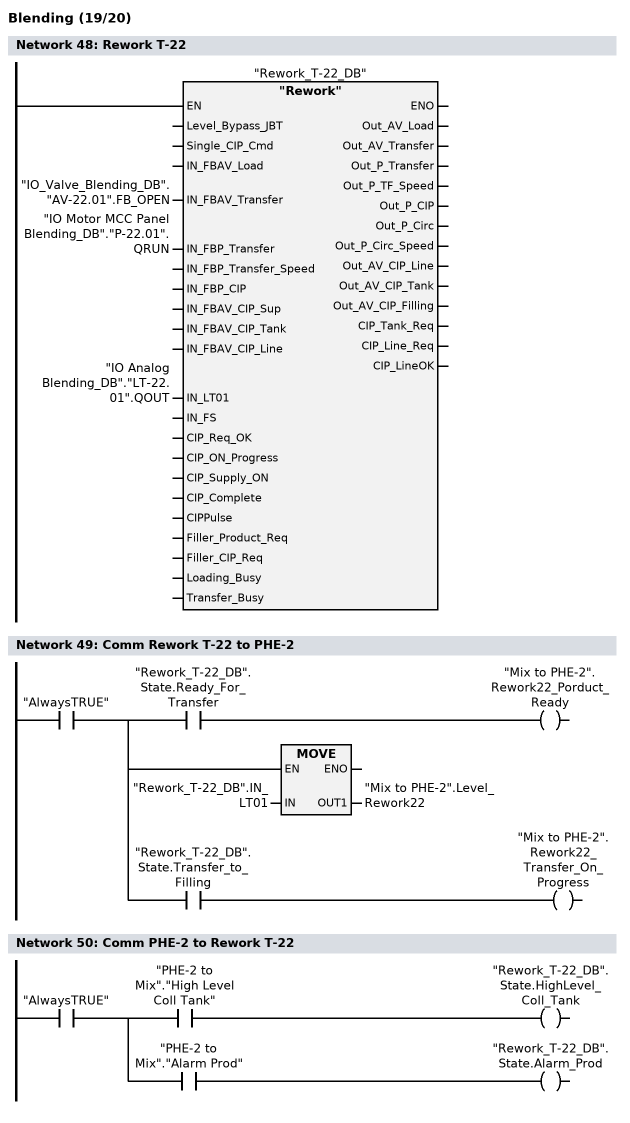
   RUNG wire#powerrail
      "Rework_T-22_DB"(Level_Bypass_JBT :=, Single_CIP_Cmd :=, IN_FBAV_Load :=, IN_FBAV_Transfer := "IO_Valve_Blending_DB"."AV-22.01".FB_OPEN, IN_FBP_Transfer := "IO Motor MCC Panel Blending_DB"."P-22.01".QRUN, IN_FBP_Transfer_Speed :=, IN_FBP_CIP :=, IN_FBAV_CIP_Sup :=, IN_FBAV_CIP_Tank :=, IN_FBAV_CIP_Line :=, IN_LT01 := "IO Analog Blending_DB"."LT-22.01".QOUT, IN_FS :=, CIP_Req_OK :=, CIP_ON_Progress :=, CIP_Supply_ON :=, CIP_Complete :=, CIPPulse :=, Filler_Product_Req :=, Filler_CIP_Req :=, Loading_Busy :=, Transfer_Busy :=, Out_AV_Load =>, Out_AV_Transfer =>, Out_P_Transfer =>, Out_P_TF_Speed =>, Out_P_CIP =>, Out_P_Circ =>, Out_P_Circ_Speed =>, Out_AV_CIP_Line =>, Out_AV_CIP_Tank =>, Out_AV_CIP_Filling =>, CIP_Tank_Req =>, CIP_Line_Req =>, CIP_LineOK =>)
   END_RUNG
   // the same network as SCL:
   "Rework_T-22_DB"(IN_FBAV_Transfer := "IO_Valve_Blending_DB"."AV-22.01".FB_OPEN,   // "Rework"
                    IN_FBP_Transfer := "IO Motor MCC Panel Blending_DB"."P-22.01".QRUN,
                    IN_LT01 := "IO Analog Blending_DB"."LT-22.01".QOUT);
END_REGION

REGION Network 49: Comm Rework T-22 to PHE-2
   RUNG wire#powerrail
      Contact( "AlwaysTRUE" )
      wire#w1
      Contact( "Rework_T-22_DB".State.Ready_For_Transfer )
      Coil( "Mix to PHE-2".Rework22_Porduct_Ready )
   END_RUNG
   RUNG wire#w1
      Move(in := "Rework_T-22_DB".IN_LT01, out1 => "Mix to PHE-2".Level_Rework22)
   END_RUNG
   RUNG wire#w1
      Contact( "Rework_T-22_DB".State.Transfer_to_Filling )
      Coil( "Mix to PHE-2".Rework22_Transfer_On_Progress )
   END_RUNG
   // the same network as SCL:
   "Mix to PHE-2".Rework22_Porduct_Ready := "AlwaysTRUE" AND "Rework_T-22_DB".State.Ready_For_Transfer;
   IF "AlwaysTRUE" THEN "Mix to PHE-2".Level_Rework22 := "Rework_T-22_DB".IN_LT01; END_IF;
   "Mix to PHE-2".Rework22_Transfer_On_Progress := "AlwaysTRUE" AND "Rework_T-22_DB".State.Transfer_to_Filling;
END_REGION

REGION Network 50: Comm PHE-2 to Rework T-22
   RUNG wire#powerrail
      Contact( "AlwaysTRUE" )
      wire#w1
      Contact( "PHE-2 to Mix"."High Level Coll Tank" )
      Coil( "Rework_T-22_DB".State.HighLevel_Coll_Tank )
   END_RUNG
   RUNG wire#w1
      Contact( "PHE-2 to Mix"."Alarm Prod" )
      Coil( "Rework_T-22_DB".State.Alarm_Prod )
   END_RUNG
   // the same network as SCL:
   "Rework_T-22_DB".State.HighLevel_Coll_Tank := "AlwaysTRUE" AND "PHE-2 to Mix"."High Level Coll Tank";
   "Rework_T-22_DB".State.Alarm_Prod := "AlwaysTRUE" AND "PHE-2 to Mix"."Alarm Prod";
END_REGION

REGION Network 51: Rework T-32
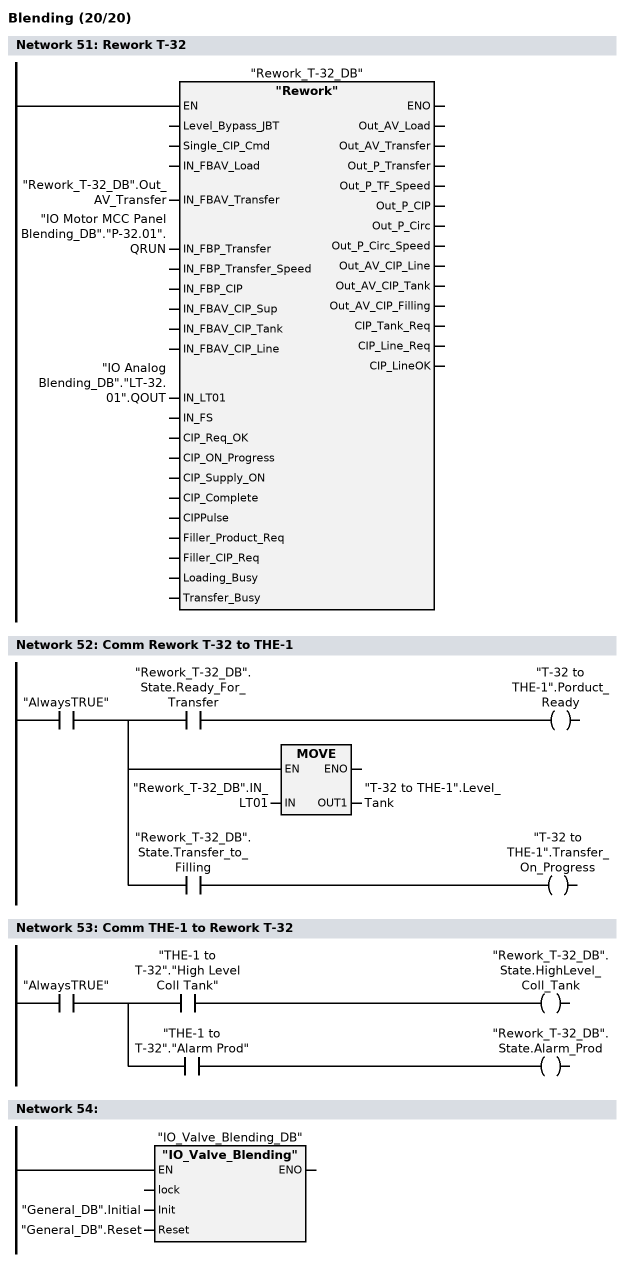
   RUNG wire#powerrail
      "Rework_T-32_DB"(Level_Bypass_JBT :=, Single_CIP_Cmd :=, IN_FBAV_Load :=, IN_FBAV_Transfer := "Rework_T-32_DB".Out_AV_Transfer, IN_FBP_Transfer := "IO Motor MCC Panel Blending_DB"."P-32.01".QRUN, IN_FBP_Transfer_Speed :=, IN_FBP_CIP :=, IN_FBAV_CIP_Sup :=, IN_FBAV_CIP_Tank :=, IN_FBAV_CIP_Line :=, IN_LT01 := "IO Analog Blending_DB"."LT-32.01".QOUT, IN_FS :=, CIP_Req_OK :=, CIP_ON_Progress :=, CIP_Supply_ON :=, CIP_Complete :=, CIPPulse :=, Filler_Product_Req :=, Filler_CIP_Req :=, Loading_Busy :=, Transfer_Busy :=, Out_AV_Load =>, Out_AV_Transfer =>, Out_P_Transfer =>, Out_P_TF_Speed =>, Out_P_CIP =>, Out_P_Circ =>, Out_P_Circ_Speed =>, Out_AV_CIP_Line =>, Out_AV_CIP_Tank =>, Out_AV_CIP_Filling =>, CIP_Tank_Req =>, CIP_Line_Req =>, CIP_LineOK =>)
   END_RUNG
   // the same network as SCL:
   "Rework_T-32_DB"(IN_FBAV_Transfer := "Rework_T-32_DB".Out_AV_Transfer,   // "Rework"
                    IN_FBP_Transfer := "IO Motor MCC Panel Blending_DB"."P-32.01".QRUN,
                    IN_LT01 := "IO Analog Blending_DB"."LT-32.01".QOUT);
END_REGION

REGION Network 52: Comm Rework T-32 to THE-1
   RUNG wire#powerrail
      Contact( "AlwaysTRUE" )
      wire#w1
      Contact( "Rework_T-32_DB".State.Ready_For_Transfer )
      Coil( "T-32 to THE-1".Porduct_Ready )
   END_RUNG
   RUNG wire#w1
      Move(in := "Rework_T-32_DB".IN_LT01, out1 => "T-32 to THE-1".Level_Tank)
   END_RUNG
   RUNG wire#w1
      Contact( "Rework_T-32_DB".State.Transfer_to_Filling )
      Coil( "T-32 to THE-1".Transfer_On_Progress )
   END_RUNG
   // the same network as SCL:
   "T-32 to THE-1".Porduct_Ready := "AlwaysTRUE" AND "Rework_T-32_DB".State.Ready_For_Transfer;
   IF "AlwaysTRUE" THEN "T-32 to THE-1".Level_Tank := "Rework_T-32_DB".IN_LT01; END_IF;
   "T-32 to THE-1".Transfer_On_Progress := "AlwaysTRUE" AND "Rework_T-32_DB".State.Transfer_to_Filling;
END_REGION

REGION Network 53: Comm THE-1 to Rework T-32
   RUNG wire#powerrail
      Contact( "AlwaysTRUE" )
      wire#w1
      Contact( "THE-1 to T-32"."High Level Coll Tank" )
      Coil( "Rework_T-32_DB".State.HighLevel_Coll_Tank )
   END_RUNG
   RUNG wire#w1
      Contact( "THE-1 to T-32"."Alarm Prod" )
      Coil( "Rework_T-32_DB".State.Alarm_Prod )
   END_RUNG
   // the same network as SCL:
   "Rework_T-32_DB".State.HighLevel_Coll_Tank := "AlwaysTRUE" AND "THE-1 to T-32"."High Level Coll Tank";
   "Rework_T-32_DB".State.Alarm_Prod := "AlwaysTRUE" AND "THE-1 to T-32"."Alarm Prod";
END_REGION

REGION Network 54
   RUNG wire#powerrail
      "IO_Valve_Blending_DB"(lock :=, Init := "General_DB".Initial, Reset := "General_DB".Reset)
   END_RUNG
   // the same network as SCL:
   "IO_Valve_Blending_DB"(Init := "General_DB".Initial, Reset := "General_DB".Reset);   // "IO_Valve_Blending"
END_REGION
END_FUNCTION

FUNCTION_BLOCK "Rework"   // FB32, LAD
{ S7_Optimized_Access := 'FALSE' }
VERSION : 0.1
// stored: AutoNumber false, IsIECCheckEnabled false, SetENOAutomatically false, UDAEnableTagReadback false
   VAR_INPUT
      Level_Bypass_JBT : Bool;
      Single_CIP_Cmd : Bool;
      IN_FBAV_Load : Bool;
      IN_FBAV_Transfer : Bool;
      IN_FBP_Transfer : Bool;
      IN_FBP_Transfer_Speed : Real;
      IN_FBP_CIP : Bool;
      IN_FBAV_CIP_Sup : Bool;
      IN_FBAV_CIP_Tank : Bool;
      IN_FBAV_CIP_Line : Bool;
      IN_LT01 : Real;
      IN_FS : Bool;
      CIP_Req_OK : Bool;
      CIP_ON_Progress : Bool;
      CIP_Supply_ON : Bool;
      CIP_Complete : Bool;
      CIPPulse : Bool;
      Filler_Product_Req : Bool;
      Filler_CIP_Req : Bool;
      Loading_Busy : Bool;
      Transfer_Busy : Bool;
   END_VAR
   VAR_OUTPUT
      Out_AV_Load : Bool;
      Out_AV_Transfer : Bool;
      Out_P_Transfer : Bool;
      Out_P_TF_Speed : Real;
      Out_P_CIP : Bool;
      Out_P_Circ : Bool;
      Out_P_Circ_Speed : Real;
      Out_AV_CIP_Line : Bool;
      Out_AV_CIP_Tank : Bool;
      Out_AV_CIP_Filling : Bool;
      CIP_Tank_Req : Bool;
      CIP_Line_Req : Bool;
      CIP_LineOK : Bool;
   END_VAR
   VAR DB_SPECIFIC
      Cmd : Struct
         Inload_Select_Tank : Bool;
         Inload : Bool;   // Start Loading
         Tank_CIP_Req : Bool;
         Line_CIP_Req : Bool;
         Tank_Filling_CIP_Req : Bool;
         CIP_Filling_En : Bool;
         CIP_Line_Req_OK : Bool;
         CIP_Supply_ON : Bool;
         CIP_ON_Progress : Bool;
         Transfer : Bool;   // Water Flushing
         RaadyForTF : Bool;   // Tank Ready for Blending
         Flush_Select : Byte;
         Drain_In : Bool;
         Drain_Transfer : Bool;
         Circulation_CMD_ON : Bool := true;
         free : Bool;
         free_1 : Bool;
         free_2 : Bool;
         free_3 : Bool;
      END_STRUCT;
      Param : Struct
         SP_Level_LL : Real := 10.0;
         SP_Level_ML : Real := 80.0;
         SP_Level_HL : Real := 100.0;
         SupplyPump_SP_Speed : Real := 80.0;
         L_Hi_Lim : Real := 100.0;
         L_Lo_Lim : Real := 0.0;
         L_Hys : Real := 5.0;
         FlushingTime : DInt := 10000;
         CIP_Trf_SP_Speed : Real := 80.0;
         CIP_Ret_ON_SP : Real := 10.0;
         CIP_Ret_OFF_SP : Real;
         Transfer_P_Speed : Real := 60.0;
         Drain_Inload_SP : DInt := 10;
         Drain_Transfer_SP : DInt := 10;
         "Circulation Level" : Real := 50.0;
         free : DInt;
         free_1 : DInt;
         free_2 : Real;
         free_3 : Real;
         free_4 : Real;
      END_STRUCT;
      State : Struct   // Tank in loading state
         Tank_inloading : Bool;
         Tank_inCIP : Bool;
         Tank_Filling_inCIP : Bool;
         Line_inCIP : Bool;
         FIlling_inCIP : Bool;
         Flushing : Bool;
         Tank_LL : Bool;
         Tank_ML : Bool;
         Tank_HL : Bool;
         Inload_Enable : Bool;
         Tank_CIP_Enable : Bool;
         Line_CIP_Enable : Bool;
         Tank_Filling_CIP_Enable : Bool;
         Flushing_Enable : Bool;
         Flush_selected : Byte;
         CIP_Request_OK : Bool;
         CIP_ReturnON : Bool;
         Ready_For_Transfer_EN : Bool;   // Tank Ready for Transfer to Blending
         Ready_For_Transfer : Bool;   // Tank Ready for Transfer to Blending
         HWT_Status : Int;
         Transfer_to_Filling : Bool;
         "Line_AV4&AV5" : Bool;
         "Line_AV1&AV2" : Bool;
         "Line_AV7&AV8" : Bool;
         "Line_AV10&AV11" : Bool;
         "Line_AV5&AV6" : Bool;
         CIP_Line1_ON : Bool;
         CIP_Line2_ON : Bool;
         CIP_Line3_ON : Bool;
         CIP_Line4_ON : Bool;
         Drain_Inload : Bool;
         Drain_Transfer : Bool;
         "Circulation Enable" : Bool;
         Circulation_ON : Bool;
         Tank_Circulation : Bool;
         HighLevel_Coll_Tank : Bool;
         Alarm_Prod : Bool;
         free_2 : Bool;
         free_3 : Bool;
      END_STRUCT;
      alwaysON : Bool;
      L_Hys_Abs : Real;
      Hys_Level_HL : Real;
      Hys_Level_ML : Real;
      Hys_Level_LL : Real;
      Hys_Level_Circ : Real;
      Drain_Inload_MSec : DInt;
      Drain_Inload_Count : IEC_DCOUNTER;
      Drain_Inload_Act { S7_SetPoint := 'True'} : DInt;
      Drain_Transfer_MSec : DInt;
      Drain_Transfer_Count : IEC_DCOUNTER;
      Drain_Transfer_Act : DInt;
      r : Struct
         PosE1 : Bool;
         PosE2 : Bool;
         PosE3 : Bool;
         PosE4 : Bool;
         PosE5 : Bool;
         PosE6 : Bool;
         PosE7 : Bool;
         PosE8 : Bool;
         PosE9 : Bool;
         PosE10 : Bool;
         PosE11 : Bool;
         PosE12 : Bool;
         PosE13 : Bool;
         PosE14 : Bool;
         PosE15 : Bool;
         PosE16 : Bool;
         PosE17 : Bool;
         PosE18 : Bool;
         PosE19 : Bool;
         PosE20 : Bool;
         PosE21 : Bool;
         PosE22 : Bool;
         PosE23 : Bool;
         PosE24 : Bool;
         PosE25 : Bool;
         PosE26 : Bool;
         PosE27 : Bool;
         PosE28 : Bool;
         PosE29 : Bool;
         PosE30 : Bool;
         PosE31 : Bool;
         PosE32 : Bool;
      END_STRUCT;
      Actuator : Struct
         AV_Outlet : Bool;
         AV_Load : Bool;
         AV_Transfer : Bool;
         CIP_Line_Pump : Bool;
         CIP_Tank_Pump : Bool;
         TransferPump : Bool;
         FlushPump : Bool;
         CV_Steam : Bool;
         Pump : Bool;
      END_STRUCT;
      SPumpTim { S7_SetPoint := 'True'} : TON_TIME;
      SAV_CIPLine { S7_SetPoint := 'True'} : TON_TIME;
      SAV_CIPTANK { S7_SetPoint := 'True'} : TON_TIME;
      SAV_CIPFILLING { S7_SetPoint := 'True'} : TON_TIME;
      AVinloadTim { S7_SetPoint := 'True'} : TON_TIME;
      AVOutletTim { S7_SetPoint := 'True'} : TON_TIME;
      Drain_In_Tim { S7_SetPoint := 'True'} : TON_TIME;
      Drain_Out_Tim { S7_SetPoint := 'True'} : TON_TIME;
      "Pump Off Tim" { S7_SetPoint := 'True'} : TON_TIME;
      "Loading_Busy Tim" { S7_SetPoint := 'True'} : TON_TIME;
   END_VAR
   VAR_TEMP   // added for the SCL form of the ladder/FBD networks
      _w1 : Bool;
      _w2 : Bool;
   END_VAR
BEGIN

REGION Network 1: Always ON
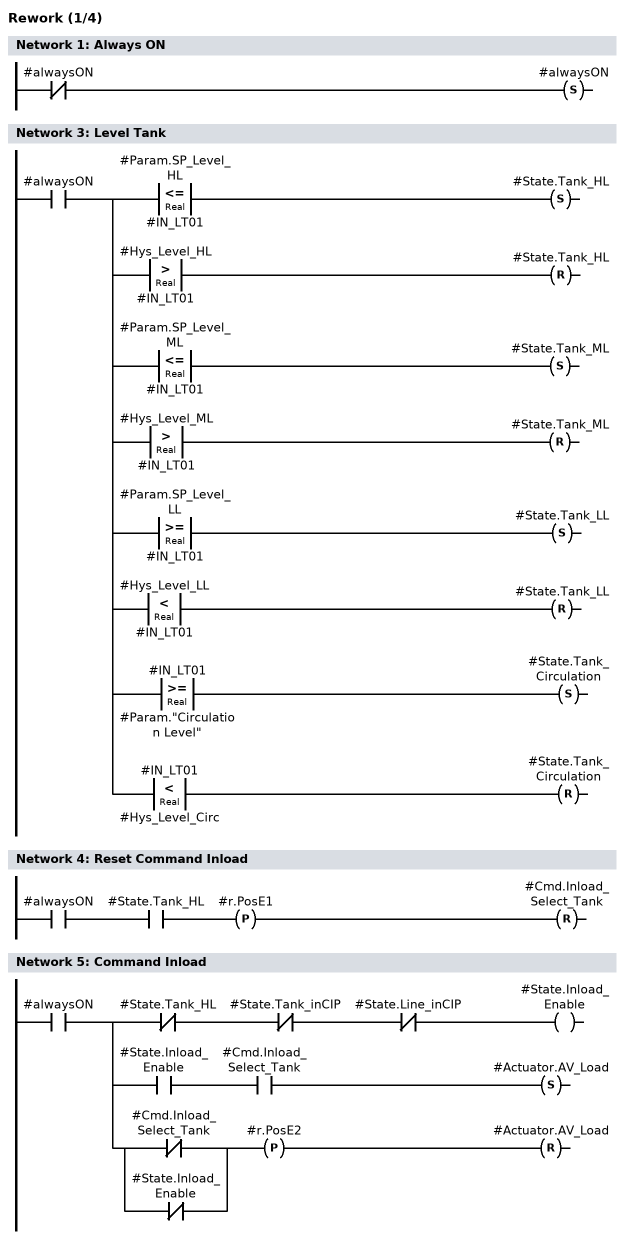
   RUNG wire#powerrail
      I_Contact( #alwaysON )
      S_Coil( #alwaysON )
   END_RUNG
   // the same network as SCL:
   IF NOT #alwaysON THEN #alwaysON := TRUE; END_IF;
END_REGION

NETWORK
TITLE = Hys Calculation
//Level Hys Absolute
      L     #Param.L_Hi_Lim;
      L     #Param.L_Lo_Lim;
      -R;
      L     100.0;
      /R;
      L     #Param.L_Hys;
      *R;
      T     #L_Hys_Abs;
//Tank High Level
      L     #Param.SP_Level_HL;
      L     #L_Hys_Abs;
      -R;
      T     #Hys_Level_HL;
//Tank Mid Level
      L     #Param.SP_Level_ML;
      L     #L_Hys_Abs;
      -R;
      T     #Hys_Level_ML;
//Tank Low Level
      L     #Param.SP_Level_LL;
      L     #L_Hys_Abs;
      +R;
      T     #Hys_Level_LL;
//Level Circulation
      L     #Param."Circulation Level";
      L     #L_Hys_Abs;
      -R;
      T     #Hys_Level_Circ;



REGION Network 3: Level Tank
   RUNG wire#powerrail
      Contact( #alwaysON )
      wire#w1
      { S7_Templates := "SrcType := Real" } LE_Contact(in1 := #Param.SP_Level_HL, in2 := #IN_LT01)
      S_Coil( #State.Tank_HL )
   END_RUNG
   RUNG wire#w1
      { S7_Templates := "SrcType := Real" } GT_Contact(in1 := #Hys_Level_HL, in2 := #IN_LT01)
      R_Coil( #State.Tank_HL )
   END_RUNG
   RUNG wire#w1
      { S7_Templates := "SrcType := Real" } LE_Contact(in1 := #Param.SP_Level_ML, in2 := #IN_LT01)
      S_Coil( #State.Tank_ML )
   END_RUNG
   RUNG wire#w1
      { S7_Templates := "SrcType := Real" } GT_Contact(in1 := #Hys_Level_ML, in2 := #IN_LT01)
      R_Coil( #State.Tank_ML )
   END_RUNG
   RUNG wire#w1
      { S7_Templates := "SrcType := Real" } GE_Contact(in1 := #Param.SP_Level_LL, in2 := #IN_LT01)
      S_Coil( #State.Tank_LL )
   END_RUNG
   RUNG wire#w1
      { S7_Templates := "SrcType := Real" } LT_Contact(in1 := #Hys_Level_LL, in2 := #IN_LT01)
      R_Coil( #State.Tank_LL )
   END_RUNG
   RUNG wire#w1
      { S7_Templates := "SrcType := Real" } GE_Contact(in1 := #IN_LT01, in2 := #Param."Circulation Level")
      S_Coil( #State.Tank_Circulation )
   END_RUNG
   RUNG wire#w1
      { S7_Templates := "SrcType := Real" } LT_Contact(in1 := #IN_LT01, in2 := #Hys_Level_Circ)
      R_Coil( #State.Tank_Circulation )
   END_RUNG
   // the same network as SCL:
   IF #alwaysON AND (#Param.SP_Level_HL <= #IN_LT01) THEN #State.Tank_HL := TRUE; END_IF;
   IF #alwaysON AND (#Hys_Level_HL > #IN_LT01) THEN #State.Tank_HL := FALSE; END_IF;
   IF #alwaysON AND (#Param.SP_Level_ML <= #IN_LT01) THEN #State.Tank_ML := TRUE; END_IF;
   IF #alwaysON AND (#Hys_Level_ML > #IN_LT01) THEN #State.Tank_ML := FALSE; END_IF;
   IF #alwaysON AND (#Param.SP_Level_LL >= #IN_LT01) THEN #State.Tank_LL := TRUE; END_IF;
   IF #alwaysON AND (#Hys_Level_LL < #IN_LT01) THEN #State.Tank_LL := FALSE; END_IF;
   IF #alwaysON AND (#IN_LT01 >= #Param."Circulation Level") THEN #State.Tank_Circulation := TRUE; END_IF;
   IF #alwaysON AND (#IN_LT01 < #Hys_Level_Circ) THEN #State.Tank_Circulation := FALSE; END_IF;
END_REGION

REGION Network 4: Reset Command Inload
   RUNG wire#powerrail
      Contact( #alwaysON )
      Contact( #State.Tank_HL )
      P_Trig( #r.PosE1 )
      R_Coil( #Cmd.Inload_Select_Tank )
   END_RUNG
   // the same network as SCL:
   #_w1 := #alwaysON AND #State.Tank_HL;
   #_w2 := #_w1 AND NOT #r.PosE1;   // rising edge
   #r.PosE1 := #_w1;
   IF #_w2 THEN #Cmd.Inload_Select_Tank := FALSE; END_IF;
END_REGION

REGION Network 5: Command Inload
   RUNG wire#powerrail
      Contact( #alwaysON )
      wire#w1
      I_Contact( #State.Tank_HL )
      I_Contact( #State.Tank_inCIP )
      I_Contact( #State.Line_inCIP )
      Coil( #State.Inload_Enable )
   END_RUNG
   RUNG wire#w1
      Contact( #State.Inload_Enable )
      Contact( #Cmd.Inload_Select_Tank )
      S_Coil( #Actuator.AV_Load )
   END_RUNG
   RUNG wire#w1
      I_Contact( #Cmd.Inload_Select_Tank )
      wire#w2
      P_Trig( #r.PosE2 )
      R_Coil( #Actuator.AV_Load )
   END_RUNG
   RUNG wire#w1
      I_Contact( #State.Inload_Enable )
   END_RUNG wire#w2
   // the same network as SCL:
   #State.Inload_Enable := #alwaysON AND NOT #State.Tank_HL AND NOT #State.Tank_inCIP AND NOT #State.Line_inCIP;
   IF #alwaysON AND #State.Inload_Enable AND #Cmd.Inload_Select_Tank THEN #Actuator.AV_Load := TRUE; END_IF;
   #_w1 := #alwaysON AND (NOT #Cmd.Inload_Select_Tank OR NOT #State.Inload_Enable);
   #_w2 := #_w1 AND NOT #r.PosE2;   // rising edge
   #r.PosE2 := #_w1;
   IF #_w2 THEN #Actuator.AV_Load := FALSE; END_IF;
END_REGION

REGION Network 6: Command Transfer to Filling
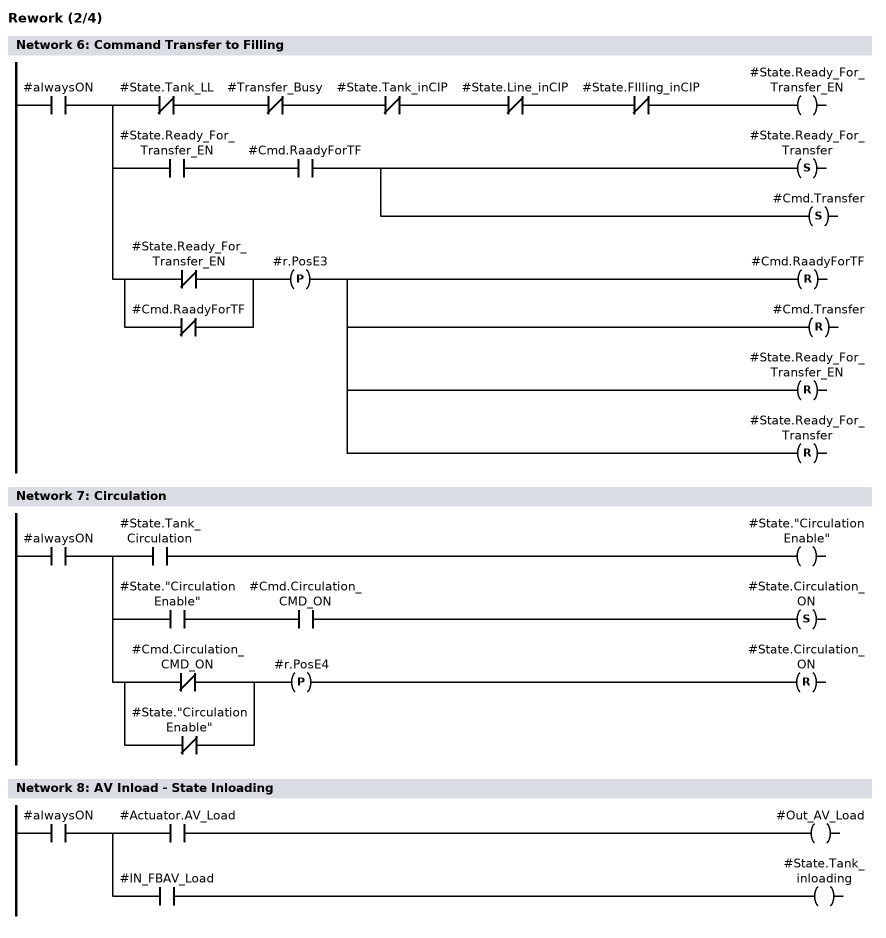
   RUNG wire#powerrail
      Contact( #alwaysON )
      wire#w1
      I_Contact( #State.Tank_LL )
      I_Contact( #Transfer_Busy )
      I_Contact( #State.Tank_inCIP )
      I_Contact( #State.Line_inCIP )
      I_Contact( #State.FIlling_inCIP )
      Coil( #State.Ready_For_Transfer_EN )
   END_RUNG
   RUNG wire#w1
      Contact( #State.Ready_For_Transfer_EN )
      Contact( #Cmd.RaadyForTF )
      wire#w2
      S_Coil( #State.Ready_For_Transfer )
   END_RUNG
   RUNG wire#w2
      S_Coil( #Cmd.Transfer )
   END_RUNG
   RUNG wire#w1
      I_Contact( #State.Ready_For_Transfer_EN )
      wire#w3
      P_Trig( #r.PosE3 )
      wire#w4
      R_Coil( #Cmd.RaadyForTF )
   END_RUNG
   RUNG wire#w1
      I_Contact( #Cmd.RaadyForTF )
   END_RUNG wire#w3
   RUNG wire#w4
      R_Coil( #Cmd.Transfer )
   END_RUNG
   RUNG wire#w4
      R_Coil( #State.Ready_For_Transfer_EN )
   END_RUNG
   RUNG wire#w4
      R_Coil( #State.Ready_For_Transfer )
   END_RUNG
   // the same network as SCL:
   #State.Ready_For_Transfer_EN := #alwaysON AND NOT #State.Tank_LL AND NOT #Transfer_Busy AND NOT #State.Tank_inCIP AND NOT #State.Line_inCIP AND NOT #State.FIlling_inCIP;
   IF #alwaysON AND #State.Ready_For_Transfer_EN AND #Cmd.RaadyForTF THEN
       #State.Ready_For_Transfer := TRUE;
       #Cmd.Transfer := TRUE;
   END_IF;
   #_w1 := #alwaysON AND (NOT #State.Ready_For_Transfer_EN OR NOT #Cmd.RaadyForTF);
   #_w2 := #_w1 AND NOT #r.PosE3;   // rising edge
   #r.PosE3 := #_w1;
   IF #_w2 THEN
       #Cmd.RaadyForTF := FALSE;
       #Cmd.Transfer := FALSE;
       #State.Ready_For_Transfer_EN := FALSE;
       #State.Ready_For_Transfer := FALSE;
   END_IF;
END_REGION

REGION Network 7: Circulation
   RUNG wire#powerrail
      Contact( #alwaysON )
      wire#w1
      Contact( #State.Tank_Circulation )
      Coil( #State."Circulation Enable" )
   END_RUNG
   RUNG wire#w1
      Contact( #State."Circulation Enable" )
      Contact( #Cmd.Circulation_CMD_ON )
      S_Coil( #State.Circulation_ON )
   END_RUNG
   RUNG wire#w1
      I_Contact( #Cmd.Circulation_CMD_ON )
      wire#w2
      P_Trig( #r.PosE4 )
      R_Coil( #State.Circulation_ON )
   END_RUNG
   RUNG wire#w1
      I_Contact( #State."Circulation Enable" )
   END_RUNG wire#w2
   // the same network as SCL:
   #State."Circulation Enable" := #alwaysON AND #State.Tank_Circulation;
   IF #alwaysON AND #State."Circulation Enable" AND #Cmd.Circulation_CMD_ON THEN
       #State.Circulation_ON := TRUE;
   END_IF;
   #_w1 := #alwaysON AND (NOT #Cmd.Circulation_CMD_ON OR NOT #State."Circulation Enable");
   #_w2 := #_w1 AND NOT #r.PosE4;   // rising edge
   #r.PosE4 := #_w1;
   IF #_w2 THEN #State.Circulation_ON := FALSE; END_IF;
END_REGION

REGION Network 8: AV Inload - State Inloading
   RUNG wire#powerrail
      Contact( #alwaysON )
      wire#w1
      Contact( #Actuator.AV_Load )
      Coil( #Out_AV_Load )
   END_RUNG
   RUNG wire#w1
      Contact( #IN_FBAV_Load )
      Coil( #State.Tank_inloading )
   END_RUNG
   // the same network as SCL:
   #Out_AV_Load := #alwaysON AND #Actuator.AV_Load;
   #State.Tank_inloading := #alwaysON AND #IN_FBAV_Load;
END_REGION

REGION Network 9: AV Transfer / Output
